(* IEC 61131-3 sources: LTL-Test-Case-Generation/, 14 files *)

(* ---- SF_DoubleValveMonitoring.st ---- *)
FUNCTION_BLOCK SF_DoubleValveMonitoring
VAR_INPUT
    Activate: BOOL;
    InitTime: TIME := T#500MS;
    S_OutControl: BOOL;
    EDM1: BOOL;
    EDM2: BOOL;
    ValveType: BOOL;
    MonitoringTime: TIME := T#100ms;
    S_StartReset: BOOL;
    Reset: BOOL;
END_VAR
VAR_OUTPUT
    Ready: BOOL;
    S_SafeState: BOOL;
    S_ValveOut: BOOL;
    S_ValveStatus: UINT;
    SafetyDemand: BOOL;
    ResetRequest: BOOL;
    Error: BOOL;
    DiagCode: UINT;
END_VAR
VAR
    T_Init: TON;
    T_Monitoring: TON;
    EDM1_: BOOL;
    EDM2_: BOOL;
    Reset_Before: BOOL;
    S_OutControl_Before: BOOL;
END_VAR

BEGIN

// state changes
IF NOT Activate THEN
    DiagCode := 16#0000;

    T_Init(IN:=0);
    T_Monitoring(IN:=0);

    Ready := FALSE;
    S_SafeState := FALSE;
    S_ValveOut := FALSE;
    SafetyDemand := FALSE;
    ResetRequest := FALSE;
    Error := FALSE;
    S_ValveStatus := DiagCode;

    Reset_Before := FALSE;
    S_OutControl_Before := FALSE;
    IF ValveType THEN
        EDM1_ := EDM1;
        EDM2_ := EDM2;
    ELSE
        EDM1_ := NOT EDM1;
        EDM2_ := NOT EDM2;
    END_IF;

ELSE
    T_Init(PT:=InitTime);
    T_Monitoring(PT:=MonitoringTime);

    IF ValveType THEN
        EDM1_ := EDM1;
        EDM2_ := EDM2;
    ELSE
        EDM1_ := NOT EDM1;
        EDM2_ := NOT EDM2;
    END_IF;

    CASE DiagCode OF
    16#0000:
        T_Init(IN:=0);
        T_Monitoring(IN:=0);
        T_Init(IN:=1, PT:=InitTime);
        DiagCode := 16#83FF;
    16#83FF:
        IF T_Init.Q THEN
            DiagCode := 16#8401;
        END_IF;
    16#8401:
        IF Reset_Before AND Reset THEN
            DiagCode := 16#C001;
        ELSIF NOT Reset_Before AND Reset AND NOT S_OutControl_Before AND S_OutControl AND NOT S_StartReset THEN
            DiagCode := 16#C100;
        ELSIF (NOT Reset_Before AND Reset) OR S_StartReset THEN
            T_Monitoring(IN:=0);T_Monitoring(IN:=1, PT:=MonitoringTime);
            DiagCode := 16#8802;
        END_IF;
    16#C001:
        IF NOT Reset THEN
            DiagCode := 16#8401;
        END_IF;
    16#C100:
        IF NOT Reset THEN
            DiagCode := 16#8401;
        END_IF;
    16#8802:
        IF S_OutControl AND NOT EDM1_ AND NOT EDM2_ THEN
            T_Monitoring(IN:=0);
            DiagCode := 16#C030;
        ELSIF S_OutControl AND EDM1_ AND NOT EDM2_ THEN
            T_Monitoring(IN:=0);
            DiagCode := 16#C020;
        ELSIF S_OutControl AND NOT EDM1_ AND EDM2_ THEN
            T_Monitoring(IN:=0);
            DiagCode := 16#C010;
        ELSIF T_Monitoring.Q AND NOT EDM1_ AND NOT EDM2_ THEN
            DiagCode := 16#C060;
        ELSIF T_Monitoring.Q AND EDM1_ AND NOT EDM2_ THEN
            DiagCode := 16#C050;
        ELSIF T_Monitoring.Q AND NOT EDM1_ AND EDM2_ THEN
            DiagCode := 16#C040;
        ELSIF EDM1_ AND EDM2_ THEN
            T_Monitoring(IN:=0);
            DiagCode := 16#8804;
        END_IF;
    16#8804:
        IF NOT EDM1_ AND NOT EDM2_ THEN
            DiagCode := 16#C060;
        ELSIF EDM1_ AND NOT EDM2_ THEN
            DiagCode := 16#C050;
        ELSIF NOT EDM1_ AND EDM2_ THEN
            DiagCode := 16#C040;
        ELSIF S_OutControl THEN
            T_Monitoring(IN:=0);T_Monitoring(IN:=1, PT:=MonitoringTime);
            DiagCode := 16#8020;
        END_IF;
    16#8020:
        IF T_Monitoring.Q AND EDM1_ AND EDM2_ THEN
            DiagCode := 16#C090;
        ELSIF T_Monitoring.Q AND NOT EDM1_ AND EDM2_ THEN
            DiagCode := 16#C080;
        ELSIF T_Monitoring.Q AND EDM1_ AND NOT EDM2_ THEN
            DiagCode := 16#C070;
        ELSIF NOT S_OutControl THEN
            T_Monitoring(IN:=0);T_Monitoring(IN:=1, PT:=MonitoringTime);
            DiagCode := 16#8802;
        ELSIF NOT EDM1_ AND NOT EDM2_ THEN
            T_Monitoring(IN:=0);
            DiagCode := 16#8010;
        END_IF;
    16#8010:
        IF EDM1_ AND EDM2_ THEN
            DiagCode := 16#C090;
        ELSIF  NOT EDM1_ AND EDM2_ THEN
            DiagCode := 16#C080;
        ELSIF EDM1_ AND NOT EDM2_ THEN
            DiagCode := 16#C070;
        ELSIF NOT S_OutControl THEN
            T_Monitoring(IN:=0);T_Monitoring(IN:=1, PT:=MonitoringTime);
            DiagCode := 16#8802;
        END_IF;
    16#C010:
        IF Reset_Before AND Reset THEN
            DiagCode := DiagCode + 1;
        ELSIF NOT Reset_Before AND Reset AND NOT S_OutControl AND EDM1_ AND EDM2_ THEN
            T_Monitoring(IN:=0);T_Monitoring(IN:=1, PT:=MonitoringTime);
            DiagCode := 16#8802;
        ELSIF NOT S_OutControl THEN
            DiagCode := DiagCode + 16#400;
        END_IF;
    16#C020:
        IF Reset_Before AND Reset THEN
            DiagCode := DiagCode + 1;
        ELSIF NOT Reset_Before AND Reset AND NOT S_OutControl AND EDM1_ AND EDM2_ THEN
            T_Monitoring(IN:=0);T_Monitoring(IN:=1, PT:=MonitoringTime);
            DiagCode := 16#8802;
        ELSIF NOT S_OutControl THEN
            DiagCode := DiagCode + 16#400;
        END_IF;
    16#C030:
        IF Reset_Before AND Reset THEN
            DiagCode := DiagCode + 1;
        ELSIF NOT Reset_Before AND Reset AND NOT S_OutControl AND EDM1_ AND EDM2_ THEN
            T_Monitoring(IN:=0);T_Monitoring(IN:=1, PT:=MonitoringTime);
            DiagCode := 16#8802;
        ELSIF NOT S_OutControl THEN
            DiagCode := DiagCode + 16#400;
        END_IF;
    16#C040:
        IF Reset_Before AND Reset THEN
            DiagCode := DiagCode + 1;
        ELSIF NOT Reset_Before AND Reset AND NOT S_OutControl AND EDM1_ AND EDM2_ THEN
            T_Monitoring(IN:=0);T_Monitoring(IN:=1, PT:=MonitoringTime);
            DiagCode := 16#8802;
        ELSIF NOT S_OutControl THEN
            DiagCode := DiagCode + 16#400;
        END_IF;
    16#C050:
        IF Reset_Before AND Reset THEN
            DiagCode := DiagCode + 1;
        ELSIF NOT Reset_Before AND Reset AND NOT S_OutControl AND EDM1_ AND EDM2_ THEN
            T_Monitoring(IN:=0);T_Monitoring(IN:=1, PT:=MonitoringTime);
            DiagCode := 16#8802;
        ELSIF NOT S_OutControl THEN
            DiagCode := DiagCode + 16#400;
        END_IF;
    16#C060:
        IF Reset_Before AND Reset THEN
            DiagCode := DiagCode + 1;
        ELSIF NOT Reset_Before AND Reset AND NOT S_OutControl AND EDM1_ AND EDM2_ THEN
            T_Monitoring(IN:=0);T_Monitoring(IN:=1, PT:=MonitoringTime);
            DiagCode := 16#8802;
        ELSIF NOT S_OutControl THEN
            DiagCode := DiagCode + 16#400;
        END_IF;
    16#C070:
        IF Reset_Before AND Reset THEN
            DiagCode := DiagCode + 1;
        ELSIF NOT Reset_Before AND Reset AND NOT S_OutControl AND EDM1_ AND EDM2_ THEN
            T_Monitoring(IN:=0);T_Monitoring(IN:=1, PT:=MonitoringTime);
            DiagCode := 16#8802;
        ELSIF NOT S_OutControl THEN
            DiagCode := DiagCode + 16#400;
        END_IF;
    16#C080:
        IF Reset_Before AND Reset THEN
            DiagCode := DiagCode + 1;
        ELSIF NOT Reset_Before AND Reset AND NOT S_OutControl AND EDM1_ AND EDM2_ THEN
            T_Monitoring(IN:=0);T_Monitoring(IN:=1, PT:=MonitoringTime);
            DiagCode := 16#8802;
        ELSIF NOT S_OutControl THEN
            DiagCode := DiagCode + 16#400;
        END_IF;
    16#C090:
        IF Reset_Before AND Reset THEN
            DiagCode := DiagCode + 1;
        ELSIF NOT Reset_Before AND Reset AND NOT S_OutControl AND EDM1_ AND EDM2_ THEN
            T_Monitoring(IN:=0);T_Monitoring(IN:=1, PT:=MonitoringTime);
            DiagCode := 16#8802;
        ELSIF NOT S_OutControl THEN
            DiagCode := DiagCode + 16#400;
        END_IF;
    16#C011:
        IF NOT Reset THEN
            DiagCode := DiagCode - 1;
        END_IF;
    16#C021:
        IF NOT Reset THEN
            DiagCode := DiagCode - 1;
        END_IF;
    16#C031:
        IF NOT Reset THEN
            DiagCode := DiagCode - 1;
        END_IF;
    16#C041:
        IF NOT Reset THEN
            DiagCode := DiagCode - 1;
        END_IF;
    16#C051:
        IF NOT Reset THEN
            DiagCode := DiagCode - 1;
        END_IF;
    16#C061:
        IF NOT Reset THEN
            DiagCode := DiagCode - 1;
        END_IF;
    16#C071:
        IF NOT Reset THEN
            DiagCode := DiagCode - 1;
        END_IF;
    16#C081:
        IF NOT Reset THEN
            DiagCode := DiagCode - 1;
        END_IF;
    16#C091:
        IF NOT Reset THEN
            DiagCode := DiagCode - 1;
        END_IF;
    16#C410:
        IF Reset_Before AND Reset THEN
            DiagCode := DiagCode - 16#400 + 1;
        ELSIF NOT Reset_Before AND Reset AND NOT S_OutControl AND EDM1_ AND EDM2_ THEN
            T_Monitoring(IN:=0);T_Monitoring(IN:=1, PT:=MonitoringTime);
            DiagCode := 16#8802;
        ELSIF S_OutControl THEN
            DiagCode := DiagCode - 16#400;
        END_IF;
    16#C420:
        IF Reset_Before AND Reset THEN
            DiagCode := DiagCode - 16#400 + 1;
        ELSIF NOT Reset_Before AND Reset AND NOT S_OutControl AND EDM1_ AND EDM2_ THEN
            T_Monitoring(IN:=0);T_Monitoring(IN:=1, PT:=MonitoringTime);
            DiagCode := 16#8802;
        ELSIF S_OutControl THEN
            DiagCode := DiagCode - 16#400;
        END_IF;
    16#C430:
        IF Reset_Before AND Reset THEN
            DiagCode := DiagCode - 16#400 + 1;
        ELSIF NOT Reset_Before AND Reset AND NOT S_OutControl AND EDM1_ AND EDM2_ THEN
            T_Monitoring(IN:=0);T_Monitoring(IN:=1, PT:=MonitoringTime);
            DiagCode := 16#8802;
        ELSIF S_OutControl THEN
            DiagCode := DiagCode - 16#400;
        END_IF;
    16#C440:
        IF Reset_Before AND Reset THEN
            DiagCode := DiagCode - 16#400 + 1;
        ELSIF NOT Reset_Before AND Reset AND NOT S_OutControl AND EDM1_ AND EDM2_ THEN
            T_Monitoring(IN:=0);T_Monitoring(IN:=1, PT:=MonitoringTime);
            DiagCode := 16#8802;
        ELSIF S_OutControl THEN
            DiagCode := DiagCode - 16#400;
        END_IF;
    16#C450:
        IF Reset_Before AND Reset THEN
            DiagCode := DiagCode - 16#400 + 1;
        ELSIF NOT Reset_Before AND Reset AND NOT S_OutControl AND EDM1_ AND EDM2_ THEN
            T_Monitoring(IN:=0);T_Monitoring(IN:=1, PT:=MonitoringTime);
            DiagCode := 16#8802;
        ELSIF S_OutControl THEN
            DiagCode := DiagCode - 16#400;
        END_IF;
    16#C460:
        IF Reset_Before AND Reset THEN
            DiagCode := DiagCode - 16#400 + 1;
        ELSIF NOT Reset_Before AND Reset AND NOT S_OutControl AND EDM1_ AND EDM2_ THEN
            T_Monitoring(IN:=0);T_Monitoring(IN:=1, PT:=MonitoringTime);
            DiagCode := 16#8802;
        ELSIF S_OutControl THEN
            DiagCode := DiagCode - 16#400;
        END_IF;
    16#C470:
        IF Reset_Before AND Reset THEN
            DiagCode := DiagCode - 16#400 + 1;
        ELSIF NOT Reset_Before AND Reset AND NOT S_OutControl AND EDM1_ AND EDM2_ THEN
            T_Monitoring(IN:=0);T_Monitoring(IN:=1, PT:=MonitoringTime);
            DiagCode := 16#8802;
        ELSIF S_OutControl THEN
            DiagCode := DiagCode - 16#400;
        END_IF;
    16#C480:
        IF Reset_Before AND Reset THEN
            DiagCode := DiagCode - 16#400 + 1;
        ELSIF NOT Reset_Before AND Reset AND NOT S_OutControl AND EDM1_ AND EDM2_ THEN
            T_Monitoring(IN:=0);T_Monitoring(IN:=1, PT:=MonitoringTime);
            DiagCode := 16#8802;
        ELSIF S_OutControl THEN
            DiagCode := DiagCode - 16#400;
        END_IF;
    16#C490:
        IF Reset_Before AND Reset THEN
            DiagCode := DiagCode - 16#400 + 1;
        ELSIF NOT Reset_Before AND Reset AND NOT S_OutControl AND EDM1_ AND EDM2_ THEN
            T_Monitoring(IN:=0);T_Monitoring(IN:=1, PT:=MonitoringTime);
            DiagCode := 16#8802;
        ELSIF S_OutControl THEN
            DiagCode := DiagCode - 16#400;
        END_IF;
    END_CASE;
    CASE DiagCode OF
    16#C010:
        IF NOT S_OutControl THEN
            DiagCode := DiagCode + 16#400;
        END_IF;
    16#C020:
        IF NOT S_OutControl THEN
            DiagCode := DiagCode + 16#400;
        END_IF;
    16#C030:
        IF NOT S_OutControl THEN
            DiagCode := DiagCode + 16#400;
        END_IF;
    16#C040:
        IF NOT S_OutControl THEN
            DiagCode := DiagCode + 16#400;
        END_IF;
    16#C050:
        IF NOT S_OutControl THEN
            DiagCode := DiagCode + 16#400;
        END_IF;
    16#C060:
        IF NOT S_OutControl THEN
            DiagCode := DiagCode + 16#400;
        END_IF;
    16#C070:
        IF NOT S_OutControl THEN
            DiagCode := DiagCode + 16#400;
        END_IF;
    16#C080:
        IF NOT S_OutControl THEN
            DiagCode := DiagCode + 16#400;
        END_IF;
    16#C090:
        IF NOT S_OutControl THEN
            DiagCode := DiagCode + 16#400;
        END_IF;
    END_CASE;

    // set output variables
    S_ValveStatus := DiagCode;

    IF DiagCode > 16#C000 THEN
        Ready := TRUE;
        S_SafeState := FALSE;
        S_ValveOut := FALSE;
        SafetyDemand := FALSE;
        ResetRequest := FALSE;
        Error := TRUE;
    END_IF;
    IF DiagCode > 16#C400 THEN
        ResetRequest := TRUE;
    END_IF;

    CASE DiagCode OF
    16#83FF:
        Ready := TRUE;
        S_SafeState := FALSE;
        S_ValveOut := FALSE;
        SafetyDemand := FALSE;
        ResetRequest := FALSE;
        Error := FALSE;
    16#8401:
        Ready := TRUE;
        S_SafeState := FALSE;
        S_ValveOut := FALSE;
        SafetyDemand := FALSE;
        ResetRequest := TRUE;
        Error := FALSE;
    16#8802:
        Ready := TRUE;
        S_SafeState := FALSE;
        S_ValveOut := FALSE;
        SafetyDemand := TRUE;
        ResetRequest := FALSE;
        Error := FALSE;
    16#8804:
        Ready := TRUE;
        S_SafeState := TRUE;
        S_ValveOut := FALSE;
        SafetyDemand := TRUE;
        ResetRequest := FALSE;
        Error := FALSE;
    16#8010:
        Ready := TRUE;
        S_SafeState := FALSE;
        S_ValveOut := TRUE;
        SafetyDemand := FALSE;
        ResetRequest := FALSE;
        Error := FALSE;
    16#8020:
        Ready := TRUE;
        S_SafeState := FALSE;
        S_ValveOut := TRUE;
        SafetyDemand := FALSE;
        ResetRequest := FALSE;
        Error := FALSE;
    END_CASE;

    Reset_Before := Reset;
    S_OutControl_Before := S_OutControl;
END_IF;

END_FUNCTION_BLOCK

(* ---- SF_DoubleValveMonitoring_Test.st ---- *)
FUNCTION_BLOCK SF_DoubleValveMonitoring_Test
VAR_INPUT
END_VAR
VAR_OUTPUT
	failed_0: BOOL := FALSE;
	finished_0: BOOL := FALSE;
END_VAR
VAR
	fb_0: SF_DoubleValveMonitoring_BranchCounters;
	waitCounter_0: UINT := 0;
	testState_0: UINT := 0;
END_VAR

IF NOT failed_0 AND NOT finished_0 THEN
CASE testState_0 OF
0:
	fb_0.Activate := FALSE;
	fb_0();
	failed_0 := NOT ((((((((((((NOT (fb_0.Reset_Before) AND NOT (fb_0.S_OutControl_Before)) AND NOT (fb_0.T_Init.Q)) AND NOT (fb_0.T_Monitoring.Q)) AND (fb_0.DiagCode = 0)) AND NOT (fb_0.Ready)) AND NOT (fb_0.S_SafeState)) AND NOT (fb_0.S_ValveOut)) AND (fb_0.S_ValveStatus = fb_0.DiagCode)) AND NOT (fb_0.SafetyDemand)) AND NOT (fb_0.ResetRequest)) AND NOT (fb_0.Error)));
	testState_0 := testState_0 + 1;
1:
	fb_0.Activate := TRUE; fb_0.S_OutControl := FALSE; fb_0.EDM1 := FALSE; fb_0.EDM2 := FALSE; fb_0.ValveType := TRUE; fb_0.S_StartReset := FALSE; fb_0.Reset := FALSE;
	fb_0();
	failed_0 := NOT ((((((((((((NOT (fb_0.Reset_Before) AND NOT (fb_0.S_OutControl_Before)) AND NOT (fb_0.T_Init.Q)) AND NOT (fb_0.T_Monitoring.Q)) AND (fb_0.DiagCode = 33791)) AND fb_0.Ready) AND NOT (fb_0.S_SafeState)) AND NOT (fb_0.S_ValveOut)) AND (fb_0.S_ValveStatus = fb_0.DiagCode)) AND NOT (fb_0.SafetyDemand)) AND NOT (fb_0.ResetRequest)) AND NOT (fb_0.Error)));
	testState_0 := testState_0 + 1;
2:
	IF (fb_0.T_Init.Q AND (fb_0.DiagCode = 33793)) THEN
		waitCounter_0 := 0;
		testState_0 := testState_0 + 1;
	ELSE
		failed_0 := NOT ((NOT (fb_0.Reset_Before) AND (NOT (fb_0.S_OutControl_Before) AND (NOT (fb_0.T_Init.Q) AND (NOT (fb_0.T_Monitoring.Q) AND ((fb_0.DiagCode = 33791) AND (fb_0.Ready AND (NOT (fb_0.S_SafeState) AND (NOT (fb_0.S_ValveOut) AND ((fb_0.S_ValveStatus = fb_0.DiagCode) AND (NOT (fb_0.SafetyDemand) AND (NOT (fb_0.ResetRequest) AND NOT (fb_0.Error)))))))))))));
		IF waitCounter_0 > 100 THEN
			finished_0 := TRUE;
		ELSE
			waitCounter_0 := waitCounter_0 + 1;
			fb_0();
		END_IF
	END_IF
3:
	failed_0 := NOT ((((((((((((NOT (fb_0.Reset_Before) AND NOT (fb_0.S_OutControl_Before)) AND fb_0.T_Init.Q) AND NOT (fb_0.T_Monitoring.Q)) AND (fb_0.DiagCode = 33793)) AND fb_0.Ready) AND NOT (fb_0.S_SafeState)) AND NOT (fb_0.S_ValveOut)) AND (fb_0.S_ValveStatus = fb_0.DiagCode)) AND NOT (fb_0.SafetyDemand)) AND fb_0.ResetRequest) AND NOT (fb_0.Error)));
	testState_0 := testState_0 + 1;
4:
	fb_0.Activate := TRUE; fb_0.S_OutControl := TRUE; fb_0.EDM1 := FALSE; fb_0.EDM2 := FALSE; fb_0.ValveType := TRUE; fb_0.S_StartReset := FALSE; fb_0.Reset := TRUE;
	fb_0();
	failed_0 := NOT ((((((((((((fb_0.Reset_Before AND fb_0.S_OutControl_Before) AND fb_0.T_Init.Q) AND NOT (fb_0.T_Monitoring.Q)) AND (fb_0.DiagCode = 49408)) AND fb_0.Ready) AND NOT (fb_0.S_SafeState)) AND NOT (fb_0.S_ValveOut)) AND (fb_0.S_ValveStatus = fb_0.DiagCode)) AND NOT (fb_0.SafetyDemand)) AND NOT (fb_0.ResetRequest)) AND fb_0.Error));
	testState_0 := testState_0 + 1;
5:
	fb_0.Activate := TRUE; fb_0.S_OutControl := TRUE; fb_0.EDM1 := FALSE; fb_0.EDM2 := FALSE; fb_0.ValveType := TRUE; fb_0.S_StartReset := FALSE; fb_0.Reset := TRUE;
	fb_0();
	failed_0 := NOT ((((((((((((fb_0.Reset_Before AND fb_0.S_OutControl_Before) AND fb_0.T_Init.Q) AND NOT (fb_0.T_Monitoring.Q)) AND (fb_0.DiagCode = 49408)) AND fb_0.Ready) AND NOT (fb_0.S_SafeState)) AND NOT (fb_0.S_ValveOut)) AND (fb_0.S_ValveStatus = fb_0.DiagCode)) AND NOT (fb_0.SafetyDemand)) AND NOT (fb_0.ResetRequest)) AND fb_0.Error));
	testState_0 := testState_0 + 1;
6:
	fb_0.Activate := TRUE; fb_0.S_OutControl := TRUE; fb_0.EDM1 := FALSE; fb_0.EDM2 := FALSE; fb_0.ValveType := TRUE; fb_0.S_StartReset := FALSE; fb_0.Reset := FALSE;
	fb_0();
	failed_0 := NOT ((((((((((((NOT (fb_0.Reset_Before) AND fb_0.S_OutControl_Before) AND fb_0.T_Init.Q) AND NOT (fb_0.T_Monitoring.Q)) AND (fb_0.DiagCode = 33793)) AND fb_0.Ready) AND NOT (fb_0.S_SafeState)) AND NOT (fb_0.S_ValveOut)) AND (fb_0.S_ValveStatus = fb_0.DiagCode)) AND NOT (fb_0.SafetyDemand)) AND fb_0.ResetRequest) AND NOT (fb_0.Error)));
	testState_0 := testState_0 + 1;
7:
	fb_0.Activate := TRUE; fb_0.S_OutControl := FALSE; fb_0.EDM1 := FALSE; fb_0.EDM2 := FALSE; fb_0.ValveType := TRUE; fb_0.S_StartReset := FALSE; fb_0.Reset := FALSE;
	fb_0();
	failed_0 := NOT ((((((((((((NOT (fb_0.Reset_Before) AND NOT (fb_0.S_OutControl_Before)) AND fb_0.T_Init.Q) AND NOT (fb_0.T_Monitoring.Q)) AND (fb_0.DiagCode = 33793)) AND fb_0.Ready) AND NOT (fb_0.S_SafeState)) AND NOT (fb_0.S_ValveOut)) AND (fb_0.S_ValveStatus = fb_0.DiagCode)) AND NOT (fb_0.SafetyDemand)) AND fb_0.ResetRequest) AND NOT (fb_0.Error)));
	testState_0 := testState_0 + 1;
8:
	fb_0.Activate := FALSE; fb_0.S_OutControl := FALSE; fb_0.EDM1 := FALSE; fb_0.EDM2 := FALSE; fb_0.ValveType := TRUE; fb_0.S_StartReset := FALSE; fb_0.Reset := FALSE;
	fb_0();
	failed_0 := NOT ((((((((((((NOT (fb_0.Reset_Before) AND NOT (fb_0.S_OutControl_Before)) AND NOT (fb_0.T_Init.Q)) AND NOT (fb_0.T_Monitoring.Q)) AND (fb_0.DiagCode = 0)) AND NOT (fb_0.Ready)) AND NOT (fb_0.S_SafeState)) AND NOT (fb_0.S_ValveOut)) AND (fb_0.S_ValveStatus = fb_0.DiagCode)) AND NOT (fb_0.SafetyDemand)) AND NOT (fb_0.ResetRequest)) AND NOT (fb_0.Error)));
	testState_0 := testState_0 + 1;
9:
	fb_0.Activate := TRUE; fb_0.S_OutControl := FALSE; fb_0.EDM1 := FALSE; fb_0.EDM2 := FALSE; fb_0.ValveType := TRUE; fb_0.S_StartReset := FALSE; fb_0.Reset := TRUE;
	fb_0();
	failed_0 := NOT ((((((((((((fb_0.Reset_Before AND NOT (fb_0.S_OutControl_Before)) AND NOT (fb_0.T_Init.Q)) AND NOT (fb_0.T_Monitoring.Q)) AND (fb_0.DiagCode = 33791)) AND fb_0.Ready) AND NOT (fb_0.S_SafeState)) AND NOT (fb_0.S_ValveOut)) AND (fb_0.S_ValveStatus = fb_0.DiagCode)) AND NOT (fb_0.SafetyDemand)) AND NOT (fb_0.ResetRequest)) AND NOT (fb_0.Error)));
	testState_0 := testState_0 + 1;
10:
	IF (fb_0.T_Init.Q AND (fb_0.DiagCode = 33793)) THEN
		waitCounter_0 := 0;
		testState_0 := testState_0 + 1;
	ELSE
		failed_0 := NOT ((fb_0.Reset_Before AND (NOT (fb_0.S_OutControl_Before) AND (NOT (fb_0.T_Init.Q) AND (NOT (fb_0.T_Monitoring.Q) AND ((fb_0.DiagCode = 33791) AND (fb_0.Ready AND (NOT (fb_0.S_SafeState) AND (NOT (fb_0.S_ValveOut) AND ((fb_0.S_ValveStatus = fb_0.DiagCode) AND (NOT (fb_0.SafetyDemand) AND (NOT (fb_0.ResetRequest) AND NOT (fb_0.Error)))))))))))));
		IF waitCounter_0 > 100 THEN
			finished_0 := TRUE;
		ELSE
			waitCounter_0 := waitCounter_0 + 1;
			fb_0();
		END_IF
	END_IF
11:
	failed_0 := NOT ((((((((((((fb_0.Reset_Before AND NOT (fb_0.S_OutControl_Before)) AND fb_0.T_Init.Q) AND NOT (fb_0.T_Monitoring.Q)) AND (fb_0.DiagCode = 33793)) AND fb_0.Ready) AND NOT (fb_0.S_SafeState)) AND NOT (fb_0.S_ValveOut)) AND (fb_0.S_ValveStatus = fb_0.DiagCode)) AND NOT (fb_0.SafetyDemand)) AND fb_0.ResetRequest) AND NOT (fb_0.Error)));
	testState_0 := testState_0 + 1;
12:
	fb_0.Activate := TRUE; fb_0.S_OutControl := FALSE; fb_0.EDM1 := FALSE; fb_0.EDM2 := FALSE; fb_0.ValveType := TRUE; fb_0.S_StartReset := FALSE; fb_0.Reset := TRUE;
	fb_0();
	failed_0 := NOT ((((((((((((fb_0.Reset_Before AND NOT (fb_0.S_OutControl_Before)) AND fb_0.T_Init.Q) AND NOT (fb_0.T_Monitoring.Q)) AND (fb_0.DiagCode = 49153)) AND fb_0.Ready) AND NOT (fb_0.S_SafeState)) AND NOT (fb_0.S_ValveOut)) AND (fb_0.S_ValveStatus = fb_0.DiagCode)) AND NOT (fb_0.SafetyDemand)) AND NOT (fb_0.ResetRequest)) AND fb_0.Error));
	testState_0 := testState_0 + 1;
13:
	fb_0.Activate := TRUE; fb_0.S_OutControl := FALSE; fb_0.EDM1 := FALSE; fb_0.EDM2 := FALSE; fb_0.ValveType := TRUE; fb_0.S_StartReset := FALSE; fb_0.Reset := TRUE;
	fb_0();
	failed_0 := NOT ((((((((((((fb_0.Reset_Before AND NOT (fb_0.S_OutControl_Before)) AND fb_0.T_Init.Q) AND NOT (fb_0.T_Monitoring.Q)) AND (fb_0.DiagCode = 49153)) AND fb_0.Ready) AND NOT (fb_0.S_SafeState)) AND NOT (fb_0.S_ValveOut)) AND (fb_0.S_ValveStatus = fb_0.DiagCode)) AND NOT (fb_0.SafetyDemand)) AND NOT (fb_0.ResetRequest)) AND fb_0.Error));
	testState_0 := testState_0 + 1;
14:
	fb_0.Activate := TRUE; fb_0.S_OutControl := FALSE; fb_0.EDM1 := FALSE; fb_0.EDM2 := FALSE; fb_0.ValveType := TRUE; fb_0.S_StartReset := FALSE; fb_0.Reset := FALSE;
	fb_0();
	failed_0 := NOT ((((((((((((NOT (fb_0.Reset_Before) AND NOT (fb_0.S_OutControl_Before)) AND fb_0.T_Init.Q) AND NOT (fb_0.T_Monitoring.Q)) AND (fb_0.DiagCode = 33793)) AND fb_0.Ready) AND NOT (fb_0.S_SafeState)) AND NOT (fb_0.S_ValveOut)) AND (fb_0.S_ValveStatus = fb_0.DiagCode)) AND NOT (fb_0.SafetyDemand)) AND fb_0.ResetRequest) AND NOT (fb_0.Error)));
	testState_0 := testState_0 + 1;
15:
	fb_0.Activate := TRUE; fb_0.S_OutControl := FALSE; fb_0.EDM1 := FALSE; fb_0.EDM2 := FALSE; fb_0.ValveType := TRUE; fb_0.S_StartReset := FALSE; fb_0.Reset := TRUE;
	fb_0();
	failed_0 := NOT ((((((((((((fb_0.Reset_Before AND NOT (fb_0.S_OutControl_Before)) AND fb_0.T_Init.Q) AND NOT (fb_0.T_Monitoring.Q)) AND (fb_0.DiagCode = 34818)) AND fb_0.Ready) AND NOT (fb_0.S_SafeState)) AND NOT (fb_0.S_ValveOut)) AND (fb_0.S_ValveStatus = fb_0.DiagCode)) AND fb_0.SafetyDemand) AND NOT (fb_0.ResetRequest)) AND NOT (fb_0.Error)));
	testState_0 := testState_0 + 1;
16:
	fb_0.Activate := FALSE; fb_0.S_OutControl := FALSE; fb_0.EDM1 := FALSE; fb_0.EDM2 := FALSE; fb_0.ValveType := TRUE; fb_0.S_StartReset := FALSE; fb_0.Reset := FALSE;
	fb_0();
	failed_0 := NOT ((((((((((((NOT (fb_0.Reset_Before) AND NOT (fb_0.S_OutControl_Before)) AND NOT (fb_0.T_Init.Q)) AND NOT (fb_0.T_Monitoring.Q)) AND (fb_0.DiagCode = 0)) AND NOT (fb_0.Ready)) AND NOT (fb_0.S_SafeState)) AND NOT (fb_0.S_ValveOut)) AND (fb_0.S_ValveStatus = fb_0.DiagCode)) AND NOT (fb_0.SafetyDemand)) AND NOT (fb_0.ResetRequest)) AND NOT (fb_0.Error)));
	testState_0 := testState_0 + 1;
17:
	fb_0.Activate := TRUE; fb_0.S_OutControl := FALSE; fb_0.EDM1 := FALSE; fb_0.EDM2 := FALSE; fb_0.ValveType := TRUE; fb_0.S_StartReset := TRUE; fb_0.Reset := FALSE;
	fb_0();
	failed_0 := NOT ((((((((((((NOT (fb_0.Reset_Before) AND NOT (fb_0.S_OutControl_Before)) AND NOT (fb_0.T_Init.Q)) AND NOT (fb_0.T_Monitoring.Q)) AND (fb_0.DiagCode = 33791)) AND fb_0.Ready) AND NOT (fb_0.S_SafeState)) AND NOT (fb_0.S_ValveOut)) AND (fb_0.S_ValveStatus = fb_0.DiagCode)) AND NOT (fb_0.SafetyDemand)) AND NOT (fb_0.ResetRequest)) AND NOT (fb_0.Error)));
	testState_0 := testState_0 + 1;
18:
	IF (fb_0.T_Init.Q AND (fb_0.DiagCode = 33793)) THEN
		waitCounter_0 := 0;
		testState_0 := testState_0 + 1;
	ELSE
		failed_0 := NOT ((NOT (fb_0.Reset_Before) AND (NOT (fb_0.S_OutControl_Before) AND (NOT (fb_0.T_Init.Q) AND (NOT (fb_0.T_Monitoring.Q) AND ((fb_0.DiagCode = 33791) AND (fb_0.Ready AND (NOT (fb_0.S_SafeState) AND (NOT (fb_0.S_ValveOut) AND ((fb_0.S_ValveStatus = fb_0.DiagCode) AND (NOT (fb_0.SafetyDemand) AND (NOT (fb_0.ResetRequest) AND NOT (fb_0.Error)))))))))))));
		IF waitCounter_0 > 100 THEN
			finished_0 := TRUE;
		ELSE
			waitCounter_0 := waitCounter_0 + 1;
			fb_0();
		END_IF
	END_IF
19:
	failed_0 := NOT ((((((((((((NOT (fb_0.Reset_Before) AND NOT (fb_0.S_OutControl_Before)) AND fb_0.T_Init.Q) AND NOT (fb_0.T_Monitoring.Q)) AND (fb_0.DiagCode = 33793)) AND fb_0.Ready) AND NOT (fb_0.S_SafeState)) AND NOT (fb_0.S_ValveOut)) AND (fb_0.S_ValveStatus = fb_0.DiagCode)) AND NOT (fb_0.SafetyDemand)) AND fb_0.ResetRequest) AND NOT (fb_0.Error)));
	testState_0 := testState_0 + 1;
20:
	fb_0.Activate := TRUE; fb_0.S_OutControl := FALSE; fb_0.EDM1 := FALSE; fb_0.EDM2 := TRUE; fb_0.ValveType := TRUE; fb_0.S_StartReset := TRUE; fb_0.Reset := FALSE;
	fb_0();
	failed_0 := NOT ((((((((((((NOT (fb_0.Reset_Before) AND NOT (fb_0.S_OutControl_Before)) AND fb_0.T_Init.Q) AND NOT (fb_0.T_Monitoring.Q)) AND (fb_0.DiagCode = 34818)) AND fb_0.Ready) AND NOT (fb_0.S_SafeState)) AND NOT (fb_0.S_ValveOut)) AND (fb_0.S_ValveStatus = fb_0.DiagCode)) AND fb_0.SafetyDemand) AND NOT (fb_0.ResetRequest)) AND NOT (fb_0.Error)));
	testState_0 := testState_0 + 1;
21:
	IF (fb_0.T_Monitoring.Q AND (fb_0.DiagCode = 50240)) THEN
		waitCounter_0 := 0;
		testState_0 := testState_0 + 1;
	ELSE
		failed_0 := NOT ((NOT (fb_0.Reset_Before) AND (NOT (fb_0.S_OutControl_Before) AND (fb_0.T_Init.Q AND (NOT (fb_0.T_Monitoring.Q) AND ((fb_0.DiagCode = 34818) AND (fb_0.Ready AND (NOT (fb_0.S_SafeState) AND (NOT (fb_0.S_ValveOut) AND ((fb_0.S_ValveStatus = fb_0.DiagCode) AND (fb_0.SafetyDemand AND (NOT (fb_0.ResetRequest) AND NOT (fb_0.Error)))))))))))));
		IF waitCounter_0 > 100 THEN
			finished_0 := TRUE;
		ELSE
			waitCounter_0 := waitCounter_0 + 1;
			fb_0();
		END_IF
	END_IF
22:
	failed_0 := NOT ((((((((((((NOT (fb_0.Reset_Before) AND NOT (fb_0.S_OutControl_Before)) AND fb_0.T_Init.Q) AND fb_0.T_Monitoring.Q) AND (fb_0.DiagCode = 50240)) AND fb_0.Ready) AND NOT (fb_0.S_SafeState)) AND NOT (fb_0.S_ValveOut)) AND (fb_0.S_ValveStatus = fb_0.DiagCode)) AND NOT (fb_0.SafetyDemand)) AND fb_0.ResetRequest) AND fb_0.Error));
	testState_0 := testState_0 + 1;
23:
	fb_0.Activate := TRUE; fb_0.S_OutControl := TRUE; fb_0.EDM1 := FALSE; fb_0.EDM2 := TRUE; fb_0.ValveType := TRUE; fb_0.S_StartReset := TRUE; fb_0.Reset := FALSE;
	fb_0();
	failed_0 := NOT ((((((((((((NOT (fb_0.Reset_Before) AND fb_0.S_OutControl_Before) AND fb_0.T_Init.Q) AND fb_0.T_Monitoring.Q) AND (fb_0.DiagCode = 49216)) AND fb_0.Ready) AND NOT (fb_0.S_SafeState)) AND NOT (fb_0.S_ValveOut)) AND (fb_0.S_ValveStatus = fb_0.DiagCode)) AND NOT (fb_0.SafetyDemand)) AND NOT (fb_0.ResetRequest)) AND fb_0.Error));
	testState_0 := testState_0 + 1;
24:
	fb_0.Activate := TRUE; fb_0.S_OutControl := TRUE; fb_0.EDM1 := FALSE; fb_0.EDM2 := TRUE; fb_0.ValveType := TRUE; fb_0.S_StartReset := TRUE; fb_0.Reset := TRUE;
	fb_0();
	failed_0 := NOT ((((((((((((fb_0.Reset_Before AND fb_0.S_OutControl_Before) AND fb_0.T_Init.Q) AND fb_0.T_Monitoring.Q) AND (fb_0.DiagCode = 49216)) AND fb_0.Ready) AND NOT (fb_0.S_SafeState)) AND NOT (fb_0.S_ValveOut)) AND (fb_0.S_ValveStatus = fb_0.DiagCode)) AND NOT (fb_0.SafetyDemand)) AND NOT (fb_0.ResetRequest)) AND fb_0.Error));
	testState_0 := testState_0 + 1;
25:
	fb_0.Activate := TRUE; fb_0.S_OutControl := TRUE; fb_0.EDM1 := FALSE; fb_0.EDM2 := TRUE; fb_0.ValveType := TRUE; fb_0.S_StartReset := TRUE; fb_0.Reset := TRUE;
	fb_0();
	failed_0 := NOT ((((((((((((fb_0.Reset_Before AND fb_0.S_OutControl_Before) AND fb_0.T_Init.Q) AND fb_0.T_Monitoring.Q) AND (fb_0.DiagCode = 49217)) AND fb_0.Ready) AND NOT (fb_0.S_SafeState)) AND NOT (fb_0.S_ValveOut)) AND (fb_0.S_ValveStatus = fb_0.DiagCode)) AND NOT (fb_0.SafetyDemand)) AND NOT (fb_0.ResetRequest)) AND fb_0.Error));
	testState_0 := testState_0 + 1;
26:
	fb_0.Activate := TRUE; fb_0.S_OutControl := TRUE; fb_0.EDM1 := FALSE; fb_0.EDM2 := TRUE; fb_0.ValveType := TRUE; fb_0.S_StartReset := TRUE; fb_0.Reset := TRUE;
	fb_0();
	failed_0 := NOT ((((((((((((fb_0.Reset_Before AND fb_0.S_OutControl_Before) AND fb_0.T_Init.Q) AND fb_0.T_Monitoring.Q) AND (fb_0.DiagCode = 49217)) AND fb_0.Ready) AND NOT (fb_0.S_SafeState)) AND NOT (fb_0.S_ValveOut)) AND (fb_0.S_ValveStatus = fb_0.DiagCode)) AND NOT (fb_0.SafetyDemand)) AND NOT (fb_0.ResetRequest)) AND fb_0.Error));
	testState_0 := testState_0 + 1;
27:
	fb_0.Activate := TRUE; fb_0.S_OutControl := TRUE; fb_0.EDM1 := FALSE; fb_0.EDM2 := TRUE; fb_0.ValveType := TRUE; fb_0.S_StartReset := TRUE; fb_0.Reset := FALSE;
	fb_0();
	failed_0 := NOT ((((((((((((NOT (fb_0.Reset_Before) AND fb_0.S_OutControl_Before) AND fb_0.T_Init.Q) AND fb_0.T_Monitoring.Q) AND (fb_0.DiagCode = 49216)) AND fb_0.Ready) AND NOT (fb_0.S_SafeState)) AND NOT (fb_0.S_ValveOut)) AND (fb_0.S_ValveStatus = fb_0.DiagCode)) AND NOT (fb_0.SafetyDemand)) AND NOT (fb_0.ResetRequest)) AND fb_0.Error));
	testState_0 := testState_0 + 1;
28:
	fb_0.Activate := TRUE; fb_0.S_OutControl := FALSE; fb_0.EDM1 := FALSE; fb_0.EDM2 := TRUE; fb_0.ValveType := TRUE; fb_0.S_StartReset := TRUE; fb_0.Reset := FALSE;
	fb_0();
	failed_0 := NOT ((((((((((((NOT (fb_0.Reset_Before) AND NOT (fb_0.S_OutControl_Before)) AND fb_0.T_Init.Q) AND fb_0.T_Monitoring.Q) AND (fb_0.DiagCode = 50240)) AND fb_0.Ready) AND NOT (fb_0.S_SafeState)) AND NOT (fb_0.S_ValveOut)) AND (fb_0.S_ValveStatus = fb_0.DiagCode)) AND NOT (fb_0.SafetyDemand)) AND fb_0.ResetRequest) AND fb_0.Error));
	testState_0 := testState_0 + 1;
29:
	fb_0.Activate := TRUE; fb_0.S_OutControl := TRUE; fb_0.EDM1 := FALSE; fb_0.EDM2 := TRUE; fb_0.ValveType := TRUE; fb_0.S_StartReset := TRUE; fb_0.Reset := FALSE;
	fb_0();
	failed_0 := NOT ((((((((((((NOT (fb_0.Reset_Before) AND fb_0.S_OutControl_Before) AND fb_0.T_Init.Q) AND fb_0.T_Monitoring.Q) AND (fb_0.DiagCode = 49216)) AND fb_0.Ready) AND NOT (fb_0.S_SafeState)) AND NOT (fb_0.S_ValveOut)) AND (fb_0.S_ValveStatus = fb_0.DiagCode)) AND NOT (fb_0.SafetyDemand)) AND NOT (fb_0.ResetRequest)) AND fb_0.Error));
	testState_0 := testState_0 + 1;
30:
	fb_0.Activate := TRUE; fb_0.S_OutControl := FALSE; fb_0.EDM1 := TRUE; fb_0.EDM2 := TRUE; fb_0.ValveType := TRUE; fb_0.S_StartReset := TRUE; fb_0.Reset := TRUE;
	fb_0();
	failed_0 := NOT ((((((((((((fb_0.Reset_Before AND NOT (fb_0.S_OutControl_Before)) AND fb_0.T_Init.Q) AND NOT (fb_0.T_Monitoring.Q)) AND (fb_0.DiagCode = 34818)) AND fb_0.Ready) AND NOT (fb_0.S_SafeState)) AND NOT (fb_0.S_ValveOut)) AND (fb_0.S_ValveStatus = fb_0.DiagCode)) AND fb_0.SafetyDemand) AND NOT (fb_0.ResetRequest)) AND NOT (fb_0.Error)));
	testState_0 := testState_0 + 1;
31:
	fb_0.Activate := TRUE; fb_0.S_OutControl := FALSE; fb_0.EDM1 := FALSE; fb_0.EDM2 := TRUE; fb_0.ValveType := TRUE; fb_0.S_StartReset := TRUE; fb_0.Reset := FALSE;
	fb_0();
	failed_0 := NOT ((((((((((((NOT (fb_0.Reset_Before) AND NOT (fb_0.S_OutControl_Before)) AND fb_0.T_Init.Q) AND NOT (fb_0.T_Monitoring.Q)) AND (fb_0.DiagCode = 34818)) AND fb_0.Ready) AND NOT (fb_0.S_SafeState)) AND NOT (fb_0.S_ValveOut)) AND (fb_0.S_ValveStatus = fb_0.DiagCode)) AND fb_0.SafetyDemand) AND NOT (fb_0.ResetRequest)) AND NOT (fb_0.Error)));
	testState_0 := testState_0 + 1;
32:
	IF (fb_0.T_Monitoring.Q AND (fb_0.DiagCode = 50240)) THEN
		waitCounter_0 := 0;
		testState_0 := testState_0 + 1;
	ELSE
		failed_0 := NOT ((NOT (fb_0.Reset_Before) AND (NOT (fb_0.S_OutControl_Before) AND (fb_0.T_Init.Q AND (NOT (fb_0.T_Monitoring.Q) AND ((fb_0.DiagCode = 34818) AND (fb_0.Ready AND (NOT (fb_0.S_SafeState) AND (NOT (fb_0.S_ValveOut) AND ((fb_0.S_ValveStatus = fb_0.DiagCode) AND (fb_0.SafetyDemand AND (NOT (fb_0.ResetRequest) AND NOT (fb_0.Error)))))))))))));
		IF waitCounter_0 > 100 THEN
			finished_0 := TRUE;
		ELSE
			waitCounter_0 := waitCounter_0 + 1;
			fb_0();
		END_IF
	END_IF
33:
	failed_0 := NOT ((((((((((((NOT (fb_0.Reset_Before) AND NOT (fb_0.S_OutControl_Before)) AND fb_0.T_Init.Q) AND fb_0.T_Monitoring.Q) AND (fb_0.DiagCode = 50240)) AND fb_0.Ready) AND NOT (fb_0.S_SafeState)) AND NOT (fb_0.S_ValveOut)) AND (fb_0.S_ValveStatus = fb_0.DiagCode)) AND NOT (fb_0.SafetyDemand)) AND fb_0.ResetRequest) AND fb_0.Error));
	testState_0 := testState_0 + 1;
34:
	fb_0.Activate := TRUE; fb_0.S_OutControl := FALSE; fb_0.EDM1 := FALSE; fb_0.EDM2 := TRUE; fb_0.ValveType := TRUE; fb_0.S_StartReset := TRUE; fb_0.Reset := TRUE;
	fb_0();
	failed_0 := NOT ((((((((((((fb_0.Reset_Before AND NOT (fb_0.S_OutControl_Before)) AND fb_0.T_Init.Q) AND fb_0.T_Monitoring.Q) AND (fb_0.DiagCode = 50240)) AND fb_0.Ready) AND NOT (fb_0.S_SafeState)) AND NOT (fb_0.S_ValveOut)) AND (fb_0.S_ValveStatus = fb_0.DiagCode)) AND NOT (fb_0.SafetyDemand)) AND fb_0.ResetRequest) AND fb_0.Error));
	testState_0 := testState_0 + 1;
35:
	fb_0.Activate := TRUE; fb_0.S_OutControl := FALSE; fb_0.EDM1 := FALSE; fb_0.EDM2 := TRUE; fb_0.ValveType := TRUE; fb_0.S_StartReset := TRUE; fb_0.Reset := TRUE;
	fb_0();
	failed_0 := NOT ((((((((((((fb_0.Reset_Before AND NOT (fb_0.S_OutControl_Before)) AND fb_0.T_Init.Q) AND fb_0.T_Monitoring.Q) AND (fb_0.DiagCode = 49217)) AND fb_0.Ready) AND NOT (fb_0.S_SafeState)) AND NOT (fb_0.S_ValveOut)) AND (fb_0.S_ValveStatus = fb_0.DiagCode)) AND NOT (fb_0.SafetyDemand)) AND NOT (fb_0.ResetRequest)) AND fb_0.Error));
	testState_0 := testState_0 + 1;
36:
	fb_0.Activate := TRUE; fb_0.S_OutControl := FALSE; fb_0.EDM1 := FALSE; fb_0.EDM2 := TRUE; fb_0.ValveType := TRUE; fb_0.S_StartReset := TRUE; fb_0.Reset := FALSE;
	fb_0();
	failed_0 := NOT ((((((((((((NOT (fb_0.Reset_Before) AND NOT (fb_0.S_OutControl_Before)) AND fb_0.T_Init.Q) AND fb_0.T_Monitoring.Q) AND (fb_0.DiagCode = 50240)) AND fb_0.Ready) AND NOT (fb_0.S_SafeState)) AND NOT (fb_0.S_ValveOut)) AND (fb_0.S_ValveStatus = fb_0.DiagCode)) AND NOT (fb_0.SafetyDemand)) AND fb_0.ResetRequest) AND fb_0.Error));
	testState_0 := testState_0 + 1;
37:
	fb_0.Activate := TRUE; fb_0.S_OutControl := FALSE; fb_0.EDM1 := TRUE; fb_0.EDM2 := TRUE; fb_0.ValveType := TRUE; fb_0.S_StartReset := TRUE; fb_0.Reset := TRUE;
	fb_0();
	failed_0 := NOT ((((((((((((fb_0.Reset_Before AND NOT (fb_0.S_OutControl_Before)) AND fb_0.T_Init.Q) AND NOT (fb_0.T_Monitoring.Q)) AND (fb_0.DiagCode = 34818)) AND fb_0.Ready) AND NOT (fb_0.S_SafeState)) AND NOT (fb_0.S_ValveOut)) AND (fb_0.S_ValveStatus = fb_0.DiagCode)) AND fb_0.SafetyDemand) AND NOT (fb_0.ResetRequest)) AND NOT (fb_0.Error)));
	testState_0 := testState_0 + 1;
38:
	fb_0.Activate := TRUE; fb_0.S_OutControl := FALSE; fb_0.EDM1 := TRUE; fb_0.EDM2 := FALSE; fb_0.ValveType := TRUE; fb_0.S_StartReset := TRUE; fb_0.Reset := FALSE;
	fb_0();
	failed_0 := NOT ((((((((((((NOT (fb_0.Reset_Before) AND NOT (fb_0.S_OutControl_Before)) AND fb_0.T_Init.Q) AND NOT (fb_0.T_Monitoring.Q)) AND (fb_0.DiagCode = 34818)) AND fb_0.Ready) AND NOT (fb_0.S_SafeState)) AND NOT (fb_0.S_ValveOut)) AND (fb_0.S_ValveStatus = fb_0.DiagCode)) AND fb_0.SafetyDemand) AND NOT (fb_0.ResetRequest)) AND NOT (fb_0.Error)));
	testState_0 := testState_0 + 1;
39:
	IF (fb_0.T_Monitoring.Q AND (fb_0.DiagCode = 50256)) THEN
		waitCounter_0 := 0;
		testState_0 := testState_0 + 1;
	ELSE
		failed_0 := NOT ((NOT (fb_0.Reset_Before) AND (NOT (fb_0.S_OutControl_Before) AND (fb_0.T_Init.Q AND (NOT (fb_0.T_Monitoring.Q) AND ((fb_0.DiagCode = 34818) AND (fb_0.Ready AND (NOT (fb_0.S_SafeState) AND (NOT (fb_0.S_ValveOut) AND ((fb_0.S_ValveStatus = fb_0.DiagCode) AND (fb_0.SafetyDemand AND (NOT (fb_0.ResetRequest) AND NOT (fb_0.Error)))))))))))));
		IF waitCounter_0 > 100 THEN
			finished_0 := TRUE;
		ELSE
			waitCounter_0 := waitCounter_0 + 1;
			fb_0();
		END_IF
	END_IF
40:
	failed_0 := NOT ((((((((((((NOT (fb_0.Reset_Before) AND NOT (fb_0.S_OutControl_Before)) AND fb_0.T_Init.Q) AND fb_0.T_Monitoring.Q) AND (fb_0.DiagCode = 50256)) AND fb_0.Ready) AND NOT (fb_0.S_SafeState)) AND NOT (fb_0.S_ValveOut)) AND (fb_0.S_ValveStatus = fb_0.DiagCode)) AND NOT (fb_0.SafetyDemand)) AND fb_0.ResetRequest) AND fb_0.Error));
	testState_0 := testState_0 + 1;
41:
	fb_0.Activate := TRUE; fb_0.S_OutControl := TRUE; fb_0.EDM1 := TRUE; fb_0.EDM2 := FALSE; fb_0.ValveType := TRUE; fb_0.S_StartReset := TRUE; fb_0.Reset := FALSE;
	fb_0();
	failed_0 := NOT ((((((((((((NOT (fb_0.Reset_Before) AND fb_0.S_OutControl_Before) AND fb_0.T_Init.Q) AND fb_0.T_Monitoring.Q) AND (fb_0.DiagCode = 49232)) AND fb_0.Ready) AND NOT (fb_0.S_SafeState)) AND NOT (fb_0.S_ValveOut)) AND (fb_0.S_ValveStatus = fb_0.DiagCode)) AND NOT (fb_0.SafetyDemand)) AND NOT (fb_0.ResetRequest)) AND fb_0.Error));
	testState_0 := testState_0 + 1;
42:
	fb_0.Activate := TRUE; fb_0.S_OutControl := TRUE; fb_0.EDM1 := TRUE; fb_0.EDM2 := FALSE; fb_0.ValveType := TRUE; fb_0.S_StartReset := TRUE; fb_0.Reset := TRUE;
	fb_0();
	failed_0 := NOT ((((((((((((fb_0.Reset_Before AND fb_0.S_OutControl_Before) AND fb_0.T_Init.Q) AND fb_0.T_Monitoring.Q) AND (fb_0.DiagCode = 49232)) AND fb_0.Ready) AND NOT (fb_0.S_SafeState)) AND NOT (fb_0.S_ValveOut)) AND (fb_0.S_ValveStatus = fb_0.DiagCode)) AND NOT (fb_0.SafetyDemand)) AND NOT (fb_0.ResetRequest)) AND fb_0.Error));
	testState_0 := testState_0 + 1;
43:
	fb_0.Activate := TRUE; fb_0.S_OutControl := TRUE; fb_0.EDM1 := TRUE; fb_0.EDM2 := FALSE; fb_0.ValveType := TRUE; fb_0.S_StartReset := TRUE; fb_0.Reset := TRUE;
	fb_0();
	failed_0 := NOT ((((((((((((fb_0.Reset_Before AND fb_0.S_OutControl_Before) AND fb_0.T_Init.Q) AND fb_0.T_Monitoring.Q) AND (fb_0.DiagCode = 49233)) AND fb_0.Ready) AND NOT (fb_0.S_SafeState)) AND NOT (fb_0.S_ValveOut)) AND (fb_0.S_ValveStatus = fb_0.DiagCode)) AND NOT (fb_0.SafetyDemand)) AND NOT (fb_0.ResetRequest)) AND fb_0.Error));
	testState_0 := testState_0 + 1;
44:
	fb_0.Activate := TRUE; fb_0.S_OutControl := TRUE; fb_0.EDM1 := TRUE; fb_0.EDM2 := FALSE; fb_0.ValveType := TRUE; fb_0.S_StartReset := TRUE; fb_0.Reset := TRUE;
	fb_0();
	failed_0 := NOT ((((((((((((fb_0.Reset_Before AND fb_0.S_OutControl_Before) AND fb_0.T_Init.Q) AND fb_0.T_Monitoring.Q) AND (fb_0.DiagCode = 49233)) AND fb_0.Ready) AND NOT (fb_0.S_SafeState)) AND NOT (fb_0.S_ValveOut)) AND (fb_0.S_ValveStatus = fb_0.DiagCode)) AND NOT (fb_0.SafetyDemand)) AND NOT (fb_0.ResetRequest)) AND fb_0.Error));
	testState_0 := testState_0 + 1;
45:
	fb_0.Activate := TRUE; fb_0.S_OutControl := TRUE; fb_0.EDM1 := TRUE; fb_0.EDM2 := FALSE; fb_0.ValveType := TRUE; fb_0.S_StartReset := TRUE; fb_0.Reset := FALSE;
	fb_0();
	failed_0 := NOT ((((((((((((NOT (fb_0.Reset_Before) AND fb_0.S_OutControl_Before) AND fb_0.T_Init.Q) AND fb_0.T_Monitoring.Q) AND (fb_0.DiagCode = 49232)) AND fb_0.Ready) AND NOT (fb_0.S_SafeState)) AND NOT (fb_0.S_ValveOut)) AND (fb_0.S_ValveStatus = fb_0.DiagCode)) AND NOT (fb_0.SafetyDemand)) AND NOT (fb_0.ResetRequest)) AND fb_0.Error));
	testState_0 := testState_0 + 1;
46:
	fb_0.Activate := TRUE; fb_0.S_OutControl := FALSE; fb_0.EDM1 := TRUE; fb_0.EDM2 := FALSE; fb_0.ValveType := TRUE; fb_0.S_StartReset := TRUE; fb_0.Reset := FALSE;
	fb_0();
	failed_0 := NOT ((((((((((((NOT (fb_0.Reset_Before) AND NOT (fb_0.S_OutControl_Before)) AND fb_0.T_Init.Q) AND fb_0.T_Monitoring.Q) AND (fb_0.DiagCode = 50256)) AND fb_0.Ready) AND NOT (fb_0.S_SafeState)) AND NOT (fb_0.S_ValveOut)) AND (fb_0.S_ValveStatus = fb_0.DiagCode)) AND NOT (fb_0.SafetyDemand)) AND fb_0.ResetRequest) AND fb_0.Error));
	testState_0 := testState_0 + 1;
47:
	fb_0.Activate := TRUE; fb_0.S_OutControl := TRUE; fb_0.EDM1 := TRUE; fb_0.EDM2 := FALSE; fb_0.ValveType := TRUE; fb_0.S_StartReset := TRUE; fb_0.Reset := FALSE;
	fb_0();
	failed_0 := NOT ((((((((((((NOT (fb_0.Reset_Before) AND fb_0.S_OutControl_Before) AND fb_0.T_Init.Q) AND fb_0.T_Monitoring.Q) AND (fb_0.DiagCode = 49232)) AND fb_0.Ready) AND NOT (fb_0.S_SafeState)) AND NOT (fb_0.S_ValveOut)) AND (fb_0.S_ValveStatus = fb_0.DiagCode)) AND NOT (fb_0.SafetyDemand)) AND NOT (fb_0.ResetRequest)) AND fb_0.Error));
	testState_0 := testState_0 + 1;
48:
	fb_0.Activate := TRUE; fb_0.S_OutControl := FALSE; fb_0.EDM1 := TRUE; fb_0.EDM2 := TRUE; fb_0.ValveType := TRUE; fb_0.S_StartReset := TRUE; fb_0.Reset := TRUE;
	fb_0();
	failed_0 := NOT ((((((((((((fb_0.Reset_Before AND NOT (fb_0.S_OutControl_Before)) AND fb_0.T_Init.Q) AND NOT (fb_0.T_Monitoring.Q)) AND (fb_0.DiagCode = 34818)) AND fb_0.Ready) AND NOT (fb_0.S_SafeState)) AND NOT (fb_0.S_ValveOut)) AND (fb_0.S_ValveStatus = fb_0.DiagCode)) AND fb_0.SafetyDemand) AND NOT (fb_0.ResetRequest)) AND NOT (fb_0.Error)));
	testState_0 := testState_0 + 1;
49:
	fb_0.Activate := TRUE; fb_0.S_OutControl := FALSE; fb_0.EDM1 := TRUE; fb_0.EDM2 := FALSE; fb_0.ValveType := TRUE; fb_0.S_StartReset := TRUE; fb_0.Reset := FALSE;
	fb_0();
	failed_0 := NOT ((((((((((((NOT (fb_0.Reset_Before) AND NOT (fb_0.S_OutControl_Before)) AND fb_0.T_Init.Q) AND NOT (fb_0.T_Monitoring.Q)) AND (fb_0.DiagCode = 34818)) AND fb_0.Ready) AND NOT (fb_0.S_SafeState)) AND NOT (fb_0.S_ValveOut)) AND (fb_0.S_ValveStatus = fb_0.DiagCode)) AND fb_0.SafetyDemand) AND NOT (fb_0.ResetRequest)) AND NOT (fb_0.Error)));
	testState_0 := testState_0 + 1;
50:
	IF (fb_0.T_Monitoring.Q AND (fb_0.DiagCode = 50256)) THEN
		waitCounter_0 := 0;
		testState_0 := testState_0 + 1;
	ELSE
		failed_0 := NOT ((NOT (fb_0.Reset_Before) AND (NOT (fb_0.S_OutControl_Before) AND (fb_0.T_Init.Q AND (NOT (fb_0.T_Monitoring.Q) AND ((fb_0.DiagCode = 34818) AND (fb_0.Ready AND (NOT (fb_0.S_SafeState) AND (NOT (fb_0.S_ValveOut) AND ((fb_0.S_ValveStatus = fb_0.DiagCode) AND (fb_0.SafetyDemand AND (NOT (fb_0.ResetRequest) AND NOT (fb_0.Error)))))))))))));
		IF waitCounter_0 > 100 THEN
			finished_0 := TRUE;
		ELSE
			waitCounter_0 := waitCounter_0 + 1;
			fb_0();
		END_IF
	END_IF
51:
	failed_0 := NOT ((((((((((((NOT (fb_0.Reset_Before) AND NOT (fb_0.S_OutControl_Before)) AND fb_0.T_Init.Q) AND fb_0.T_Monitoring.Q) AND (fb_0.DiagCode = 50256)) AND fb_0.Ready) AND NOT (fb_0.S_SafeState)) AND NOT (fb_0.S_ValveOut)) AND (fb_0.S_ValveStatus = fb_0.DiagCode)) AND NOT (fb_0.SafetyDemand)) AND fb_0.ResetRequest) AND fb_0.Error));
	testState_0 := testState_0 + 1;
52:
	fb_0.Activate := TRUE; fb_0.S_OutControl := FALSE; fb_0.EDM1 := TRUE; fb_0.EDM2 := FALSE; fb_0.ValveType := TRUE; fb_0.S_StartReset := TRUE; fb_0.Reset := TRUE;
	fb_0();
	failed_0 := NOT ((((((((((((fb_0.Reset_Before AND NOT (fb_0.S_OutControl_Before)) AND fb_0.T_Init.Q) AND fb_0.T_Monitoring.Q) AND (fb_0.DiagCode = 50256)) AND fb_0.Ready) AND NOT (fb_0.S_SafeState)) AND NOT (fb_0.S_ValveOut)) AND (fb_0.S_ValveStatus = fb_0.DiagCode)) AND NOT (fb_0.SafetyDemand)) AND fb_0.ResetRequest) AND fb_0.Error));
	testState_0 := testState_0 + 1;
53:
	fb_0.Activate := TRUE; fb_0.S_OutControl := FALSE; fb_0.EDM1 := TRUE; fb_0.EDM2 := FALSE; fb_0.ValveType := TRUE; fb_0.S_StartReset := TRUE; fb_0.Reset := TRUE;
	fb_0();
	failed_0 := NOT ((((((((((((fb_0.Reset_Before AND NOT (fb_0.S_OutControl_Before)) AND fb_0.T_Init.Q) AND fb_0.T_Monitoring.Q) AND (fb_0.DiagCode = 49233)) AND fb_0.Ready) AND NOT (fb_0.S_SafeState)) AND NOT (fb_0.S_ValveOut)) AND (fb_0.S_ValveStatus = fb_0.DiagCode)) AND NOT (fb_0.SafetyDemand)) AND NOT (fb_0.ResetRequest)) AND fb_0.Error));
	testState_0 := testState_0 + 1;
54:
	fb_0.Activate := TRUE; fb_0.S_OutControl := FALSE; fb_0.EDM1 := TRUE; fb_0.EDM2 := FALSE; fb_0.ValveType := TRUE; fb_0.S_StartReset := TRUE; fb_0.Reset := FALSE;
	fb_0();
	failed_0 := NOT ((((((((((((NOT (fb_0.Reset_Before) AND NOT (fb_0.S_OutControl_Before)) AND fb_0.T_Init.Q) AND fb_0.T_Monitoring.Q) AND (fb_0.DiagCode = 50256)) AND fb_0.Ready) AND NOT (fb_0.S_SafeState)) AND NOT (fb_0.S_ValveOut)) AND (fb_0.S_ValveStatus = fb_0.DiagCode)) AND NOT (fb_0.SafetyDemand)) AND fb_0.ResetRequest) AND fb_0.Error));
	testState_0 := testState_0 + 1;
55:
	fb_0.Activate := TRUE; fb_0.S_OutControl := FALSE; fb_0.EDM1 := TRUE; fb_0.EDM2 := TRUE; fb_0.ValveType := TRUE; fb_0.S_StartReset := TRUE; fb_0.Reset := TRUE;
	fb_0();
	failed_0 := NOT ((((((((((((fb_0.Reset_Before AND NOT (fb_0.S_OutControl_Before)) AND fb_0.T_Init.Q) AND NOT (fb_0.T_Monitoring.Q)) AND (fb_0.DiagCode = 34818)) AND fb_0.Ready) AND NOT (fb_0.S_SafeState)) AND NOT (fb_0.S_ValveOut)) AND (fb_0.S_ValveStatus = fb_0.DiagCode)) AND fb_0.SafetyDemand) AND NOT (fb_0.ResetRequest)) AND NOT (fb_0.Error)));
	testState_0 := testState_0 + 1;
56:
	fb_0.Activate := TRUE; fb_0.S_OutControl := FALSE; fb_0.EDM1 := FALSE; fb_0.EDM2 := FALSE; fb_0.ValveType := TRUE; fb_0.S_StartReset := TRUE; fb_0.Reset := FALSE;
	fb_0();
	failed_0 := NOT ((((((((((((NOT (fb_0.Reset_Before) AND NOT (fb_0.S_OutControl_Before)) AND fb_0.T_Init.Q) AND NOT (fb_0.T_Monitoring.Q)) AND (fb_0.DiagCode = 34818)) AND fb_0.Ready) AND NOT (fb_0.S_SafeState)) AND NOT (fb_0.S_ValveOut)) AND (fb_0.S_ValveStatus = fb_0.DiagCode)) AND fb_0.SafetyDemand) AND NOT (fb_0.ResetRequest)) AND NOT (fb_0.Error)));
	testState_0 := testState_0 + 1;
57:
	IF (fb_0.T_Monitoring.Q AND (fb_0.DiagCode = 50272)) THEN
		waitCounter_0 := 0;
		testState_0 := testState_0 + 1;
	ELSE
		failed_0 := NOT ((NOT (fb_0.Reset_Before) AND (NOT (fb_0.S_OutControl_Before) AND (fb_0.T_Init.Q AND (NOT (fb_0.T_Monitoring.Q) AND ((fb_0.DiagCode = 34818) AND (fb_0.Ready AND (NOT (fb_0.S_SafeState) AND (NOT (fb_0.S_ValveOut) AND ((fb_0.S_ValveStatus = fb_0.DiagCode) AND (fb_0.SafetyDemand AND (NOT (fb_0.ResetRequest) AND NOT (fb_0.Error)))))))))))));
		IF waitCounter_0 > 100 THEN
			finished_0 := TRUE;
		ELSE
			waitCounter_0 := waitCounter_0 + 1;
			fb_0();
		END_IF
	END_IF
58:
	failed_0 := NOT ((((((((((((NOT (fb_0.Reset_Before) AND NOT (fb_0.S_OutControl_Before)) AND fb_0.T_Init.Q) AND fb_0.T_Monitoring.Q) AND (fb_0.DiagCode = 50272)) AND fb_0.Ready) AND NOT (fb_0.S_SafeState)) AND NOT (fb_0.S_ValveOut)) AND (fb_0.S_ValveStatus = fb_0.DiagCode)) AND NOT (fb_0.SafetyDemand)) AND fb_0.ResetRequest) AND fb_0.Error));
	testState_0 := testState_0 + 1;
59:
	fb_0.Activate := TRUE; fb_0.S_OutControl := TRUE; fb_0.EDM1 := FALSE; fb_0.EDM2 := FALSE; fb_0.ValveType := TRUE; fb_0.S_StartReset := TRUE; fb_0.Reset := FALSE;
	fb_0();
	failed_0 := NOT ((((((((((((NOT (fb_0.Reset_Before) AND fb_0.S_OutControl_Before) AND fb_0.T_Init.Q) AND fb_0.T_Monitoring.Q) AND (fb_0.DiagCode = 49248)) AND fb_0.Ready) AND NOT (fb_0.S_SafeState)) AND NOT (fb_0.S_ValveOut)) AND (fb_0.S_ValveStatus = fb_0.DiagCode)) AND NOT (fb_0.SafetyDemand)) AND NOT (fb_0.ResetRequest)) AND fb_0.Error));
	testState_0 := testState_0 + 1;
60:
	fb_0.Activate := TRUE; fb_0.S_OutControl := TRUE; fb_0.EDM1 := FALSE; fb_0.EDM2 := FALSE; fb_0.ValveType := TRUE; fb_0.S_StartReset := TRUE; fb_0.Reset := TRUE;
	fb_0();
	failed_0 := NOT ((((((((((((fb_0.Reset_Before AND fb_0.S_OutControl_Before) AND fb_0.T_Init.Q) AND fb_0.T_Monitoring.Q) AND (fb_0.DiagCode = 49248)) AND fb_0.Ready) AND NOT (fb_0.S_SafeState)) AND NOT (fb_0.S_ValveOut)) AND (fb_0.S_ValveStatus = fb_0.DiagCode)) AND NOT (fb_0.SafetyDemand)) AND NOT (fb_0.ResetRequest)) AND fb_0.Error));
	testState_0 := testState_0 + 1;
61:
	fb_0.Activate := TRUE; fb_0.S_OutControl := TRUE; fb_0.EDM1 := FALSE; fb_0.EDM2 := FALSE; fb_0.ValveType := TRUE; fb_0.S_StartReset := TRUE; fb_0.Reset := TRUE;
	fb_0();
	failed_0 := NOT ((((((((((((fb_0.Reset_Before AND fb_0.S_OutControl_Before) AND fb_0.T_Init.Q) AND fb_0.T_Monitoring.Q) AND (fb_0.DiagCode = 49249)) AND fb_0.Ready) AND NOT (fb_0.S_SafeState)) AND NOT (fb_0.S_ValveOut)) AND (fb_0.S_ValveStatus = fb_0.DiagCode)) AND NOT (fb_0.SafetyDemand)) AND NOT (fb_0.ResetRequest)) AND fb_0.Error));
	testState_0 := testState_0 + 1;
62:
	fb_0.Activate := TRUE; fb_0.S_OutControl := TRUE; fb_0.EDM1 := FALSE; fb_0.EDM2 := FALSE; fb_0.ValveType := TRUE; fb_0.S_StartReset := TRUE; fb_0.Reset := TRUE;
	fb_0();
	failed_0 := NOT ((((((((((((fb_0.Reset_Before AND fb_0.S_OutControl_Before) AND fb_0.T_Init.Q) AND fb_0.T_Monitoring.Q) AND (fb_0.DiagCode = 49249)) AND fb_0.Ready) AND NOT (fb_0.S_SafeState)) AND NOT (fb_0.S_ValveOut)) AND (fb_0.S_ValveStatus = fb_0.DiagCode)) AND NOT (fb_0.SafetyDemand)) AND NOT (fb_0.ResetRequest)) AND fb_0.Error));
	testState_0 := testState_0 + 1;
63:
	fb_0.Activate := TRUE; fb_0.S_OutControl := TRUE; fb_0.EDM1 := FALSE; fb_0.EDM2 := FALSE; fb_0.ValveType := TRUE; fb_0.S_StartReset := TRUE; fb_0.Reset := FALSE;
	fb_0();
	failed_0 := NOT ((((((((((((NOT (fb_0.Reset_Before) AND fb_0.S_OutControl_Before) AND fb_0.T_Init.Q) AND fb_0.T_Monitoring.Q) AND (fb_0.DiagCode = 49248)) AND fb_0.Ready) AND NOT (fb_0.S_SafeState)) AND NOT (fb_0.S_ValveOut)) AND (fb_0.S_ValveStatus = fb_0.DiagCode)) AND NOT (fb_0.SafetyDemand)) AND NOT (fb_0.ResetRequest)) AND fb_0.Error));
	testState_0 := testState_0 + 1;
64:
	fb_0.Activate := TRUE; fb_0.S_OutControl := FALSE; fb_0.EDM1 := FALSE; fb_0.EDM2 := FALSE; fb_0.ValveType := TRUE; fb_0.S_StartReset := TRUE; fb_0.Reset := FALSE;
	fb_0();
	failed_0 := NOT ((((((((((((NOT (fb_0.Reset_Before) AND NOT (fb_0.S_OutControl_Before)) AND fb_0.T_Init.Q) AND fb_0.T_Monitoring.Q) AND (fb_0.DiagCode = 50272)) AND fb_0.Ready) AND NOT (fb_0.S_SafeState)) AND NOT (fb_0.S_ValveOut)) AND (fb_0.S_ValveStatus = fb_0.DiagCode)) AND NOT (fb_0.SafetyDemand)) AND fb_0.ResetRequest) AND fb_0.Error));
	testState_0 := testState_0 + 1;
65:
	fb_0.Activate := TRUE; fb_0.S_OutControl := TRUE; fb_0.EDM1 := FALSE; fb_0.EDM2 := FALSE; fb_0.ValveType := TRUE; fb_0.S_StartReset := TRUE; fb_0.Reset := FALSE;
	fb_0();
	failed_0 := NOT ((((((((((((NOT (fb_0.Reset_Before) AND fb_0.S_OutControl_Before) AND fb_0.T_Init.Q) AND fb_0.T_Monitoring.Q) AND (fb_0.DiagCode = 49248)) AND fb_0.Ready) AND NOT (fb_0.S_SafeState)) AND NOT (fb_0.S_ValveOut)) AND (fb_0.S_ValveStatus = fb_0.DiagCode)) AND NOT (fb_0.SafetyDemand)) AND NOT (fb_0.ResetRequest)) AND fb_0.Error));
	testState_0 := testState_0 + 1;
66:
	fb_0.Activate := TRUE; fb_0.S_OutControl := FALSE; fb_0.EDM1 := TRUE; fb_0.EDM2 := TRUE; fb_0.ValveType := TRUE; fb_0.S_StartReset := TRUE; fb_0.Reset := TRUE;
	fb_0();
	failed_0 := NOT ((((((((((((fb_0.Reset_Before AND NOT (fb_0.S_OutControl_Before)) AND fb_0.T_Init.Q) AND NOT (fb_0.T_Monitoring.Q)) AND (fb_0.DiagCode = 34818)) AND fb_0.Ready) AND NOT (fb_0.S_SafeState)) AND NOT (fb_0.S_ValveOut)) AND (fb_0.S_ValveStatus = fb_0.DiagCode)) AND fb_0.SafetyDemand) AND NOT (fb_0.ResetRequest)) AND NOT (fb_0.Error)));
	testState_0 := testState_0 + 1;
67:
	fb_0.Activate := TRUE; fb_0.S_OutControl := FALSE; fb_0.EDM1 := FALSE; fb_0.EDM2 := FALSE; fb_0.ValveType := TRUE; fb_0.S_StartReset := TRUE; fb_0.Reset := FALSE;
	fb_0();
	failed_0 := NOT ((((((((((((NOT (fb_0.Reset_Before) AND NOT (fb_0.S_OutControl_Before)) AND fb_0.T_Init.Q) AND NOT (fb_0.T_Monitoring.Q)) AND (fb_0.DiagCode = 34818)) AND fb_0.Ready) AND NOT (fb_0.S_SafeState)) AND NOT (fb_0.S_ValveOut)) AND (fb_0.S_ValveStatus = fb_0.DiagCode)) AND fb_0.SafetyDemand) AND NOT (fb_0.ResetRequest)) AND NOT (fb_0.Error)));
	testState_0 := testState_0 + 1;
68:
	IF (fb_0.T_Monitoring.Q AND (fb_0.DiagCode = 50272)) THEN
		waitCounter_0 := 0;
		testState_0 := testState_0 + 1;
	ELSE
		failed_0 := NOT ((NOT (fb_0.Reset_Before) AND (NOT (fb_0.S_OutControl_Before) AND (fb_0.T_Init.Q AND (NOT (fb_0.T_Monitoring.Q) AND ((fb_0.DiagCode = 34818) AND (fb_0.Ready AND (NOT (fb_0.S_SafeState) AND (NOT (fb_0.S_ValveOut) AND ((fb_0.S_ValveStatus = fb_0.DiagCode) AND (fb_0.SafetyDemand AND (NOT (fb_0.ResetRequest) AND NOT (fb_0.Error)))))))))))));
		IF waitCounter_0 > 100 THEN
			finished_0 := TRUE;
		ELSE
			waitCounter_0 := waitCounter_0 + 1;
			fb_0();
		END_IF
	END_IF
69:
	failed_0 := NOT ((((((((((((NOT (fb_0.Reset_Before) AND NOT (fb_0.S_OutControl_Before)) AND fb_0.T_Init.Q) AND fb_0.T_Monitoring.Q) AND (fb_0.DiagCode = 50272)) AND fb_0.Ready) AND NOT (fb_0.S_SafeState)) AND NOT (fb_0.S_ValveOut)) AND (fb_0.S_ValveStatus = fb_0.DiagCode)) AND NOT (fb_0.SafetyDemand)) AND fb_0.ResetRequest) AND fb_0.Error));
	testState_0 := testState_0 + 1;
70:
	fb_0.Activate := TRUE; fb_0.S_OutControl := FALSE; fb_0.EDM1 := FALSE; fb_0.EDM2 := FALSE; fb_0.ValveType := TRUE; fb_0.S_StartReset := TRUE; fb_0.Reset := TRUE;
	fb_0();
	failed_0 := NOT ((((((((((((fb_0.Reset_Before AND NOT (fb_0.S_OutControl_Before)) AND fb_0.T_Init.Q) AND fb_0.T_Monitoring.Q) AND (fb_0.DiagCode = 50272)) AND fb_0.Ready) AND NOT (fb_0.S_SafeState)) AND NOT (fb_0.S_ValveOut)) AND (fb_0.S_ValveStatus = fb_0.DiagCode)) AND NOT (fb_0.SafetyDemand)) AND fb_0.ResetRequest) AND fb_0.Error));
	testState_0 := testState_0 + 1;
71:
	fb_0.Activate := TRUE; fb_0.S_OutControl := FALSE; fb_0.EDM1 := FALSE; fb_0.EDM2 := FALSE; fb_0.ValveType := TRUE; fb_0.S_StartReset := TRUE; fb_0.Reset := TRUE;
	fb_0();
	failed_0 := NOT ((((((((((((fb_0.Reset_Before AND NOT (fb_0.S_OutControl_Before)) AND fb_0.T_Init.Q) AND fb_0.T_Monitoring.Q) AND (fb_0.DiagCode = 49249)) AND fb_0.Ready) AND NOT (fb_0.S_SafeState)) AND NOT (fb_0.S_ValveOut)) AND (fb_0.S_ValveStatus = fb_0.DiagCode)) AND NOT (fb_0.SafetyDemand)) AND NOT (fb_0.ResetRequest)) AND fb_0.Error));
	testState_0 := testState_0 + 1;
72:
	fb_0.Activate := TRUE; fb_0.S_OutControl := FALSE; fb_0.EDM1 := FALSE; fb_0.EDM2 := FALSE; fb_0.ValveType := TRUE; fb_0.S_StartReset := TRUE; fb_0.Reset := FALSE;
	fb_0();
	failed_0 := NOT ((((((((((((NOT (fb_0.Reset_Before) AND NOT (fb_0.S_OutControl_Before)) AND fb_0.T_Init.Q) AND fb_0.T_Monitoring.Q) AND (fb_0.DiagCode = 50272)) AND fb_0.Ready) AND NOT (fb_0.S_SafeState)) AND NOT (fb_0.S_ValveOut)) AND (fb_0.S_ValveStatus = fb_0.DiagCode)) AND NOT (fb_0.SafetyDemand)) AND fb_0.ResetRequest) AND fb_0.Error));
	testState_0 := testState_0 + 1;
73:
	fb_0.Activate := TRUE; fb_0.S_OutControl := FALSE; fb_0.EDM1 := TRUE; fb_0.EDM2 := TRUE; fb_0.ValveType := TRUE; fb_0.S_StartReset := TRUE; fb_0.Reset := TRUE;
	fb_0();
	failed_0 := NOT ((((((((((((fb_0.Reset_Before AND NOT (fb_0.S_OutControl_Before)) AND fb_0.T_Init.Q) AND NOT (fb_0.T_Monitoring.Q)) AND (fb_0.DiagCode = 34818)) AND fb_0.Ready) AND NOT (fb_0.S_SafeState)) AND NOT (fb_0.S_ValveOut)) AND (fb_0.S_ValveStatus = fb_0.DiagCode)) AND fb_0.SafetyDemand) AND NOT (fb_0.ResetRequest)) AND NOT (fb_0.Error)));
	testState_0 := testState_0 + 1;
74:
	fb_0.Activate := TRUE; fb_0.S_OutControl := FALSE; fb_0.EDM1 := TRUE; fb_0.EDM2 := TRUE; fb_0.ValveType := TRUE; fb_0.S_StartReset := TRUE; fb_0.Reset := FALSE;
	fb_0();
	IF fb_0.T_Monitoring.Q THEN
		finished_0 := TRUE;
	ELSE
		testState_0 := testState_0 + 1;
	END_IF
75:
	failed_0 := NOT ((((((((((((NOT (fb_0.Reset_Before) AND NOT (fb_0.S_OutControl_Before)) AND fb_0.T_Init.Q) AND NOT (fb_0.T_Monitoring.Q)) AND (fb_0.DiagCode = 34820)) AND fb_0.Ready) AND fb_0.S_SafeState) AND NOT (fb_0.S_ValveOut)) AND (fb_0.S_ValveStatus = fb_0.DiagCode)) AND fb_0.SafetyDemand) AND NOT (fb_0.ResetRequest)) AND NOT (fb_0.Error)));
	testState_0 := testState_0 + 1;
76:
	fb_0.Activate := TRUE; fb_0.S_OutControl := FALSE; fb_0.EDM1 := TRUE; fb_0.EDM2 := TRUE; fb_0.ValveType := TRUE; fb_0.S_StartReset := TRUE; fb_0.Reset := FALSE;
	fb_0();
	failed_0 := NOT ((((((((((((NOT (fb_0.Reset_Before) AND NOT (fb_0.S_OutControl_Before)) AND fb_0.T_Init.Q) AND NOT (fb_0.T_Monitoring.Q)) AND (fb_0.DiagCode = 34820)) AND fb_0.Ready) AND fb_0.S_SafeState) AND NOT (fb_0.S_ValveOut)) AND (fb_0.S_ValveStatus = fb_0.DiagCode)) AND fb_0.SafetyDemand) AND NOT (fb_0.ResetRequest)) AND NOT (fb_0.Error)));
	testState_0 := testState_0 + 1;
77:
	fb_0.Activate := TRUE; fb_0.S_OutControl := FALSE; fb_0.EDM1 := FALSE; fb_0.EDM2 := TRUE; fb_0.ValveType := TRUE; fb_0.S_StartReset := TRUE; fb_0.Reset := FALSE;
	fb_0();
	failed_0 := NOT ((((((((((((NOT (fb_0.Reset_Before) AND NOT (fb_0.S_OutControl_Before)) AND fb_0.T_Init.Q) AND NOT (fb_0.T_Monitoring.Q)) AND (fb_0.DiagCode = 50240)) AND fb_0.Ready) AND NOT (fb_0.S_SafeState)) AND NOT (fb_0.S_ValveOut)) AND (fb_0.S_ValveStatus = fb_0.DiagCode)) AND NOT (fb_0.SafetyDemand)) AND fb_0.ResetRequest) AND fb_0.Error));
	testState_0 := testState_0 + 1;
78:
	fb_0.Activate := TRUE; fb_0.S_OutControl := FALSE; fb_0.EDM1 := TRUE; fb_0.EDM2 := TRUE; fb_0.ValveType := TRUE; fb_0.S_StartReset := TRUE; fb_0.Reset := TRUE;
	fb_0();
	failed_0 := NOT ((((((((((((fb_0.Reset_Before AND NOT (fb_0.S_OutControl_Before)) AND fb_0.T_Init.Q) AND NOT (fb_0.T_Monitoring.Q)) AND (fb_0.DiagCode = 34818)) AND fb_0.Ready) AND NOT (fb_0.S_SafeState)) AND NOT (fb_0.S_ValveOut)) AND (fb_0.S_ValveStatus = fb_0.DiagCode)) AND fb_0.SafetyDemand) AND NOT (fb_0.ResetRequest)) AND NOT (fb_0.Error)));
	testState_0 := testState_0 + 1;
79:
	fb_0.Activate := TRUE; fb_0.S_OutControl := FALSE; fb_0.EDM1 := TRUE; fb_0.EDM2 := TRUE; fb_0.ValveType := TRUE; fb_0.S_StartReset := TRUE; fb_0.Reset := FALSE;
	fb_0();
	IF fb_0.T_Monitoring.Q THEN
		finished_0 := TRUE;
	ELSE
		testState_0 := testState_0 + 1;
	END_IF
80:
	failed_0 := NOT ((((((((((((NOT (fb_0.Reset_Before) AND NOT (fb_0.S_OutControl_Before)) AND fb_0.T_Init.Q) AND NOT (fb_0.T_Monitoring.Q)) AND (fb_0.DiagCode = 34820)) AND fb_0.Ready) AND fb_0.S_SafeState) AND NOT (fb_0.S_ValveOut)) AND (fb_0.S_ValveStatus = fb_0.DiagCode)) AND fb_0.SafetyDemand) AND NOT (fb_0.ResetRequest)) AND NOT (fb_0.Error)));
	testState_0 := testState_0 + 1;
81:
	fb_0.Activate := TRUE; fb_0.S_OutControl := FALSE; fb_0.EDM1 := TRUE; fb_0.EDM2 := FALSE; fb_0.ValveType := TRUE; fb_0.S_StartReset := TRUE; fb_0.Reset := FALSE;
	fb_0();
	failed_0 := NOT ((((((((((((NOT (fb_0.Reset_Before) AND NOT (fb_0.S_OutControl_Before)) AND fb_0.T_Init.Q) AND NOT (fb_0.T_Monitoring.Q)) AND (fb_0.DiagCode = 50256)) AND fb_0.Ready) AND NOT (fb_0.S_SafeState)) AND NOT (fb_0.S_ValveOut)) AND (fb_0.S_ValveStatus = fb_0.DiagCode)) AND NOT (fb_0.SafetyDemand)) AND fb_0.ResetRequest) AND fb_0.Error));
	testState_0 := testState_0 + 1;
82:
	fb_0.Activate := TRUE; fb_0.S_OutControl := FALSE; fb_0.EDM1 := TRUE; fb_0.EDM2 := TRUE; fb_0.ValveType := TRUE; fb_0.S_StartReset := TRUE; fb_0.Reset := TRUE;
	fb_0();
	failed_0 := NOT ((((((((((((fb_0.Reset_Before AND NOT (fb_0.S_OutControl_Before)) AND fb_0.T_Init.Q) AND NOT (fb_0.T_Monitoring.Q)) AND (fb_0.DiagCode = 34818)) AND fb_0.Ready) AND NOT (fb_0.S_SafeState)) AND NOT (fb_0.S_ValveOut)) AND (fb_0.S_ValveStatus = fb_0.DiagCode)) AND fb_0.SafetyDemand) AND NOT (fb_0.ResetRequest)) AND NOT (fb_0.Error)));
	testState_0 := testState_0 + 1;
83:
	fb_0.Activate := TRUE; fb_0.S_OutControl := FALSE; fb_0.EDM1 := TRUE; fb_0.EDM2 := TRUE; fb_0.ValveType := TRUE; fb_0.S_StartReset := TRUE; fb_0.Reset := FALSE;
	fb_0();
	IF fb_0.T_Monitoring.Q THEN
		finished_0 := TRUE;
	ELSE
		testState_0 := testState_0 + 1;
	END_IF
84:
	failed_0 := NOT ((((((((((((NOT (fb_0.Reset_Before) AND NOT (fb_0.S_OutControl_Before)) AND fb_0.T_Init.Q) AND NOT (fb_0.T_Monitoring.Q)) AND (fb_0.DiagCode = 34820)) AND fb_0.Ready) AND fb_0.S_SafeState) AND NOT (fb_0.S_ValveOut)) AND (fb_0.S_ValveStatus = fb_0.DiagCode)) AND fb_0.SafetyDemand) AND NOT (fb_0.ResetRequest)) AND NOT (fb_0.Error)));
	testState_0 := testState_0 + 1;
85:
	fb_0.Activate := TRUE; fb_0.S_OutControl := FALSE; fb_0.EDM1 := FALSE; fb_0.EDM2 := FALSE; fb_0.ValveType := TRUE; fb_0.S_StartReset := TRUE; fb_0.Reset := FALSE;
	fb_0();
	failed_0 := NOT ((((((((((((NOT (fb_0.Reset_Before) AND NOT (fb_0.S_OutControl_Before)) AND fb_0.T_Init.Q) AND NOT (fb_0.T_Monitoring.Q)) AND (fb_0.DiagCode = 50272)) AND fb_0.Ready) AND NOT (fb_0.S_SafeState)) AND NOT (fb_0.S_ValveOut)) AND (fb_0.S_ValveStatus = fb_0.DiagCode)) AND NOT (fb_0.SafetyDemand)) AND fb_0.ResetRequest) AND fb_0.Error));
	testState_0 := testState_0 + 1;
86:
	fb_0.Activate := TRUE; fb_0.S_OutControl := FALSE; fb_0.EDM1 := TRUE; fb_0.EDM2 := TRUE; fb_0.ValveType := TRUE; fb_0.S_StartReset := TRUE; fb_0.Reset := TRUE;
	fb_0();
	failed_0 := NOT ((((((((((((fb_0.Reset_Before AND NOT (fb_0.S_OutControl_Before)) AND fb_0.T_Init.Q) AND NOT (fb_0.T_Monitoring.Q)) AND (fb_0.DiagCode = 34818)) AND fb_0.Ready) AND NOT (fb_0.S_SafeState)) AND NOT (fb_0.S_ValveOut)) AND (fb_0.S_ValveStatus = fb_0.DiagCode)) AND fb_0.SafetyDemand) AND NOT (fb_0.ResetRequest)) AND NOT (fb_0.Error)));
	testState_0 := testState_0 + 1;
87:
	fb_0.Activate := TRUE; fb_0.S_OutControl := FALSE; fb_0.EDM1 := TRUE; fb_0.EDM2 := TRUE; fb_0.ValveType := TRUE; fb_0.S_StartReset := TRUE; fb_0.Reset := FALSE;
	fb_0();
	IF fb_0.T_Monitoring.Q THEN
		finished_0 := TRUE;
	ELSE
		testState_0 := testState_0 + 1;
	END_IF
88:
	failed_0 := NOT ((((((((((((NOT (fb_0.Reset_Before) AND NOT (fb_0.S_OutControl_Before)) AND fb_0.T_Init.Q) AND NOT (fb_0.T_Monitoring.Q)) AND (fb_0.DiagCode = 34820)) AND fb_0.Ready) AND fb_0.S_SafeState) AND NOT (fb_0.S_ValveOut)) AND (fb_0.S_ValveStatus = fb_0.DiagCode)) AND fb_0.SafetyDemand) AND NOT (fb_0.ResetRequest)) AND NOT (fb_0.Error)));
	testState_0 := testState_0 + 1;
89:
	fb_0.Activate := TRUE; fb_0.S_OutControl := TRUE; fb_0.EDM1 := TRUE; fb_0.EDM2 := TRUE; fb_0.ValveType := TRUE; fb_0.S_StartReset := TRUE; fb_0.Reset := FALSE;
	fb_0();
	failed_0 := NOT ((((((((((((NOT (fb_0.Reset_Before) AND fb_0.S_OutControl_Before) AND fb_0.T_Init.Q) AND NOT (fb_0.T_Monitoring.Q)) AND (fb_0.DiagCode = 32800)) AND fb_0.Ready) AND NOT (fb_0.S_SafeState)) AND fb_0.S_ValveOut) AND (fb_0.S_ValveStatus = fb_0.DiagCode)) AND NOT (fb_0.SafetyDemand)) AND NOT (fb_0.ResetRequest)) AND NOT (fb_0.Error)));
	testState_0 := testState_0 + 1;
90:
	fb_0.Activate := TRUE; fb_0.S_OutControl := FALSE; fb_0.EDM1 := TRUE; fb_0.EDM2 := TRUE; fb_0.ValveType := TRUE; fb_0.S_StartReset := TRUE; fb_0.Reset := FALSE;
	fb_0();
	IF fb_0.T_Monitoring.Q THEN
		finished_0 := TRUE;
	ELSE
		testState_0 := testState_0 + 1;
	END_IF
91:
	failed_0 := NOT ((((((((((((NOT (fb_0.Reset_Before) AND NOT (fb_0.S_OutControl_Before)) AND fb_0.T_Init.Q) AND NOT (fb_0.T_Monitoring.Q)) AND (fb_0.DiagCode = 34818)) AND fb_0.Ready) AND NOT (fb_0.S_SafeState)) AND NOT (fb_0.S_ValveOut)) AND (fb_0.S_ValveStatus = fb_0.DiagCode)) AND fb_0.SafetyDemand) AND NOT (fb_0.ResetRequest)) AND NOT (fb_0.Error)));
	testState_0 := testState_0 + 1;
92:
	fb_0.Activate := TRUE; fb_0.S_OutControl := FALSE; fb_0.EDM1 := TRUE; fb_0.EDM2 := TRUE; fb_0.ValveType := TRUE; fb_0.S_StartReset := TRUE; fb_0.Reset := FALSE;
	fb_0();
	IF fb_0.T_Monitoring.Q THEN
		finished_0 := TRUE;
	ELSE
		testState_0 := testState_0 + 1;
	END_IF
93:
	failed_0 := NOT ((((((((((((NOT (fb_0.Reset_Before) AND NOT (fb_0.S_OutControl_Before)) AND fb_0.T_Init.Q) AND NOT (fb_0.T_Monitoring.Q)) AND (fb_0.DiagCode = 34820)) AND fb_0.Ready) AND fb_0.S_SafeState) AND NOT (fb_0.S_ValveOut)) AND (fb_0.S_ValveStatus = fb_0.DiagCode)) AND fb_0.SafetyDemand) AND NOT (fb_0.ResetRequest)) AND NOT (fb_0.Error)));
	testState_0 := testState_0 + 1;
94:
	fb_0.Activate := TRUE; fb_0.S_OutControl := TRUE; fb_0.EDM1 := TRUE; fb_0.EDM2 := TRUE; fb_0.ValveType := TRUE; fb_0.S_StartReset := TRUE; fb_0.Reset := FALSE;
	fb_0();
	failed_0 := NOT ((((((((((((NOT (fb_0.Reset_Before) AND fb_0.S_OutControl_Before) AND fb_0.T_Init.Q) AND NOT (fb_0.T_Monitoring.Q)) AND (fb_0.DiagCode = 32800)) AND fb_0.Ready) AND NOT (fb_0.S_SafeState)) AND fb_0.S_ValveOut) AND (fb_0.S_ValveStatus = fb_0.DiagCode)) AND NOT (fb_0.SafetyDemand)) AND NOT (fb_0.ResetRequest)) AND NOT (fb_0.Error)));
	testState_0 := testState_0 + 1;
95:
	fb_0.Activate := TRUE; fb_0.S_OutControl := TRUE; fb_0.EDM1 := TRUE; fb_0.EDM2 := FALSE; fb_0.ValveType := TRUE; fb_0.S_StartReset := TRUE; fb_0.Reset := FALSE;
	fb_0();
	failed_0 := NOT ((((((((((((NOT (fb_0.Reset_Before) AND fb_0.S_OutControl_Before) AND fb_0.T_Init.Q) AND NOT (fb_0.T_Monitoring.Q)) AND (fb_0.DiagCode = 32800)) AND fb_0.Ready) AND NOT (fb_0.S_SafeState)) AND fb_0.S_ValveOut) AND (fb_0.S_ValveStatus = fb_0.DiagCode)) AND NOT (fb_0.SafetyDemand)) AND NOT (fb_0.ResetRequest)) AND NOT (fb_0.Error)));
	testState_0 := testState_0 + 1;
96:
	IF (fb_0.T_Monitoring.Q AND (fb_0.DiagCode = 49264)) THEN
		waitCounter_0 := 0;
		testState_0 := testState_0 + 1;
	ELSE
		failed_0 := NOT ((NOT (fb_0.Reset_Before) AND (fb_0.S_OutControl_Before AND (fb_0.T_Init.Q AND (NOT (fb_0.T_Monitoring.Q) AND ((fb_0.DiagCode = 32800) AND (fb_0.Ready AND (NOT (fb_0.S_SafeState) AND (fb_0.S_ValveOut AND ((fb_0.S_ValveStatus = fb_0.DiagCode) AND (NOT (fb_0.SafetyDemand) AND (NOT (fb_0.ResetRequest) AND NOT (fb_0.Error)))))))))))));
		IF waitCounter_0 > 100 THEN
			finished_0 := TRUE;
		ELSE
			waitCounter_0 := waitCounter_0 + 1;
			fb_0();
		END_IF
	END_IF
97:
	failed_0 := NOT ((((((((((((NOT (fb_0.Reset_Before) AND fb_0.S_OutControl_Before) AND fb_0.T_Init.Q) AND fb_0.T_Monitoring.Q) AND (fb_0.DiagCode = 49264)) AND fb_0.Ready) AND NOT (fb_0.S_SafeState)) AND NOT (fb_0.S_ValveOut)) AND (fb_0.S_ValveStatus = fb_0.DiagCode)) AND NOT (fb_0.SafetyDemand)) AND NOT (fb_0.ResetRequest)) AND fb_0.Error));
	testState_0 := testState_0 + 1;
98:
	fb_0.Activate := TRUE; fb_0.S_OutControl := TRUE; fb_0.EDM1 := TRUE; fb_0.EDM2 := FALSE; fb_0.ValveType := TRUE; fb_0.S_StartReset := TRUE; fb_0.Reset := TRUE;
	fb_0();
	failed_0 := NOT ((((((((((((fb_0.Reset_Before AND fb_0.S_OutControl_Before) AND fb_0.T_Init.Q) AND fb_0.T_Monitoring.Q) AND (fb_0.DiagCode = 49264)) AND fb_0.Ready) AND NOT (fb_0.S_SafeState)) AND NOT (fb_0.S_ValveOut)) AND (fb_0.S_ValveStatus = fb_0.DiagCode)) AND NOT (fb_0.SafetyDemand)) AND NOT (fb_0.ResetRequest)) AND fb_0.Error));
	testState_0 := testState_0 + 1;
99:
	fb_0.Activate := TRUE; fb_0.S_OutControl := TRUE; fb_0.EDM1 := TRUE; fb_0.EDM2 := FALSE; fb_0.ValveType := TRUE; fb_0.S_StartReset := TRUE; fb_0.Reset := TRUE;
	fb_0();
	failed_0 := NOT ((((((((((((fb_0.Reset_Before AND fb_0.S_OutControl_Before) AND fb_0.T_Init.Q) AND fb_0.T_Monitoring.Q) AND (fb_0.DiagCode = 49265)) AND fb_0.Ready) AND NOT (fb_0.S_SafeState)) AND NOT (fb_0.S_ValveOut)) AND (fb_0.S_ValveStatus = fb_0.DiagCode)) AND NOT (fb_0.SafetyDemand)) AND NOT (fb_0.ResetRequest)) AND fb_0.Error));
	testState_0 := testState_0 + 1;
100:
	fb_0.Activate := TRUE; fb_0.S_OutControl := TRUE; fb_0.EDM1 := TRUE; fb_0.EDM2 := FALSE; fb_0.ValveType := TRUE; fb_0.S_StartReset := TRUE; fb_0.Reset := TRUE;
	fb_0();
	failed_0 := NOT ((((((((((((fb_0.Reset_Before AND fb_0.S_OutControl_Before) AND fb_0.T_Init.Q) AND fb_0.T_Monitoring.Q) AND (fb_0.DiagCode = 49265)) AND fb_0.Ready) AND NOT (fb_0.S_SafeState)) AND NOT (fb_0.S_ValveOut)) AND (fb_0.S_ValveStatus = fb_0.DiagCode)) AND NOT (fb_0.SafetyDemand)) AND NOT (fb_0.ResetRequest)) AND fb_0.Error));
	testState_0 := testState_0 + 1;
101:
	fb_0.Activate := TRUE; fb_0.S_OutControl := TRUE; fb_0.EDM1 := TRUE; fb_0.EDM2 := FALSE; fb_0.ValveType := TRUE; fb_0.S_StartReset := TRUE; fb_0.Reset := FALSE;
	fb_0();
	failed_0 := NOT ((((((((((((NOT (fb_0.Reset_Before) AND fb_0.S_OutControl_Before) AND fb_0.T_Init.Q) AND fb_0.T_Monitoring.Q) AND (fb_0.DiagCode = 49264)) AND fb_0.Ready) AND NOT (fb_0.S_SafeState)) AND NOT (fb_0.S_ValveOut)) AND (fb_0.S_ValveStatus = fb_0.DiagCode)) AND NOT (fb_0.SafetyDemand)) AND NOT (fb_0.ResetRequest)) AND fb_0.Error));
	testState_0 := testState_0 + 1;
102:
	fb_0.Activate := TRUE; fb_0.S_OutControl := FALSE; fb_0.EDM1 := TRUE; fb_0.EDM2 := FALSE; fb_0.ValveType := TRUE; fb_0.S_StartReset := TRUE; fb_0.Reset := TRUE;
	fb_0();
	failed_0 := NOT ((((((((((((fb_0.Reset_Before AND NOT (fb_0.S_OutControl_Before)) AND fb_0.T_Init.Q) AND fb_0.T_Monitoring.Q) AND (fb_0.DiagCode = 50288)) AND fb_0.Ready) AND NOT (fb_0.S_SafeState)) AND NOT (fb_0.S_ValveOut)) AND (fb_0.S_ValveStatus = fb_0.DiagCode)) AND NOT (fb_0.SafetyDemand)) AND fb_0.ResetRequest) AND fb_0.Error));
	testState_0 := testState_0 + 1;
103:
	fb_0.Activate := TRUE; fb_0.S_OutControl := FALSE; fb_0.EDM1 := TRUE; fb_0.EDM2 := FALSE; fb_0.ValveType := TRUE; fb_0.S_StartReset := TRUE; fb_0.Reset := TRUE;
	fb_0();
	failed_0 := NOT ((((((((((((fb_0.Reset_Before AND NOT (fb_0.S_OutControl_Before)) AND fb_0.T_Init.Q) AND fb_0.T_Monitoring.Q) AND (fb_0.DiagCode = 49265)) AND fb_0.Ready) AND NOT (fb_0.S_SafeState)) AND NOT (fb_0.S_ValveOut)) AND (fb_0.S_ValveStatus = fb_0.DiagCode)) AND NOT (fb_0.SafetyDemand)) AND NOT (fb_0.ResetRequest)) AND fb_0.Error));
	testState_0 := testState_0 + 1;
104:
	fb_0.Activate := TRUE; fb_0.S_OutControl := FALSE; fb_0.EDM1 := TRUE; fb_0.EDM2 := FALSE; fb_0.ValveType := TRUE; fb_0.S_StartReset := TRUE; fb_0.Reset := FALSE;
	fb_0();
	failed_0 := NOT ((((((((((((NOT (fb_0.Reset_Before) AND NOT (fb_0.S_OutControl_Before)) AND fb_0.T_Init.Q) AND fb_0.T_Monitoring.Q) AND (fb_0.DiagCode = 50288)) AND fb_0.Ready) AND NOT (fb_0.S_SafeState)) AND NOT (fb_0.S_ValveOut)) AND (fb_0.S_ValveStatus = fb_0.DiagCode)) AND NOT (fb_0.SafetyDemand)) AND fb_0.ResetRequest) AND fb_0.Error));
	testState_0 := testState_0 + 1;
105:
	fb_0.Activate := TRUE; fb_0.S_OutControl := FALSE; fb_0.EDM1 := TRUE; fb_0.EDM2 := FALSE; fb_0.ValveType := TRUE; fb_0.S_StartReset := TRUE; fb_0.Reset := FALSE;
	fb_0();
	failed_0 := NOT ((((((((((((NOT (fb_0.Reset_Before) AND NOT (fb_0.S_OutControl_Before)) AND fb_0.T_Init.Q) AND fb_0.T_Monitoring.Q) AND (fb_0.DiagCode = 50288)) AND fb_0.Ready) AND NOT (fb_0.S_SafeState)) AND NOT (fb_0.S_ValveOut)) AND (fb_0.S_ValveStatus = fb_0.DiagCode)) AND NOT (fb_0.SafetyDemand)) AND fb_0.ResetRequest) AND fb_0.Error));
	testState_0 := testState_0 + 1;
106:
	fb_0.Activate := TRUE; fb_0.S_OutControl := TRUE; fb_0.EDM1 := TRUE; fb_0.EDM2 := FALSE; fb_0.ValveType := TRUE; fb_0.S_StartReset := TRUE; fb_0.Reset := FALSE;
	fb_0();
	failed_0 := NOT ((((((((((((NOT (fb_0.Reset_Before) AND fb_0.S_OutControl_Before) AND fb_0.T_Init.Q) AND fb_0.T_Monitoring.Q) AND (fb_0.DiagCode = 49264)) AND fb_0.Ready) AND NOT (fb_0.S_SafeState)) AND NOT (fb_0.S_ValveOut)) AND (fb_0.S_ValveStatus = fb_0.DiagCode)) AND NOT (fb_0.SafetyDemand)) AND NOT (fb_0.ResetRequest)) AND fb_0.Error));
	testState_0 := testState_0 + 1;
107:
	fb_0.Activate := TRUE; fb_0.S_OutControl := FALSE; fb_0.EDM1 := TRUE; fb_0.EDM2 := FALSE; fb_0.ValveType := TRUE; fb_0.S_StartReset := TRUE; fb_0.Reset := FALSE;
	fb_0();
	failed_0 := NOT ((((((((((((NOT (fb_0.Reset_Before) AND NOT (fb_0.S_OutControl_Before)) AND fb_0.T_Init.Q) AND fb_0.T_Monitoring.Q) AND (fb_0.DiagCode = 50288)) AND fb_0.Ready) AND NOT (fb_0.S_SafeState)) AND NOT (fb_0.S_ValveOut)) AND (fb_0.S_ValveStatus = fb_0.DiagCode)) AND NOT (fb_0.SafetyDemand)) AND fb_0.ResetRequest) AND fb_0.Error));
	testState_0 := testState_0 + 1;
108:
	fb_0.Activate := TRUE; fb_0.S_OutControl := FALSE; fb_0.EDM1 := TRUE; fb_0.EDM2 := TRUE; fb_0.ValveType := TRUE; fb_0.S_StartReset := TRUE; fb_0.Reset := TRUE;
	fb_0();
	failed_0 := NOT ((((((((((((fb_0.Reset_Before AND NOT (fb_0.S_OutControl_Before)) AND fb_0.T_Init.Q) AND NOT (fb_0.T_Monitoring.Q)) AND (fb_0.DiagCode = 34818)) AND fb_0.Ready) AND NOT (fb_0.S_SafeState)) AND NOT (fb_0.S_ValveOut)) AND (fb_0.S_ValveStatus = fb_0.DiagCode)) AND fb_0.SafetyDemand) AND NOT (fb_0.ResetRequest)) AND NOT (fb_0.Error)));
	testState_0 := testState_0 + 1;
109:
	fb_0.Activate := TRUE; fb_0.S_OutControl := FALSE; fb_0.EDM1 := TRUE; fb_0.EDM2 := TRUE; fb_0.ValveType := TRUE; fb_0.S_StartReset := TRUE; fb_0.Reset := FALSE;
	fb_0();
	IF fb_0.T_Monitoring.Q THEN
		finished_0 := TRUE;
	ELSE
		testState_0 := testState_0 + 1;
	END_IF
110:
	failed_0 := NOT ((((((((((((NOT (fb_0.Reset_Before) AND NOT (fb_0.S_OutControl_Before)) AND fb_0.T_Init.Q) AND NOT (fb_0.T_Monitoring.Q)) AND (fb_0.DiagCode = 34820)) AND fb_0.Ready) AND fb_0.S_SafeState) AND NOT (fb_0.S_ValveOut)) AND (fb_0.S_ValveStatus = fb_0.DiagCode)) AND fb_0.SafetyDemand) AND NOT (fb_0.ResetRequest)) AND NOT (fb_0.Error)));
	testState_0 := testState_0 + 1;
111:
	fb_0.Activate := TRUE; fb_0.S_OutControl := TRUE; fb_0.EDM1 := TRUE; fb_0.EDM2 := TRUE; fb_0.ValveType := TRUE; fb_0.S_StartReset := TRUE; fb_0.Reset := FALSE;
	fb_0();
	failed_0 := NOT ((((((((((((NOT (fb_0.Reset_Before) AND fb_0.S_OutControl_Before) AND fb_0.T_Init.Q) AND NOT (fb_0.T_Monitoring.Q)) AND (fb_0.DiagCode = 32800)) AND fb_0.Ready) AND NOT (fb_0.S_SafeState)) AND fb_0.S_ValveOut) AND (fb_0.S_ValveStatus = fb_0.DiagCode)) AND NOT (fb_0.SafetyDemand)) AND NOT (fb_0.ResetRequest)) AND NOT (fb_0.Error)));
	testState_0 := testState_0 + 1;
112:
	fb_0.Activate := TRUE; fb_0.S_OutControl := TRUE; fb_0.EDM1 := TRUE; fb_0.EDM2 := FALSE; fb_0.ValveType := TRUE; fb_0.S_StartReset := TRUE; fb_0.Reset := FALSE;
	fb_0();
	failed_0 := NOT ((((((((((((NOT (fb_0.Reset_Before) AND fb_0.S_OutControl_Before) AND fb_0.T_Init.Q) AND NOT (fb_0.T_Monitoring.Q)) AND (fb_0.DiagCode = 32800)) AND fb_0.Ready) AND NOT (fb_0.S_SafeState)) AND fb_0.S_ValveOut) AND (fb_0.S_ValveStatus = fb_0.DiagCode)) AND NOT (fb_0.SafetyDemand)) AND NOT (fb_0.ResetRequest)) AND NOT (fb_0.Error)));
	testState_0 := testState_0 + 1;
113:
	IF (fb_0.T_Monitoring.Q AND (fb_0.DiagCode = 49264)) THEN
		waitCounter_0 := 0;
		testState_0 := testState_0 + 1;
	ELSE
		failed_0 := NOT ((NOT (fb_0.Reset_Before) AND (fb_0.S_OutControl_Before AND (fb_0.T_Init.Q AND (NOT (fb_0.T_Monitoring.Q) AND ((fb_0.DiagCode = 32800) AND (fb_0.Ready AND (NOT (fb_0.S_SafeState) AND (fb_0.S_ValveOut AND ((fb_0.S_ValveStatus = fb_0.DiagCode) AND (NOT (fb_0.SafetyDemand) AND (NOT (fb_0.ResetRequest) AND NOT (fb_0.Error)))))))))))));
		IF waitCounter_0 > 100 THEN
			finished_0 := TRUE;
		ELSE
			waitCounter_0 := waitCounter_0 + 1;
			fb_0();
		END_IF
	END_IF
114:
	failed_0 := NOT ((((((((((((NOT (fb_0.Reset_Before) AND fb_0.S_OutControl_Before) AND fb_0.T_Init.Q) AND fb_0.T_Monitoring.Q) AND (fb_0.DiagCode = 49264)) AND fb_0.Ready) AND NOT (fb_0.S_SafeState)) AND NOT (fb_0.S_ValveOut)) AND (fb_0.S_ValveStatus = fb_0.DiagCode)) AND NOT (fb_0.SafetyDemand)) AND NOT (fb_0.ResetRequest)) AND fb_0.Error));
	testState_0 := testState_0 + 1;
115:
	fb_0.Activate := TRUE; fb_0.S_OutControl := FALSE; fb_0.EDM1 := TRUE; fb_0.EDM2 := TRUE; fb_0.ValveType := TRUE; fb_0.S_StartReset := TRUE; fb_0.Reset := TRUE;
	fb_0();
	failed_0 := NOT ((((((((((((fb_0.Reset_Before AND NOT (fb_0.S_OutControl_Before)) AND fb_0.T_Init.Q) AND NOT (fb_0.T_Monitoring.Q)) AND (fb_0.DiagCode = 34818)) AND fb_0.Ready) AND NOT (fb_0.S_SafeState)) AND NOT (fb_0.S_ValveOut)) AND (fb_0.S_ValveStatus = fb_0.DiagCode)) AND fb_0.SafetyDemand) AND NOT (fb_0.ResetRequest)) AND NOT (fb_0.Error)));
	testState_0 := testState_0 + 1;
116:
	fb_0.Activate := TRUE; fb_0.S_OutControl := FALSE; fb_0.EDM1 := TRUE; fb_0.EDM2 := TRUE; fb_0.ValveType := TRUE; fb_0.S_StartReset := TRUE; fb_0.Reset := FALSE;
	fb_0();
	IF fb_0.T_Monitoring.Q THEN
		finished_0 := TRUE;
	ELSE
		testState_0 := testState_0 + 1;
	END_IF
117:
	failed_0 := NOT ((((((((((((NOT (fb_0.Reset_Before) AND NOT (fb_0.S_OutControl_Before)) AND fb_0.T_Init.Q) AND NOT (fb_0.T_Monitoring.Q)) AND (fb_0.DiagCode = 34820)) AND fb_0.Ready) AND fb_0.S_SafeState) AND NOT (fb_0.S_ValveOut)) AND (fb_0.S_ValveStatus = fb_0.DiagCode)) AND fb_0.SafetyDemand) AND NOT (fb_0.ResetRequest)) AND NOT (fb_0.Error)));
	testState_0 := testState_0 + 1;
118:
	fb_0.Activate := TRUE; fb_0.S_OutControl := TRUE; fb_0.EDM1 := TRUE; fb_0.EDM2 := TRUE; fb_0.ValveType := TRUE; fb_0.S_StartReset := TRUE; fb_0.Reset := FALSE;
	fb_0();
	failed_0 := NOT ((((((((((((NOT (fb_0.Reset_Before) AND fb_0.S_OutControl_Before) AND fb_0.T_Init.Q) AND NOT (fb_0.T_Monitoring.Q)) AND (fb_0.DiagCode = 32800)) AND fb_0.Ready) AND NOT (fb_0.S_SafeState)) AND fb_0.S_ValveOut) AND (fb_0.S_ValveStatus = fb_0.DiagCode)) AND NOT (fb_0.SafetyDemand)) AND NOT (fb_0.ResetRequest)) AND NOT (fb_0.Error)));
	testState_0 := testState_0 + 1;
119:
	fb_0.Activate := TRUE; fb_0.S_OutControl := TRUE; fb_0.EDM1 := FALSE; fb_0.EDM2 := TRUE; fb_0.ValveType := TRUE; fb_0.S_StartReset := TRUE; fb_0.Reset := FALSE;
	fb_0();
	failed_0 := NOT ((((((((((((NOT (fb_0.Reset_Before) AND fb_0.S_OutControl_Before) AND fb_0.T_Init.Q) AND NOT (fb_0.T_Monitoring.Q)) AND (fb_0.DiagCode = 32800)) AND fb_0.Ready) AND NOT (fb_0.S_SafeState)) AND fb_0.S_ValveOut) AND (fb_0.S_ValveStatus = fb_0.DiagCode)) AND NOT (fb_0.SafetyDemand)) AND NOT (fb_0.ResetRequest)) AND NOT (fb_0.Error)));
	testState_0 := testState_0 + 1;
120:
	IF (fb_0.T_Monitoring.Q AND (fb_0.DiagCode = 49280)) THEN
		waitCounter_0 := 0;
		testState_0 := testState_0 + 1;
	ELSE
		failed_0 := NOT ((NOT (fb_0.Reset_Before) AND (fb_0.S_OutControl_Before AND (fb_0.T_Init.Q AND (NOT (fb_0.T_Monitoring.Q) AND ((fb_0.DiagCode = 32800) AND (fb_0.Ready AND (NOT (fb_0.S_SafeState) AND (fb_0.S_ValveOut AND ((fb_0.S_ValveStatus = fb_0.DiagCode) AND (NOT (fb_0.SafetyDemand) AND (NOT (fb_0.ResetRequest) AND NOT (fb_0.Error)))))))))))));
		IF waitCounter_0 > 100 THEN
			finished_0 := TRUE;
		ELSE
			waitCounter_0 := waitCounter_0 + 1;
			fb_0();
		END_IF
	END_IF
121:
	failed_0 := NOT ((((((((((((NOT (fb_0.Reset_Before) AND fb_0.S_OutControl_Before) AND fb_0.T_Init.Q) AND fb_0.T_Monitoring.Q) AND (fb_0.DiagCode = 49280)) AND fb_0.Ready) AND NOT (fb_0.S_SafeState)) AND NOT (fb_0.S_ValveOut)) AND (fb_0.S_ValveStatus = fb_0.DiagCode)) AND NOT (fb_0.SafetyDemand)) AND NOT (fb_0.ResetRequest)) AND fb_0.Error));
	testState_0 := testState_0 + 1;
122:
	fb_0.Activate := TRUE; fb_0.S_OutControl := TRUE; fb_0.EDM1 := FALSE; fb_0.EDM2 := TRUE; fb_0.ValveType := TRUE; fb_0.S_StartReset := TRUE; fb_0.Reset := TRUE;
	fb_0();
	failed_0 := NOT ((((((((((((fb_0.Reset_Before AND fb_0.S_OutControl_Before) AND fb_0.T_Init.Q) AND fb_0.T_Monitoring.Q) AND (fb_0.DiagCode = 49280)) AND fb_0.Ready) AND NOT (fb_0.S_SafeState)) AND NOT (fb_0.S_ValveOut)) AND (fb_0.S_ValveStatus = fb_0.DiagCode)) AND NOT (fb_0.SafetyDemand)) AND NOT (fb_0.ResetRequest)) AND fb_0.Error));
	testState_0 := testState_0 + 1;
123:
	fb_0.Activate := TRUE; fb_0.S_OutControl := TRUE; fb_0.EDM1 := FALSE; fb_0.EDM2 := TRUE; fb_0.ValveType := TRUE; fb_0.S_StartReset := TRUE; fb_0.Reset := TRUE;
	fb_0();
	failed_0 := NOT ((((((((((((fb_0.Reset_Before AND fb_0.S_OutControl_Before) AND fb_0.T_Init.Q) AND fb_0.T_Monitoring.Q) AND (fb_0.DiagCode = 49281)) AND fb_0.Ready) AND NOT (fb_0.S_SafeState)) AND NOT (fb_0.S_ValveOut)) AND (fb_0.S_ValveStatus = fb_0.DiagCode)) AND NOT (fb_0.SafetyDemand)) AND NOT (fb_0.ResetRequest)) AND fb_0.Error));
	testState_0 := testState_0 + 1;
124:
	fb_0.Activate := TRUE; fb_0.S_OutControl := TRUE; fb_0.EDM1 := FALSE; fb_0.EDM2 := TRUE; fb_0.ValveType := TRUE; fb_0.S_StartReset := TRUE; fb_0.Reset := TRUE;
	fb_0();
	failed_0 := NOT ((((((((((((fb_0.Reset_Before AND fb_0.S_OutControl_Before) AND fb_0.T_Init.Q) AND fb_0.T_Monitoring.Q) AND (fb_0.DiagCode = 49281)) AND fb_0.Ready) AND NOT (fb_0.S_SafeState)) AND NOT (fb_0.S_ValveOut)) AND (fb_0.S_ValveStatus = fb_0.DiagCode)) AND NOT (fb_0.SafetyDemand)) AND NOT (fb_0.ResetRequest)) AND fb_0.Error));
	testState_0 := testState_0 + 1;
125:
	fb_0.Activate := TRUE; fb_0.S_OutControl := TRUE; fb_0.EDM1 := FALSE; fb_0.EDM2 := TRUE; fb_0.ValveType := TRUE; fb_0.S_StartReset := TRUE; fb_0.Reset := FALSE;
	fb_0();
	failed_0 := NOT ((((((((((((NOT (fb_0.Reset_Before) AND fb_0.S_OutControl_Before) AND fb_0.T_Init.Q) AND fb_0.T_Monitoring.Q) AND (fb_0.DiagCode = 49280)) AND fb_0.Ready) AND NOT (fb_0.S_SafeState)) AND NOT (fb_0.S_ValveOut)) AND (fb_0.S_ValveStatus = fb_0.DiagCode)) AND NOT (fb_0.SafetyDemand)) AND NOT (fb_0.ResetRequest)) AND fb_0.Error));
	testState_0 := testState_0 + 1;
126:
	fb_0.Activate := TRUE; fb_0.S_OutControl := FALSE; fb_0.EDM1 := FALSE; fb_0.EDM2 := TRUE; fb_0.ValveType := TRUE; fb_0.S_StartReset := TRUE; fb_0.Reset := TRUE;
	fb_0();
	failed_0 := NOT ((((((((((((fb_0.Reset_Before AND NOT (fb_0.S_OutControl_Before)) AND fb_0.T_Init.Q) AND fb_0.T_Monitoring.Q) AND (fb_0.DiagCode = 50304)) AND fb_0.Ready) AND NOT (fb_0.S_SafeState)) AND NOT (fb_0.S_ValveOut)) AND (fb_0.S_ValveStatus = fb_0.DiagCode)) AND NOT (fb_0.SafetyDemand)) AND fb_0.ResetRequest) AND fb_0.Error));
	testState_0 := testState_0 + 1;
127:
	fb_0.Activate := TRUE; fb_0.S_OutControl := FALSE; fb_0.EDM1 := FALSE; fb_0.EDM2 := TRUE; fb_0.ValveType := TRUE; fb_0.S_StartReset := TRUE; fb_0.Reset := TRUE;
	fb_0();
	failed_0 := NOT ((((((((((((fb_0.Reset_Before AND NOT (fb_0.S_OutControl_Before)) AND fb_0.T_Init.Q) AND fb_0.T_Monitoring.Q) AND (fb_0.DiagCode = 49281)) AND fb_0.Ready) AND NOT (fb_0.S_SafeState)) AND NOT (fb_0.S_ValveOut)) AND (fb_0.S_ValveStatus = fb_0.DiagCode)) AND NOT (fb_0.SafetyDemand)) AND NOT (fb_0.ResetRequest)) AND fb_0.Error));
	testState_0 := testState_0 + 1;
128:
	fb_0.Activate := TRUE; fb_0.S_OutControl := FALSE; fb_0.EDM1 := FALSE; fb_0.EDM2 := TRUE; fb_0.ValveType := TRUE; fb_0.S_StartReset := TRUE; fb_0.Reset := FALSE;
	fb_0();
	failed_0 := NOT ((((((((((((NOT (fb_0.Reset_Before) AND NOT (fb_0.S_OutControl_Before)) AND fb_0.T_Init.Q) AND fb_0.T_Monitoring.Q) AND (fb_0.DiagCode = 50304)) AND fb_0.Ready) AND NOT (fb_0.S_SafeState)) AND NOT (fb_0.S_ValveOut)) AND (fb_0.S_ValveStatus = fb_0.DiagCode)) AND NOT (fb_0.SafetyDemand)) AND fb_0.ResetRequest) AND fb_0.Error));
	testState_0 := testState_0 + 1;
129:
	fb_0.Activate := TRUE; fb_0.S_OutControl := FALSE; fb_0.EDM1 := FALSE; fb_0.EDM2 := TRUE; fb_0.ValveType := TRUE; fb_0.S_StartReset := TRUE; fb_0.Reset := FALSE;
	fb_0();
	failed_0 := NOT ((((((((((((NOT (fb_0.Reset_Before) AND NOT (fb_0.S_OutControl_Before)) AND fb_0.T_Init.Q) AND fb_0.T_Monitoring.Q) AND (fb_0.DiagCode = 50304)) AND fb_0.Ready) AND NOT (fb_0.S_SafeState)) AND NOT (fb_0.S_ValveOut)) AND (fb_0.S_ValveStatus = fb_0.DiagCode)) AND NOT (fb_0.SafetyDemand)) AND fb_0.ResetRequest) AND fb_0.Error));
	testState_0 := testState_0 + 1;
130:
	fb_0.Activate := TRUE; fb_0.S_OutControl := TRUE; fb_0.EDM1 := FALSE; fb_0.EDM2 := TRUE; fb_0.ValveType := TRUE; fb_0.S_StartReset := TRUE; fb_0.Reset := FALSE;
	fb_0();
	failed_0 := NOT ((((((((((((NOT (fb_0.Reset_Before) AND fb_0.S_OutControl_Before) AND fb_0.T_Init.Q) AND fb_0.T_Monitoring.Q) AND (fb_0.DiagCode = 49280)) AND fb_0.Ready) AND NOT (fb_0.S_SafeState)) AND NOT (fb_0.S_ValveOut)) AND (fb_0.S_ValveStatus = fb_0.DiagCode)) AND NOT (fb_0.SafetyDemand)) AND NOT (fb_0.ResetRequest)) AND fb_0.Error));
	testState_0 := testState_0 + 1;
131:
	fb_0.Activate := TRUE; fb_0.S_OutControl := FALSE; fb_0.EDM1 := FALSE; fb_0.EDM2 := TRUE; fb_0.ValveType := TRUE; fb_0.S_StartReset := TRUE; fb_0.Reset := FALSE;
	fb_0();
	failed_0 := NOT ((((((((((((NOT (fb_0.Reset_Before) AND NOT (fb_0.S_OutControl_Before)) AND fb_0.T_Init.Q) AND fb_0.T_Monitoring.Q) AND (fb_0.DiagCode = 50304)) AND fb_0.Ready) AND NOT (fb_0.S_SafeState)) AND NOT (fb_0.S_ValveOut)) AND (fb_0.S_ValveStatus = fb_0.DiagCode)) AND NOT (fb_0.SafetyDemand)) AND fb_0.ResetRequest) AND fb_0.Error));
	testState_0 := testState_0 + 1;
132:
	fb_0.Activate := TRUE; fb_0.S_OutControl := FALSE; fb_0.EDM1 := TRUE; fb_0.EDM2 := TRUE; fb_0.ValveType := TRUE; fb_0.S_StartReset := TRUE; fb_0.Reset := TRUE;
	fb_0();
	failed_0 := NOT ((((((((((((fb_0.Reset_Before AND NOT (fb_0.S_OutControl_Before)) AND fb_0.T_Init.Q) AND NOT (fb_0.T_Monitoring.Q)) AND (fb_0.DiagCode = 34818)) AND fb_0.Ready) AND NOT (fb_0.S_SafeState)) AND NOT (fb_0.S_ValveOut)) AND (fb_0.S_ValveStatus = fb_0.DiagCode)) AND fb_0.SafetyDemand) AND NOT (fb_0.ResetRequest)) AND NOT (fb_0.Error)));
	testState_0 := testState_0 + 1;
133:
	fb_0.Activate := TRUE; fb_0.S_OutControl := FALSE; fb_0.EDM1 := TRUE; fb_0.EDM2 := TRUE; fb_0.ValveType := TRUE; fb_0.S_StartReset := TRUE; fb_0.Reset := FALSE;
	fb_0();
	IF fb_0.T_Monitoring.Q THEN
		finished_0 := TRUE;
	ELSE
		testState_0 := testState_0 + 1;
	END_IF
134:
	failed_0 := NOT ((((((((((((NOT (fb_0.Reset_Before) AND NOT (fb_0.S_OutControl_Before)) AND fb_0.T_Init.Q) AND NOT (fb_0.T_Monitoring.Q)) AND (fb_0.DiagCode = 34820)) AND fb_0.Ready) AND fb_0.S_SafeState) AND NOT (fb_0.S_ValveOut)) AND (fb_0.S_ValveStatus = fb_0.DiagCode)) AND fb_0.SafetyDemand) AND NOT (fb_0.ResetRequest)) AND NOT (fb_0.Error)));
	testState_0 := testState_0 + 1;
135:
	fb_0.Activate := TRUE; fb_0.S_OutControl := TRUE; fb_0.EDM1 := TRUE; fb_0.EDM2 := TRUE; fb_0.ValveType := TRUE; fb_0.S_StartReset := TRUE; fb_0.Reset := FALSE;
	fb_0();
	failed_0 := NOT ((((((((((((NOT (fb_0.Reset_Before) AND fb_0.S_OutControl_Before) AND fb_0.T_Init.Q) AND NOT (fb_0.T_Monitoring.Q)) AND (fb_0.DiagCode = 32800)) AND fb_0.Ready) AND NOT (fb_0.S_SafeState)) AND fb_0.S_ValveOut) AND (fb_0.S_ValveStatus = fb_0.DiagCode)) AND NOT (fb_0.SafetyDemand)) AND NOT (fb_0.ResetRequest)) AND NOT (fb_0.Error)));
	testState_0 := testState_0 + 1;
136:
	fb_0.Activate := TRUE; fb_0.S_OutControl := TRUE; fb_0.EDM1 := FALSE; fb_0.EDM2 := TRUE; fb_0.ValveType := TRUE; fb_0.S_StartReset := TRUE; fb_0.Reset := FALSE;
	fb_0();
	failed_0 := NOT ((((((((((((NOT (fb_0.Reset_Before) AND fb_0.S_OutControl_Before) AND fb_0.T_Init.Q) AND NOT (fb_0.T_Monitoring.Q)) AND (fb_0.DiagCode = 32800)) AND fb_0.Ready) AND NOT (fb_0.S_SafeState)) AND fb_0.S_ValveOut) AND (fb_0.S_ValveStatus = fb_0.DiagCode)) AND NOT (fb_0.SafetyDemand)) AND NOT (fb_0.ResetRequest)) AND NOT (fb_0.Error)));
	testState_0 := testState_0 + 1;
137:
	IF (fb_0.T_Monitoring.Q AND (fb_0.DiagCode = 49280)) THEN
		waitCounter_0 := 0;
		testState_0 := testState_0 + 1;
	ELSE
		failed_0 := NOT ((NOT (fb_0.Reset_Before) AND (fb_0.S_OutControl_Before AND (fb_0.T_Init.Q AND (NOT (fb_0.T_Monitoring.Q) AND ((fb_0.DiagCode = 32800) AND (fb_0.Ready AND (NOT (fb_0.S_SafeState) AND (fb_0.S_ValveOut AND ((fb_0.S_ValveStatus = fb_0.DiagCode) AND (NOT (fb_0.SafetyDemand) AND (NOT (fb_0.ResetRequest) AND NOT (fb_0.Error)))))))))))));
		IF waitCounter_0 > 100 THEN
			finished_0 := TRUE;
		ELSE
			waitCounter_0 := waitCounter_0 + 1;
			fb_0();
		END_IF
	END_IF
138:
	failed_0 := NOT ((((((((((((NOT (fb_0.Reset_Before) AND fb_0.S_OutControl_Before) AND fb_0.T_Init.Q) AND fb_0.T_Monitoring.Q) AND (fb_0.DiagCode = 49280)) AND fb_0.Ready) AND NOT (fb_0.S_SafeState)) AND NOT (fb_0.S_ValveOut)) AND (fb_0.S_ValveStatus = fb_0.DiagCode)) AND NOT (fb_0.SafetyDemand)) AND NOT (fb_0.ResetRequest)) AND fb_0.Error));
	testState_0 := testState_0 + 1;
139:
	fb_0.Activate := TRUE; fb_0.S_OutControl := FALSE; fb_0.EDM1 := TRUE; fb_0.EDM2 := TRUE; fb_0.ValveType := TRUE; fb_0.S_StartReset := TRUE; fb_0.Reset := TRUE;
	fb_0();
	failed_0 := NOT ((((((((((((fb_0.Reset_Before AND NOT (fb_0.S_OutControl_Before)) AND fb_0.T_Init.Q) AND NOT (fb_0.T_Monitoring.Q)) AND (fb_0.DiagCode = 34818)) AND fb_0.Ready) AND NOT (fb_0.S_SafeState)) AND NOT (fb_0.S_ValveOut)) AND (fb_0.S_ValveStatus = fb_0.DiagCode)) AND fb_0.SafetyDemand) AND NOT (fb_0.ResetRequest)) AND NOT (fb_0.Error)));
	testState_0 := testState_0 + 1;
140:
	fb_0.Activate := TRUE; fb_0.S_OutControl := FALSE; fb_0.EDM1 := TRUE; fb_0.EDM2 := TRUE; fb_0.ValveType := TRUE; fb_0.S_StartReset := TRUE; fb_0.Reset := FALSE;
	fb_0();
	IF fb_0.T_Monitoring.Q THEN
		finished_0 := TRUE;
	ELSE
		testState_0 := testState_0 + 1;
	END_IF
141:
	failed_0 := NOT ((((((((((((NOT (fb_0.Reset_Before) AND NOT (fb_0.S_OutControl_Before)) AND fb_0.T_Init.Q) AND NOT (fb_0.T_Monitoring.Q)) AND (fb_0.DiagCode = 34820)) AND fb_0.Ready) AND fb_0.S_SafeState) AND NOT (fb_0.S_ValveOut)) AND (fb_0.S_ValveStatus = fb_0.DiagCode)) AND fb_0.SafetyDemand) AND NOT (fb_0.ResetRequest)) AND NOT (fb_0.Error)));
	testState_0 := testState_0 + 1;
142:
	fb_0.Activate := TRUE; fb_0.S_OutControl := TRUE; fb_0.EDM1 := TRUE; fb_0.EDM2 := TRUE; fb_0.ValveType := TRUE; fb_0.S_StartReset := TRUE; fb_0.Reset := FALSE;
	fb_0();
	failed_0 := NOT ((((((((((((NOT (fb_0.Reset_Before) AND fb_0.S_OutControl_Before) AND fb_0.T_Init.Q) AND NOT (fb_0.T_Monitoring.Q)) AND (fb_0.DiagCode = 32800)) AND fb_0.Ready) AND NOT (fb_0.S_SafeState)) AND fb_0.S_ValveOut) AND (fb_0.S_ValveStatus = fb_0.DiagCode)) AND NOT (fb_0.SafetyDemand)) AND NOT (fb_0.ResetRequest)) AND NOT (fb_0.Error)));
	testState_0 := testState_0 + 1;
143:
	fb_0.Activate := TRUE; fb_0.S_OutControl := TRUE; fb_0.EDM1 := TRUE; fb_0.EDM2 := TRUE; fb_0.ValveType := TRUE; fb_0.S_StartReset := TRUE; fb_0.Reset := FALSE;
	fb_0();
	failed_0 := NOT ((((((((((((NOT (fb_0.Reset_Before) AND fb_0.S_OutControl_Before) AND fb_0.T_Init.Q) AND NOT (fb_0.T_Monitoring.Q)) AND (fb_0.DiagCode = 32800)) AND fb_0.Ready) AND NOT (fb_0.S_SafeState)) AND fb_0.S_ValveOut) AND (fb_0.S_ValveStatus = fb_0.DiagCode)) AND NOT (fb_0.SafetyDemand)) AND NOT (fb_0.ResetRequest)) AND NOT (fb_0.Error)));
	testState_0 := testState_0 + 1;
144:
	IF (fb_0.T_Monitoring.Q AND (fb_0.DiagCode = 49296)) THEN
		waitCounter_0 := 0;
		testState_0 := testState_0 + 1;
	ELSE
		failed_0 := NOT ((NOT (fb_0.Reset_Before) AND (fb_0.S_OutControl_Before AND (fb_0.T_Init.Q AND (NOT (fb_0.T_Monitoring.Q) AND ((fb_0.DiagCode = 32800) AND (fb_0.Ready AND (NOT (fb_0.S_SafeState) AND (fb_0.S_ValveOut AND ((fb_0.S_ValveStatus = fb_0.DiagCode) AND (NOT (fb_0.SafetyDemand) AND (NOT (fb_0.ResetRequest) AND NOT (fb_0.Error)))))))))))));
		IF waitCounter_0 > 100 THEN
			finished_0 := TRUE;
		ELSE
			waitCounter_0 := waitCounter_0 + 1;
			fb_0();
		END_IF
	END_IF
145:
	failed_0 := NOT ((((((((((((NOT (fb_0.Reset_Before) AND fb_0.S_OutControl_Before) AND fb_0.T_Init.Q) AND fb_0.T_Monitoring.Q) AND (fb_0.DiagCode = 49296)) AND fb_0.Ready) AND NOT (fb_0.S_SafeState)) AND NOT (fb_0.S_ValveOut)) AND (fb_0.S_ValveStatus = fb_0.DiagCode)) AND NOT (fb_0.SafetyDemand)) AND NOT (fb_0.ResetRequest)) AND fb_0.Error));
	testState_0 := testState_0 + 1;
146:
	fb_0.Activate := TRUE; fb_0.S_OutControl := TRUE; fb_0.EDM1 := TRUE; fb_0.EDM2 := TRUE; fb_0.ValveType := TRUE; fb_0.S_StartReset := TRUE; fb_0.Reset := TRUE;
	fb_0();
	failed_0 := NOT ((((((((((((fb_0.Reset_Before AND fb_0.S_OutControl_Before) AND fb_0.T_Init.Q) AND fb_0.T_Monitoring.Q) AND (fb_0.DiagCode = 49296)) AND fb_0.Ready) AND NOT (fb_0.S_SafeState)) AND NOT (fb_0.S_ValveOut)) AND (fb_0.S_ValveStatus = fb_0.DiagCode)) AND NOT (fb_0.SafetyDemand)) AND NOT (fb_0.ResetRequest)) AND fb_0.Error));
	testState_0 := testState_0 + 1;
147:
	fb_0.Activate := TRUE; fb_0.S_OutControl := TRUE; fb_0.EDM1 := TRUE; fb_0.EDM2 := TRUE; fb_0.ValveType := TRUE; fb_0.S_StartReset := TRUE; fb_0.Reset := TRUE;
	fb_0();
	failed_0 := NOT ((((((((((((fb_0.Reset_Before AND fb_0.S_OutControl_Before) AND fb_0.T_Init.Q) AND fb_0.T_Monitoring.Q) AND (fb_0.DiagCode = 49297)) AND fb_0.Ready) AND NOT (fb_0.S_SafeState)) AND NOT (fb_0.S_ValveOut)) AND (fb_0.S_ValveStatus = fb_0.DiagCode)) AND NOT (fb_0.SafetyDemand)) AND NOT (fb_0.ResetRequest)) AND fb_0.Error));
	testState_0 := testState_0 + 1;
148:
	fb_0.Activate := TRUE; fb_0.S_OutControl := TRUE; fb_0.EDM1 := TRUE; fb_0.EDM2 := TRUE; fb_0.ValveType := TRUE; fb_0.S_StartReset := TRUE; fb_0.Reset := TRUE;
	fb_0();
	failed_0 := NOT ((((((((((((fb_0.Reset_Before AND fb_0.S_OutControl_Before) AND fb_0.T_Init.Q) AND fb_0.T_Monitoring.Q) AND (fb_0.DiagCode = 49297)) AND fb_0.Ready) AND NOT (fb_0.S_SafeState)) AND NOT (fb_0.S_ValveOut)) AND (fb_0.S_ValveStatus = fb_0.DiagCode)) AND NOT (fb_0.SafetyDemand)) AND NOT (fb_0.ResetRequest)) AND fb_0.Error));
	testState_0 := testState_0 + 1;
149:
	fb_0.Activate := TRUE; fb_0.S_OutControl := TRUE; fb_0.EDM1 := TRUE; fb_0.EDM2 := TRUE; fb_0.ValveType := TRUE; fb_0.S_StartReset := TRUE; fb_0.Reset := FALSE;
	fb_0();
	failed_0 := NOT ((((((((((((NOT (fb_0.Reset_Before) AND fb_0.S_OutControl_Before) AND fb_0.T_Init.Q) AND fb_0.T_Monitoring.Q) AND (fb_0.DiagCode = 49296)) AND fb_0.Ready) AND NOT (fb_0.S_SafeState)) AND NOT (fb_0.S_ValveOut)) AND (fb_0.S_ValveStatus = fb_0.DiagCode)) AND NOT (fb_0.SafetyDemand)) AND NOT (fb_0.ResetRequest)) AND fb_0.Error));
	testState_0 := testState_0 + 1;
150:
	fb_0.Activate := TRUE; fb_0.S_OutControl := FALSE; fb_0.EDM1 := TRUE; fb_0.EDM2 := TRUE; fb_0.ValveType := TRUE; fb_0.S_StartReset := TRUE; fb_0.Reset := FALSE;
	fb_0();
	failed_0 := NOT ((((((((((((NOT (fb_0.Reset_Before) AND NOT (fb_0.S_OutControl_Before)) AND fb_0.T_Init.Q) AND fb_0.T_Monitoring.Q) AND (fb_0.DiagCode = 50320)) AND fb_0.Ready) AND NOT (fb_0.S_SafeState)) AND NOT (fb_0.S_ValveOut)) AND (fb_0.S_ValveStatus = fb_0.DiagCode)) AND NOT (fb_0.SafetyDemand)) AND fb_0.ResetRequest) AND fb_0.Error));
	testState_0 := testState_0 + 1;
151:
	fb_0.Activate := TRUE; fb_0.S_OutControl := FALSE; fb_0.EDM1 := TRUE; fb_0.EDM2 := TRUE; fb_0.ValveType := TRUE; fb_0.S_StartReset := TRUE; fb_0.Reset := FALSE;
	fb_0();
	failed_0 := NOT ((((((((((((NOT (fb_0.Reset_Before) AND NOT (fb_0.S_OutControl_Before)) AND fb_0.T_Init.Q) AND fb_0.T_Monitoring.Q) AND (fb_0.DiagCode = 50320)) AND fb_0.Ready) AND NOT (fb_0.S_SafeState)) AND NOT (fb_0.S_ValveOut)) AND (fb_0.S_ValveStatus = fb_0.DiagCode)) AND NOT (fb_0.SafetyDemand)) AND fb_0.ResetRequest) AND fb_0.Error));
	testState_0 := testState_0 + 1;
152:
	fb_0.Activate := TRUE; fb_0.S_OutControl := TRUE; fb_0.EDM1 := TRUE; fb_0.EDM2 := TRUE; fb_0.ValveType := TRUE; fb_0.S_StartReset := TRUE; fb_0.Reset := FALSE;
	fb_0();
	failed_0 := NOT ((((((((((((NOT (fb_0.Reset_Before) AND fb_0.S_OutControl_Before) AND fb_0.T_Init.Q) AND fb_0.T_Monitoring.Q) AND (fb_0.DiagCode = 49296)) AND fb_0.Ready) AND NOT (fb_0.S_SafeState)) AND NOT (fb_0.S_ValveOut)) AND (fb_0.S_ValveStatus = fb_0.DiagCode)) AND NOT (fb_0.SafetyDemand)) AND NOT (fb_0.ResetRequest)) AND fb_0.Error));
	testState_0 := testState_0 + 1;
153:
	fb_0.Activate := TRUE; fb_0.S_OutControl := FALSE; fb_0.EDM1 := TRUE; fb_0.EDM2 := TRUE; fb_0.ValveType := TRUE; fb_0.S_StartReset := TRUE; fb_0.Reset := FALSE;
	fb_0();
	failed_0 := NOT ((((((((((((NOT (fb_0.Reset_Before) AND NOT (fb_0.S_OutControl_Before)) AND fb_0.T_Init.Q) AND fb_0.T_Monitoring.Q) AND (fb_0.DiagCode = 50320)) AND fb_0.Ready) AND NOT (fb_0.S_SafeState)) AND NOT (fb_0.S_ValveOut)) AND (fb_0.S_ValveStatus = fb_0.DiagCode)) AND NOT (fb_0.SafetyDemand)) AND fb_0.ResetRequest) AND fb_0.Error));
	testState_0 := testState_0 + 1;
154:
	fb_0.Activate := TRUE; fb_0.S_OutControl := FALSE; fb_0.EDM1 := TRUE; fb_0.EDM2 := TRUE; fb_0.ValveType := TRUE; fb_0.S_StartReset := TRUE; fb_0.Reset := TRUE;
	fb_0();
	failed_0 := NOT ((((((((((((fb_0.Reset_Before AND NOT (fb_0.S_OutControl_Before)) AND fb_0.T_Init.Q) AND NOT (fb_0.T_Monitoring.Q)) AND (fb_0.DiagCode = 34818)) AND fb_0.Ready) AND NOT (fb_0.S_SafeState)) AND NOT (fb_0.S_ValveOut)) AND (fb_0.S_ValveStatus = fb_0.DiagCode)) AND fb_0.SafetyDemand) AND NOT (fb_0.ResetRequest)) AND NOT (fb_0.Error)));
	testState_0 := testState_0 + 1;
155:
	fb_0.Activate := TRUE; fb_0.S_OutControl := FALSE; fb_0.EDM1 := TRUE; fb_0.EDM2 := TRUE; fb_0.ValveType := TRUE; fb_0.S_StartReset := TRUE; fb_0.Reset := FALSE;
	fb_0();
	IF fb_0.T_Monitoring.Q THEN
		finished_0 := TRUE;
	ELSE
		testState_0 := testState_0 + 1;
	END_IF
156:
	failed_0 := NOT ((((((((((((NOT (fb_0.Reset_Before) AND NOT (fb_0.S_OutControl_Before)) AND fb_0.T_Init.Q) AND NOT (fb_0.T_Monitoring.Q)) AND (fb_0.DiagCode = 34820)) AND fb_0.Ready) AND fb_0.S_SafeState) AND NOT (fb_0.S_ValveOut)) AND (fb_0.S_ValveStatus = fb_0.DiagCode)) AND fb_0.SafetyDemand) AND NOT (fb_0.ResetRequest)) AND NOT (fb_0.Error)));
	testState_0 := testState_0 + 1;
157:
	fb_0.Activate := TRUE; fb_0.S_OutControl := TRUE; fb_0.EDM1 := TRUE; fb_0.EDM2 := TRUE; fb_0.ValveType := TRUE; fb_0.S_StartReset := TRUE; fb_0.Reset := FALSE;
	fb_0();
	failed_0 := NOT ((((((((((((NOT (fb_0.Reset_Before) AND fb_0.S_OutControl_Before) AND fb_0.T_Init.Q) AND NOT (fb_0.T_Monitoring.Q)) AND (fb_0.DiagCode = 32800)) AND fb_0.Ready) AND NOT (fb_0.S_SafeState)) AND fb_0.S_ValveOut) AND (fb_0.S_ValveStatus = fb_0.DiagCode)) AND NOT (fb_0.SafetyDemand)) AND NOT (fb_0.ResetRequest)) AND NOT (fb_0.Error)));
	testState_0 := testState_0 + 1;
158:
	fb_0.Activate := TRUE; fb_0.S_OutControl := TRUE; fb_0.EDM1 := TRUE; fb_0.EDM2 := TRUE; fb_0.ValveType := TRUE; fb_0.S_StartReset := TRUE; fb_0.Reset := FALSE;
	fb_0();
	failed_0 := NOT ((((((((((((NOT (fb_0.Reset_Before) AND fb_0.S_OutControl_Before) AND fb_0.T_Init.Q) AND NOT (fb_0.T_Monitoring.Q)) AND (fb_0.DiagCode = 32800)) AND fb_0.Ready) AND NOT (fb_0.S_SafeState)) AND fb_0.S_ValveOut) AND (fb_0.S_ValveStatus = fb_0.DiagCode)) AND NOT (fb_0.SafetyDemand)) AND NOT (fb_0.ResetRequest)) AND NOT (fb_0.Error)));
	testState_0 := testState_0 + 1;
159:
	IF (fb_0.T_Monitoring.Q AND (fb_0.DiagCode = 49296)) THEN
		waitCounter_0 := 0;
		testState_0 := testState_0 + 1;
	ELSE
		failed_0 := NOT ((NOT (fb_0.Reset_Before) AND (fb_0.S_OutControl_Before AND (fb_0.T_Init.Q AND (NOT (fb_0.T_Monitoring.Q) AND ((fb_0.DiagCode = 32800) AND (fb_0.Ready AND (NOT (fb_0.S_SafeState) AND (fb_0.S_ValveOut AND ((fb_0.S_ValveStatus = fb_0.DiagCode) AND (NOT (fb_0.SafetyDemand) AND (NOT (fb_0.ResetRequest) AND NOT (fb_0.Error)))))))))))));
		IF waitCounter_0 > 100 THEN
			finished_0 := TRUE;
		ELSE
			waitCounter_0 := waitCounter_0 + 1;
			fb_0();
		END_IF
	END_IF
160:
	failed_0 := NOT ((((((((((((NOT (fb_0.Reset_Before) AND fb_0.S_OutControl_Before) AND fb_0.T_Init.Q) AND fb_0.T_Monitoring.Q) AND (fb_0.DiagCode = 49296)) AND fb_0.Ready) AND NOT (fb_0.S_SafeState)) AND NOT (fb_0.S_ValveOut)) AND (fb_0.S_ValveStatus = fb_0.DiagCode)) AND NOT (fb_0.SafetyDemand)) AND NOT (fb_0.ResetRequest)) AND fb_0.Error));
	testState_0 := testState_0 + 1;
161:
	fb_0.Activate := TRUE; fb_0.S_OutControl := FALSE; fb_0.EDM1 := TRUE; fb_0.EDM2 := TRUE; fb_0.ValveType := TRUE; fb_0.S_StartReset := TRUE; fb_0.Reset := TRUE;
	fb_0();
	failed_0 := NOT ((((((((((((fb_0.Reset_Before AND NOT (fb_0.S_OutControl_Before)) AND fb_0.T_Init.Q) AND NOT (fb_0.T_Monitoring.Q)) AND (fb_0.DiagCode = 34818)) AND fb_0.Ready) AND NOT (fb_0.S_SafeState)) AND NOT (fb_0.S_ValveOut)) AND (fb_0.S_ValveStatus = fb_0.DiagCode)) AND fb_0.SafetyDemand) AND NOT (fb_0.ResetRequest)) AND NOT (fb_0.Error)));
	testState_0 := testState_0 + 1;
162:
	fb_0.Activate := TRUE; fb_0.S_OutControl := TRUE; fb_0.EDM1 := FALSE; fb_0.EDM2 := TRUE; fb_0.ValveType := TRUE; fb_0.S_StartReset := TRUE; fb_0.Reset := FALSE;
	fb_0();
	failed_0 := NOT ((((((((((((NOT (fb_0.Reset_Before) AND fb_0.S_OutControl_Before) AND fb_0.T_Init.Q) AND NOT (fb_0.T_Monitoring.Q)) AND (fb_0.DiagCode = 49168)) AND fb_0.Ready) AND NOT (fb_0.S_SafeState)) AND NOT (fb_0.S_ValveOut)) AND (fb_0.S_ValveStatus = fb_0.DiagCode)) AND NOT (fb_0.SafetyDemand)) AND NOT (fb_0.ResetRequest)) AND fb_0.Error));
	testState_0 := testState_0 + 1;
163:
	fb_0.Activate := TRUE; fb_0.S_OutControl := TRUE; fb_0.EDM1 := FALSE; fb_0.EDM2 := TRUE; fb_0.ValveType := TRUE; fb_0.S_StartReset := TRUE; fb_0.Reset := TRUE;
	fb_0();
	failed_0 := NOT ((((((((((((fb_0.Reset_Before AND fb_0.S_OutControl_Before) AND fb_0.T_Init.Q) AND NOT (fb_0.T_Monitoring.Q)) AND (fb_0.DiagCode = 49168)) AND fb_0.Ready) AND NOT (fb_0.S_SafeState)) AND NOT (fb_0.S_ValveOut)) AND (fb_0.S_ValveStatus = fb_0.DiagCode)) AND NOT (fb_0.SafetyDemand)) AND NOT (fb_0.ResetRequest)) AND fb_0.Error));
	testState_0 := testState_0 + 1;
164:
	fb_0.Activate := TRUE; fb_0.S_OutControl := TRUE; fb_0.EDM1 := FALSE; fb_0.EDM2 := TRUE; fb_0.ValveType := TRUE; fb_0.S_StartReset := TRUE; fb_0.Reset := TRUE;
	fb_0();
	failed_0 := NOT ((((((((((((fb_0.Reset_Before AND fb_0.S_OutControl_Before) AND fb_0.T_Init.Q) AND NOT (fb_0.T_Monitoring.Q)) AND (fb_0.DiagCode = 49169)) AND fb_0.Ready) AND NOT (fb_0.S_SafeState)) AND NOT (fb_0.S_ValveOut)) AND (fb_0.S_ValveStatus = fb_0.DiagCode)) AND NOT (fb_0.SafetyDemand)) AND NOT (fb_0.ResetRequest)) AND fb_0.Error));
	testState_0 := testState_0 + 1;
165:
	fb_0.Activate := TRUE; fb_0.S_OutControl := TRUE; fb_0.EDM1 := FALSE; fb_0.EDM2 := TRUE; fb_0.ValveType := TRUE; fb_0.S_StartReset := TRUE; fb_0.Reset := TRUE;
	fb_0();
	failed_0 := NOT ((((((((((((fb_0.Reset_Before AND fb_0.S_OutControl_Before) AND fb_0.T_Init.Q) AND NOT (fb_0.T_Monitoring.Q)) AND (fb_0.DiagCode = 49169)) AND fb_0.Ready) AND NOT (fb_0.S_SafeState)) AND NOT (fb_0.S_ValveOut)) AND (fb_0.S_ValveStatus = fb_0.DiagCode)) AND NOT (fb_0.SafetyDemand)) AND NOT (fb_0.ResetRequest)) AND fb_0.Error));
	testState_0 := testState_0 + 1;
166:
	fb_0.Activate := TRUE; fb_0.S_OutControl := TRUE; fb_0.EDM1 := FALSE; fb_0.EDM2 := TRUE; fb_0.ValveType := TRUE; fb_0.S_StartReset := TRUE; fb_0.Reset := FALSE;
	fb_0();
	failed_0 := NOT ((((((((((((NOT (fb_0.Reset_Before) AND fb_0.S_OutControl_Before) AND fb_0.T_Init.Q) AND NOT (fb_0.T_Monitoring.Q)) AND (fb_0.DiagCode = 49168)) AND fb_0.Ready) AND NOT (fb_0.S_SafeState)) AND NOT (fb_0.S_ValveOut)) AND (fb_0.S_ValveStatus = fb_0.DiagCode)) AND NOT (fb_0.SafetyDemand)) AND NOT (fb_0.ResetRequest)) AND fb_0.Error));
	testState_0 := testState_0 + 1;
167:
	fb_0.Activate := TRUE; fb_0.S_OutControl := FALSE; fb_0.EDM1 := TRUE; fb_0.EDM2 := TRUE; fb_0.ValveType := TRUE; fb_0.S_StartReset := TRUE; fb_0.Reset := TRUE;
	fb_0();
	failed_0 := NOT ((((((((((((fb_0.Reset_Before AND NOT (fb_0.S_OutControl_Before)) AND fb_0.T_Init.Q) AND NOT (fb_0.T_Monitoring.Q)) AND (fb_0.DiagCode = 34818)) AND fb_0.Ready) AND NOT (fb_0.S_SafeState)) AND NOT (fb_0.S_ValveOut)) AND (fb_0.S_ValveStatus = fb_0.DiagCode)) AND fb_0.SafetyDemand) AND NOT (fb_0.ResetRequest)) AND NOT (fb_0.Error)));
	testState_0 := testState_0 + 1;
168:
	fb_0.Activate := TRUE; fb_0.S_OutControl := TRUE; fb_0.EDM1 := FALSE; fb_0.EDM2 := TRUE; fb_0.ValveType := TRUE; fb_0.S_StartReset := TRUE; fb_0.Reset := FALSE;
	fb_0();
	failed_0 := NOT ((((((((((((NOT (fb_0.Reset_Before) AND fb_0.S_OutControl_Before) AND fb_0.T_Init.Q) AND NOT (fb_0.T_Monitoring.Q)) AND (fb_0.DiagCode = 49168)) AND fb_0.Ready) AND NOT (fb_0.S_SafeState)) AND NOT (fb_0.S_ValveOut)) AND (fb_0.S_ValveStatus = fb_0.DiagCode)) AND NOT (fb_0.SafetyDemand)) AND NOT (fb_0.ResetRequest)) AND fb_0.Error));
	testState_0 := testState_0 + 1;
169:
	fb_0.Activate := TRUE; fb_0.S_OutControl := FALSE; fb_0.EDM1 := FALSE; fb_0.EDM2 := TRUE; fb_0.ValveType := TRUE; fb_0.S_StartReset := TRUE; fb_0.Reset := FALSE;
	fb_0();
	failed_0 := NOT ((((((((((((NOT (fb_0.Reset_Before) AND NOT (fb_0.S_OutControl_Before)) AND fb_0.T_Init.Q) AND NOT (fb_0.T_Monitoring.Q)) AND (fb_0.DiagCode = 50192)) AND fb_0.Ready) AND NOT (fb_0.S_SafeState)) AND NOT (fb_0.S_ValveOut)) AND (fb_0.S_ValveStatus = fb_0.DiagCode)) AND NOT (fb_0.SafetyDemand)) AND fb_0.ResetRequest) AND fb_0.Error));
	testState_0 := testState_0 + 1;
170:
	fb_0.Activate := TRUE; fb_0.S_OutControl := FALSE; fb_0.EDM1 := FALSE; fb_0.EDM2 := TRUE; fb_0.ValveType := TRUE; fb_0.S_StartReset := TRUE; fb_0.Reset := TRUE;
	fb_0();
	failed_0 := NOT ((((((((((((fb_0.Reset_Before AND NOT (fb_0.S_OutControl_Before)) AND fb_0.T_Init.Q) AND NOT (fb_0.T_Monitoring.Q)) AND (fb_0.DiagCode = 50192)) AND fb_0.Ready) AND NOT (fb_0.S_SafeState)) AND NOT (fb_0.S_ValveOut)) AND (fb_0.S_ValveStatus = fb_0.DiagCode)) AND NOT (fb_0.SafetyDemand)) AND fb_0.ResetRequest) AND fb_0.Error));
	testState_0 := testState_0 + 1;
171:
	fb_0.Activate := TRUE; fb_0.S_OutControl := FALSE; fb_0.EDM1 := FALSE; fb_0.EDM2 := TRUE; fb_0.ValveType := TRUE; fb_0.S_StartReset := TRUE; fb_0.Reset := TRUE;
	fb_0();
	failed_0 := NOT ((((((((((((fb_0.Reset_Before AND NOT (fb_0.S_OutControl_Before)) AND fb_0.T_Init.Q) AND NOT (fb_0.T_Monitoring.Q)) AND (fb_0.DiagCode = 49169)) AND fb_0.Ready) AND NOT (fb_0.S_SafeState)) AND NOT (fb_0.S_ValveOut)) AND (fb_0.S_ValveStatus = fb_0.DiagCode)) AND NOT (fb_0.SafetyDemand)) AND NOT (fb_0.ResetRequest)) AND fb_0.Error));
	testState_0 := testState_0 + 1;
172:
	fb_0.Activate := TRUE; fb_0.S_OutControl := FALSE; fb_0.EDM1 := FALSE; fb_0.EDM2 := TRUE; fb_0.ValveType := TRUE; fb_0.S_StartReset := TRUE; fb_0.Reset := FALSE;
	fb_0();
	failed_0 := NOT ((((((((((((NOT (fb_0.Reset_Before) AND NOT (fb_0.S_OutControl_Before)) AND fb_0.T_Init.Q) AND NOT (fb_0.T_Monitoring.Q)) AND (fb_0.DiagCode = 50192)) AND fb_0.Ready) AND NOT (fb_0.S_SafeState)) AND NOT (fb_0.S_ValveOut)) AND (fb_0.S_ValveStatus = fb_0.DiagCode)) AND NOT (fb_0.SafetyDemand)) AND fb_0.ResetRequest) AND fb_0.Error));
	testState_0 := testState_0 + 1;
173:
	fb_0.Activate := TRUE; fb_0.S_OutControl := TRUE; fb_0.EDM1 := FALSE; fb_0.EDM2 := TRUE; fb_0.ValveType := TRUE; fb_0.S_StartReset := TRUE; fb_0.Reset := FALSE;
	fb_0();
	failed_0 := NOT ((((((((((((NOT (fb_0.Reset_Before) AND fb_0.S_OutControl_Before) AND fb_0.T_Init.Q) AND NOT (fb_0.T_Monitoring.Q)) AND (fb_0.DiagCode = 49168)) AND fb_0.Ready) AND NOT (fb_0.S_SafeState)) AND NOT (fb_0.S_ValveOut)) AND (fb_0.S_ValveStatus = fb_0.DiagCode)) AND NOT (fb_0.SafetyDemand)) AND NOT (fb_0.ResetRequest)) AND fb_0.Error));
	testState_0 := testState_0 + 1;
174:
	fb_0.Activate := TRUE; fb_0.S_OutControl := FALSE; fb_0.EDM1 := FALSE; fb_0.EDM2 := TRUE; fb_0.ValveType := TRUE; fb_0.S_StartReset := TRUE; fb_0.Reset := FALSE;
	fb_0();
	failed_0 := NOT ((((((((((((NOT (fb_0.Reset_Before) AND NOT (fb_0.S_OutControl_Before)) AND fb_0.T_Init.Q) AND NOT (fb_0.T_Monitoring.Q)) AND (fb_0.DiagCode = 50192)) AND fb_0.Ready) AND NOT (fb_0.S_SafeState)) AND NOT (fb_0.S_ValveOut)) AND (fb_0.S_ValveStatus = fb_0.DiagCode)) AND NOT (fb_0.SafetyDemand)) AND fb_0.ResetRequest) AND fb_0.Error));
	testState_0 := testState_0 + 1;
175:
	fb_0.Activate := TRUE; fb_0.S_OutControl := FALSE; fb_0.EDM1 := TRUE; fb_0.EDM2 := TRUE; fb_0.ValveType := TRUE; fb_0.S_StartReset := TRUE; fb_0.Reset := TRUE;
	fb_0();
	failed_0 := NOT ((((((((((((fb_0.Reset_Before AND NOT (fb_0.S_OutControl_Before)) AND fb_0.T_Init.Q) AND NOT (fb_0.T_Monitoring.Q)) AND (fb_0.DiagCode = 34818)) AND fb_0.Ready) AND NOT (fb_0.S_SafeState)) AND NOT (fb_0.S_ValveOut)) AND (fb_0.S_ValveStatus = fb_0.DiagCode)) AND fb_0.SafetyDemand) AND NOT (fb_0.ResetRequest)) AND NOT (fb_0.Error)));
	testState_0 := testState_0 + 1;
176:
	fb_0.Activate := TRUE; fb_0.S_OutControl := TRUE; fb_0.EDM1 := TRUE; fb_0.EDM2 := FALSE; fb_0.ValveType := TRUE; fb_0.S_StartReset := TRUE; fb_0.Reset := FALSE;
	fb_0();
	failed_0 := NOT ((((((((((((NOT (fb_0.Reset_Before) AND fb_0.S_OutControl_Before) AND fb_0.T_Init.Q) AND NOT (fb_0.T_Monitoring.Q)) AND (fb_0.DiagCode = 49184)) AND fb_0.Ready) AND NOT (fb_0.S_SafeState)) AND NOT (fb_0.S_ValveOut)) AND (fb_0.S_ValveStatus = fb_0.DiagCode)) AND NOT (fb_0.SafetyDemand)) AND NOT (fb_0.ResetRequest)) AND fb_0.Error));
	testState_0 := testState_0 + 1;
177:
	fb_0.Activate := TRUE; fb_0.S_OutControl := TRUE; fb_0.EDM1 := TRUE; fb_0.EDM2 := FALSE; fb_0.ValveType := TRUE; fb_0.S_StartReset := TRUE; fb_0.Reset := TRUE;
	fb_0();
	failed_0 := NOT ((((((((((((fb_0.Reset_Before AND fb_0.S_OutControl_Before) AND fb_0.T_Init.Q) AND NOT (fb_0.T_Monitoring.Q)) AND (fb_0.DiagCode = 49184)) AND fb_0.Ready) AND NOT (fb_0.S_SafeState)) AND NOT (fb_0.S_ValveOut)) AND (fb_0.S_ValveStatus = fb_0.DiagCode)) AND NOT (fb_0.SafetyDemand)) AND NOT (fb_0.ResetRequest)) AND fb_0.Error));
	testState_0 := testState_0 + 1;
178:
	fb_0.Activate := TRUE; fb_0.S_OutControl := TRUE; fb_0.EDM1 := TRUE; fb_0.EDM2 := FALSE; fb_0.ValveType := TRUE; fb_0.S_StartReset := TRUE; fb_0.Reset := TRUE;
	fb_0();
	failed_0 := NOT ((((((((((((fb_0.Reset_Before AND fb_0.S_OutControl_Before) AND fb_0.T_Init.Q) AND NOT (fb_0.T_Monitoring.Q)) AND (fb_0.DiagCode = 49185)) AND fb_0.Ready) AND NOT (fb_0.S_SafeState)) AND NOT (fb_0.S_ValveOut)) AND (fb_0.S_ValveStatus = fb_0.DiagCode)) AND NOT (fb_0.SafetyDemand)) AND NOT (fb_0.ResetRequest)) AND fb_0.Error));
	testState_0 := testState_0 + 1;
179:
	fb_0.Activate := TRUE; fb_0.S_OutControl := TRUE; fb_0.EDM1 := TRUE; fb_0.EDM2 := FALSE; fb_0.ValveType := TRUE; fb_0.S_StartReset := TRUE; fb_0.Reset := TRUE;
	fb_0();
	failed_0 := NOT ((((((((((((fb_0.Reset_Before AND fb_0.S_OutControl_Before) AND fb_0.T_Init.Q) AND NOT (fb_0.T_Monitoring.Q)) AND (fb_0.DiagCode = 49185)) AND fb_0.Ready) AND NOT (fb_0.S_SafeState)) AND NOT (fb_0.S_ValveOut)) AND (fb_0.S_ValveStatus = fb_0.DiagCode)) AND NOT (fb_0.SafetyDemand)) AND NOT (fb_0.ResetRequest)) AND fb_0.Error));
	testState_0 := testState_0 + 1;
180:
	fb_0.Activate := TRUE; fb_0.S_OutControl := TRUE; fb_0.EDM1 := TRUE; fb_0.EDM2 := FALSE; fb_0.ValveType := TRUE; fb_0.S_StartReset := TRUE; fb_0.Reset := FALSE;
	fb_0();
	failed_0 := NOT ((((((((((((NOT (fb_0.Reset_Before) AND fb_0.S_OutControl_Before) AND fb_0.T_Init.Q) AND NOT (fb_0.T_Monitoring.Q)) AND (fb_0.DiagCode = 49184)) AND fb_0.Ready) AND NOT (fb_0.S_SafeState)) AND NOT (fb_0.S_ValveOut)) AND (fb_0.S_ValveStatus = fb_0.DiagCode)) AND NOT (fb_0.SafetyDemand)) AND NOT (fb_0.ResetRequest)) AND fb_0.Error));
	testState_0 := testState_0 + 1;
181:
	fb_0.Activate := TRUE; fb_0.S_OutControl := FALSE; fb_0.EDM1 := TRUE; fb_0.EDM2 := TRUE; fb_0.ValveType := TRUE; fb_0.S_StartReset := TRUE; fb_0.Reset := TRUE;
	fb_0();
	failed_0 := NOT ((((((((((((fb_0.Reset_Before AND NOT (fb_0.S_OutControl_Before)) AND fb_0.T_Init.Q) AND NOT (fb_0.T_Monitoring.Q)) AND (fb_0.DiagCode = 34818)) AND fb_0.Ready) AND NOT (fb_0.S_SafeState)) AND NOT (fb_0.S_ValveOut)) AND (fb_0.S_ValveStatus = fb_0.DiagCode)) AND fb_0.SafetyDemand) AND NOT (fb_0.ResetRequest)) AND NOT (fb_0.Error)));
	testState_0 := testState_0 + 1;
182:
	fb_0.Activate := TRUE; fb_0.S_OutControl := TRUE; fb_0.EDM1 := TRUE; fb_0.EDM2 := FALSE; fb_0.ValveType := TRUE; fb_0.S_StartReset := TRUE; fb_0.Reset := FALSE;
	fb_0();
	failed_0 := NOT ((((((((((((NOT (fb_0.Reset_Before) AND fb_0.S_OutControl_Before) AND fb_0.T_Init.Q) AND NOT (fb_0.T_Monitoring.Q)) AND (fb_0.DiagCode = 49184)) AND fb_0.Ready) AND NOT (fb_0.S_SafeState)) AND NOT (fb_0.S_ValveOut)) AND (fb_0.S_ValveStatus = fb_0.DiagCode)) AND NOT (fb_0.SafetyDemand)) AND NOT (fb_0.ResetRequest)) AND fb_0.Error));
	testState_0 := testState_0 + 1;
183:
	fb_0.Activate := TRUE; fb_0.S_OutControl := FALSE; fb_0.EDM1 := TRUE; fb_0.EDM2 := FALSE; fb_0.ValveType := TRUE; fb_0.S_StartReset := TRUE; fb_0.Reset := FALSE;
	fb_0();
	failed_0 := NOT ((((((((((((NOT (fb_0.Reset_Before) AND NOT (fb_0.S_OutControl_Before)) AND fb_0.T_Init.Q) AND NOT (fb_0.T_Monitoring.Q)) AND (fb_0.DiagCode = 50208)) AND fb_0.Ready) AND NOT (fb_0.S_SafeState)) AND NOT (fb_0.S_ValveOut)) AND (fb_0.S_ValveStatus = fb_0.DiagCode)) AND NOT (fb_0.SafetyDemand)) AND fb_0.ResetRequest) AND fb_0.Error));
	testState_0 := testState_0 + 1;
184:
	fb_0.Activate := TRUE; fb_0.S_OutControl := FALSE; fb_0.EDM1 := TRUE; fb_0.EDM2 := FALSE; fb_0.ValveType := TRUE; fb_0.S_StartReset := TRUE; fb_0.Reset := TRUE;
	fb_0();
	failed_0 := NOT ((((((((((((fb_0.Reset_Before AND NOT (fb_0.S_OutControl_Before)) AND fb_0.T_Init.Q) AND NOT (fb_0.T_Monitoring.Q)) AND (fb_0.DiagCode = 50208)) AND fb_0.Ready) AND NOT (fb_0.S_SafeState)) AND NOT (fb_0.S_ValveOut)) AND (fb_0.S_ValveStatus = fb_0.DiagCode)) AND NOT (fb_0.SafetyDemand)) AND fb_0.ResetRequest) AND fb_0.Error));
	testState_0 := testState_0 + 1;
185:
	fb_0.Activate := TRUE; fb_0.S_OutControl := FALSE; fb_0.EDM1 := TRUE; fb_0.EDM2 := FALSE; fb_0.ValveType := TRUE; fb_0.S_StartReset := TRUE; fb_0.Reset := TRUE;
	fb_0();
	failed_0 := NOT ((((((((((((fb_0.Reset_Before AND NOT (fb_0.S_OutControl_Before)) AND fb_0.T_Init.Q) AND NOT (fb_0.T_Monitoring.Q)) AND (fb_0.DiagCode = 49185)) AND fb_0.Ready) AND NOT (fb_0.S_SafeState)) AND NOT (fb_0.S_ValveOut)) AND (fb_0.S_ValveStatus = fb_0.DiagCode)) AND NOT (fb_0.SafetyDemand)) AND NOT (fb_0.ResetRequest)) AND fb_0.Error));
	testState_0 := testState_0 + 1;
186:
	fb_0.Activate := TRUE; fb_0.S_OutControl := FALSE; fb_0.EDM1 := TRUE; fb_0.EDM2 := FALSE; fb_0.ValveType := TRUE; fb_0.S_StartReset := TRUE; fb_0.Reset := FALSE;
	fb_0();
	failed_0 := NOT ((((((((((((NOT (fb_0.Reset_Before) AND NOT (fb_0.S_OutControl_Before)) AND fb_0.T_Init.Q) AND NOT (fb_0.T_Monitoring.Q)) AND (fb_0.DiagCode = 50208)) AND fb_0.Ready) AND NOT (fb_0.S_SafeState)) AND NOT (fb_0.S_ValveOut)) AND (fb_0.S_ValveStatus = fb_0.DiagCode)) AND NOT (fb_0.SafetyDemand)) AND fb_0.ResetRequest) AND fb_0.Error));
	testState_0 := testState_0 + 1;
187:
	fb_0.Activate := TRUE; fb_0.S_OutControl := TRUE; fb_0.EDM1 := TRUE; fb_0.EDM2 := FALSE; fb_0.ValveType := TRUE; fb_0.S_StartReset := TRUE; fb_0.Reset := FALSE;
	fb_0();
	failed_0 := NOT ((((((((((((NOT (fb_0.Reset_Before) AND fb_0.S_OutControl_Before) AND fb_0.T_Init.Q) AND NOT (fb_0.T_Monitoring.Q)) AND (fb_0.DiagCode = 49184)) AND fb_0.Ready) AND NOT (fb_0.S_SafeState)) AND NOT (fb_0.S_ValveOut)) AND (fb_0.S_ValveStatus = fb_0.DiagCode)) AND NOT (fb_0.SafetyDemand)) AND NOT (fb_0.ResetRequest)) AND fb_0.Error));
	testState_0 := testState_0 + 1;
188:
	fb_0.Activate := TRUE; fb_0.S_OutControl := FALSE; fb_0.EDM1 := TRUE; fb_0.EDM2 := FALSE; fb_0.ValveType := TRUE; fb_0.S_StartReset := TRUE; fb_0.Reset := FALSE;
	fb_0();
	failed_0 := NOT ((((((((((((NOT (fb_0.Reset_Before) AND NOT (fb_0.S_OutControl_Before)) AND fb_0.T_Init.Q) AND NOT (fb_0.T_Monitoring.Q)) AND (fb_0.DiagCode = 50208)) AND fb_0.Ready) AND NOT (fb_0.S_SafeState)) AND NOT (fb_0.S_ValveOut)) AND (fb_0.S_ValveStatus = fb_0.DiagCode)) AND NOT (fb_0.SafetyDemand)) AND fb_0.ResetRequest) AND fb_0.Error));
	testState_0 := testState_0 + 1;
189:
	fb_0.Activate := TRUE; fb_0.S_OutControl := FALSE; fb_0.EDM1 := TRUE; fb_0.EDM2 := TRUE; fb_0.ValveType := TRUE; fb_0.S_StartReset := TRUE; fb_0.Reset := TRUE;
	fb_0();
	failed_0 := NOT ((((((((((((fb_0.Reset_Before AND NOT (fb_0.S_OutControl_Before)) AND fb_0.T_Init.Q) AND NOT (fb_0.T_Monitoring.Q)) AND (fb_0.DiagCode = 34818)) AND fb_0.Ready) AND NOT (fb_0.S_SafeState)) AND NOT (fb_0.S_ValveOut)) AND (fb_0.S_ValveStatus = fb_0.DiagCode)) AND fb_0.SafetyDemand) AND NOT (fb_0.ResetRequest)) AND NOT (fb_0.Error)));
	testState_0 := testState_0 + 1;
190:
	fb_0.Activate := TRUE; fb_0.S_OutControl := TRUE; fb_0.EDM1 := FALSE; fb_0.EDM2 := FALSE; fb_0.ValveType := TRUE; fb_0.S_StartReset := TRUE; fb_0.Reset := FALSE;
	fb_0();
	failed_0 := NOT ((((((((((((NOT (fb_0.Reset_Before) AND fb_0.S_OutControl_Before) AND fb_0.T_Init.Q) AND NOT (fb_0.T_Monitoring.Q)) AND (fb_0.DiagCode = 49200)) AND fb_0.Ready) AND NOT (fb_0.S_SafeState)) AND NOT (fb_0.S_ValveOut)) AND (fb_0.S_ValveStatus = fb_0.DiagCode)) AND NOT (fb_0.SafetyDemand)) AND NOT (fb_0.ResetRequest)) AND fb_0.Error));
	testState_0 := testState_0 + 1;
191:
	fb_0.Activate := TRUE; fb_0.S_OutControl := TRUE; fb_0.EDM1 := FALSE; fb_0.EDM2 := FALSE; fb_0.ValveType := TRUE; fb_0.S_StartReset := TRUE; fb_0.Reset := TRUE;
	fb_0();
	failed_0 := NOT ((((((((((((fb_0.Reset_Before AND fb_0.S_OutControl_Before) AND fb_0.T_Init.Q) AND NOT (fb_0.T_Monitoring.Q)) AND (fb_0.DiagCode = 49200)) AND fb_0.Ready) AND NOT (fb_0.S_SafeState)) AND NOT (fb_0.S_ValveOut)) AND (fb_0.S_ValveStatus = fb_0.DiagCode)) AND NOT (fb_0.SafetyDemand)) AND NOT (fb_0.ResetRequest)) AND fb_0.Error));
	testState_0 := testState_0 + 1;
192:
	fb_0.Activate := TRUE; fb_0.S_OutControl := TRUE; fb_0.EDM1 := FALSE; fb_0.EDM2 := FALSE; fb_0.ValveType := TRUE; fb_0.S_StartReset := TRUE; fb_0.Reset := TRUE;
	fb_0();
	failed_0 := NOT ((((((((((((fb_0.Reset_Before AND fb_0.S_OutControl_Before) AND fb_0.T_Init.Q) AND NOT (fb_0.T_Monitoring.Q)) AND (fb_0.DiagCode = 49201)) AND fb_0.Ready) AND NOT (fb_0.S_SafeState)) AND NOT (fb_0.S_ValveOut)) AND (fb_0.S_ValveStatus = fb_0.DiagCode)) AND NOT (fb_0.SafetyDemand)) AND NOT (fb_0.ResetRequest)) AND fb_0.Error));
	testState_0 := testState_0 + 1;
193:
	fb_0.Activate := TRUE; fb_0.S_OutControl := TRUE; fb_0.EDM1 := FALSE; fb_0.EDM2 := FALSE; fb_0.ValveType := TRUE; fb_0.S_StartReset := TRUE; fb_0.Reset := TRUE;
	fb_0();
	failed_0 := NOT ((((((((((((fb_0.Reset_Before AND fb_0.S_OutControl_Before) AND fb_0.T_Init.Q) AND NOT (fb_0.T_Monitoring.Q)) AND (fb_0.DiagCode = 49201)) AND fb_0.Ready) AND NOT (fb_0.S_SafeState)) AND NOT (fb_0.S_ValveOut)) AND (fb_0.S_ValveStatus = fb_0.DiagCode)) AND NOT (fb_0.SafetyDemand)) AND NOT (fb_0.ResetRequest)) AND fb_0.Error));
	testState_0 := testState_0 + 1;
194:
	fb_0.Activate := TRUE; fb_0.S_OutControl := TRUE; fb_0.EDM1 := FALSE; fb_0.EDM2 := FALSE; fb_0.ValveType := TRUE; fb_0.S_StartReset := TRUE; fb_0.Reset := FALSE;
	fb_0();
	failed_0 := NOT ((((((((((((NOT (fb_0.Reset_Before) AND fb_0.S_OutControl_Before) AND fb_0.T_Init.Q) AND NOT (fb_0.T_Monitoring.Q)) AND (fb_0.DiagCode = 49200)) AND fb_0.Ready) AND NOT (fb_0.S_SafeState)) AND NOT (fb_0.S_ValveOut)) AND (fb_0.S_ValveStatus = fb_0.DiagCode)) AND NOT (fb_0.SafetyDemand)) AND NOT (fb_0.ResetRequest)) AND fb_0.Error));
	testState_0 := testState_0 + 1;
195:
	fb_0.Activate := TRUE; fb_0.S_OutControl := FALSE; fb_0.EDM1 := TRUE; fb_0.EDM2 := TRUE; fb_0.ValveType := TRUE; fb_0.S_StartReset := TRUE; fb_0.Reset := TRUE;
	fb_0();
	failed_0 := NOT ((((((((((((fb_0.Reset_Before AND NOT (fb_0.S_OutControl_Before)) AND fb_0.T_Init.Q) AND NOT (fb_0.T_Monitoring.Q)) AND (fb_0.DiagCode = 34818)) AND fb_0.Ready) AND NOT (fb_0.S_SafeState)) AND NOT (fb_0.S_ValveOut)) AND (fb_0.S_ValveStatus = fb_0.DiagCode)) AND fb_0.SafetyDemand) AND NOT (fb_0.ResetRequest)) AND NOT (fb_0.Error)));
	testState_0 := testState_0 + 1;
196:
	fb_0.Activate := TRUE; fb_0.S_OutControl := TRUE; fb_0.EDM1 := FALSE; fb_0.EDM2 := FALSE; fb_0.ValveType := TRUE; fb_0.S_StartReset := TRUE; fb_0.Reset := FALSE;
	fb_0();
	failed_0 := NOT ((((((((((((NOT (fb_0.Reset_Before) AND fb_0.S_OutControl_Before) AND fb_0.T_Init.Q) AND NOT (fb_0.T_Monitoring.Q)) AND (fb_0.DiagCode = 49200)) AND fb_0.Ready) AND NOT (fb_0.S_SafeState)) AND NOT (fb_0.S_ValveOut)) AND (fb_0.S_ValveStatus = fb_0.DiagCode)) AND NOT (fb_0.SafetyDemand)) AND NOT (fb_0.ResetRequest)) AND fb_0.Error));
	testState_0 := testState_0 + 1;
197:
	fb_0.Activate := TRUE; fb_0.S_OutControl := FALSE; fb_0.EDM1 := FALSE; fb_0.EDM2 := FALSE; fb_0.ValveType := TRUE; fb_0.S_StartReset := TRUE; fb_0.Reset := FALSE;
	fb_0();
	failed_0 := NOT ((((((((((((NOT (fb_0.Reset_Before) AND NOT (fb_0.S_OutControl_Before)) AND fb_0.T_Init.Q) AND NOT (fb_0.T_Monitoring.Q)) AND (fb_0.DiagCode = 50224)) AND fb_0.Ready) AND NOT (fb_0.S_SafeState)) AND NOT (fb_0.S_ValveOut)) AND (fb_0.S_ValveStatus = fb_0.DiagCode)) AND NOT (fb_0.SafetyDemand)) AND fb_0.ResetRequest) AND fb_0.Error));
	testState_0 := testState_0 + 1;
198:
	fb_0.Activate := TRUE; fb_0.S_OutControl := FALSE; fb_0.EDM1 := FALSE; fb_0.EDM2 := FALSE; fb_0.ValveType := TRUE; fb_0.S_StartReset := TRUE; fb_0.Reset := TRUE;
	fb_0();
	failed_0 := NOT ((((((((((((fb_0.Reset_Before AND NOT (fb_0.S_OutControl_Before)) AND fb_0.T_Init.Q) AND NOT (fb_0.T_Monitoring.Q)) AND (fb_0.DiagCode = 50224)) AND fb_0.Ready) AND NOT (fb_0.S_SafeState)) AND NOT (fb_0.S_ValveOut)) AND (fb_0.S_ValveStatus = fb_0.DiagCode)) AND NOT (fb_0.SafetyDemand)) AND fb_0.ResetRequest) AND fb_0.Error));
	testState_0 := testState_0 + 1;
199:
	fb_0.Activate := TRUE; fb_0.S_OutControl := FALSE; fb_0.EDM1 := FALSE; fb_0.EDM2 := FALSE; fb_0.ValveType := TRUE; fb_0.S_StartReset := TRUE; fb_0.Reset := TRUE;
	fb_0();
	failed_0 := NOT ((((((((((((fb_0.Reset_Before AND NOT (fb_0.S_OutControl_Before)) AND fb_0.T_Init.Q) AND NOT (fb_0.T_Monitoring.Q)) AND (fb_0.DiagCode = 49201)) AND fb_0.Ready) AND NOT (fb_0.S_SafeState)) AND NOT (fb_0.S_ValveOut)) AND (fb_0.S_ValveStatus = fb_0.DiagCode)) AND NOT (fb_0.SafetyDemand)) AND NOT (fb_0.ResetRequest)) AND fb_0.Error));
	testState_0 := testState_0 + 1;
200:
	fb_0.Activate := TRUE; fb_0.S_OutControl := FALSE; fb_0.EDM1 := FALSE; fb_0.EDM2 := FALSE; fb_0.ValveType := TRUE; fb_0.S_StartReset := TRUE; fb_0.Reset := FALSE;
	fb_0();
	failed_0 := NOT ((((((((((((NOT (fb_0.Reset_Before) AND NOT (fb_0.S_OutControl_Before)) AND fb_0.T_Init.Q) AND NOT (fb_0.T_Monitoring.Q)) AND (fb_0.DiagCode = 50224)) AND fb_0.Ready) AND NOT (fb_0.S_SafeState)) AND NOT (fb_0.S_ValveOut)) AND (fb_0.S_ValveStatus = fb_0.DiagCode)) AND NOT (fb_0.SafetyDemand)) AND fb_0.ResetRequest) AND fb_0.Error));
	testState_0 := testState_0 + 1;
201:
	fb_0.Activate := TRUE; fb_0.S_OutControl := TRUE; fb_0.EDM1 := FALSE; fb_0.EDM2 := FALSE; fb_0.ValveType := TRUE; fb_0.S_StartReset := TRUE; fb_0.Reset := FALSE;
	fb_0();
	failed_0 := NOT ((((((((((((NOT (fb_0.Reset_Before) AND fb_0.S_OutControl_Before) AND fb_0.T_Init.Q) AND NOT (fb_0.T_Monitoring.Q)) AND (fb_0.DiagCode = 49200)) AND fb_0.Ready) AND NOT (fb_0.S_SafeState)) AND NOT (fb_0.S_ValveOut)) AND (fb_0.S_ValveStatus = fb_0.DiagCode)) AND NOT (fb_0.SafetyDemand)) AND NOT (fb_0.ResetRequest)) AND fb_0.Error));
	testState_0 := testState_0 + 1;
202:
	fb_0.Activate := TRUE; fb_0.S_OutControl := FALSE; fb_0.EDM1 := FALSE; fb_0.EDM2 := FALSE; fb_0.ValveType := TRUE; fb_0.S_StartReset := TRUE; fb_0.Reset := FALSE;
	fb_0();
	failed_0 := NOT ((((((((((((NOT (fb_0.Reset_Before) AND NOT (fb_0.S_OutControl_Before)) AND fb_0.T_Init.Q) AND NOT (fb_0.T_Monitoring.Q)) AND (fb_0.DiagCode = 50224)) AND fb_0.Ready) AND NOT (fb_0.S_SafeState)) AND NOT (fb_0.S_ValveOut)) AND (fb_0.S_ValveStatus = fb_0.DiagCode)) AND NOT (fb_0.SafetyDemand)) AND fb_0.ResetRequest) AND fb_0.Error));
	testState_0 := testState_0 + 1;
203:
	fb_0.Activate := TRUE; fb_0.S_OutControl := FALSE; fb_0.EDM1 := TRUE; fb_0.EDM2 := TRUE; fb_0.ValveType := TRUE; fb_0.S_StartReset := TRUE; fb_0.Reset := TRUE;
	fb_0();
	failed_0 := NOT ((((((((((((fb_0.Reset_Before AND NOT (fb_0.S_OutControl_Before)) AND fb_0.T_Init.Q) AND NOT (fb_0.T_Monitoring.Q)) AND (fb_0.DiagCode = 34818)) AND fb_0.Ready) AND NOT (fb_0.S_SafeState)) AND NOT (fb_0.S_ValveOut)) AND (fb_0.S_ValveStatus = fb_0.DiagCode)) AND fb_0.SafetyDemand) AND NOT (fb_0.ResetRequest)) AND NOT (fb_0.Error)));
	testState_0 := testState_0 + 1;
204:
	fb_0.Activate := TRUE; fb_0.S_OutControl := FALSE; fb_0.EDM1 := TRUE; fb_0.EDM2 := TRUE; fb_0.ValveType := TRUE; fb_0.S_StartReset := TRUE; fb_0.Reset := FALSE;
	fb_0();
	IF fb_0.T_Monitoring.Q THEN
		finished_0 := TRUE;
	ELSE
		testState_0 := testState_0 + 1;
	END_IF
205:
	failed_0 := NOT ((((((((((((NOT (fb_0.Reset_Before) AND NOT (fb_0.S_OutControl_Before)) AND fb_0.T_Init.Q) AND NOT (fb_0.T_Monitoring.Q)) AND (fb_0.DiagCode = 34820)) AND fb_0.Ready) AND fb_0.S_SafeState) AND NOT (fb_0.S_ValveOut)) AND (fb_0.S_ValveStatus = fb_0.DiagCode)) AND fb_0.SafetyDemand) AND NOT (fb_0.ResetRequest)) AND NOT (fb_0.Error)));
	testState_0 := testState_0 + 1;
206:
	fb_0.Activate := TRUE; fb_0.S_OutControl := TRUE; fb_0.EDM1 := TRUE; fb_0.EDM2 := TRUE; fb_0.ValveType := TRUE; fb_0.S_StartReset := TRUE; fb_0.Reset := FALSE;
	fb_0();
	failed_0 := NOT ((((((((((((NOT (fb_0.Reset_Before) AND fb_0.S_OutControl_Before) AND fb_0.T_Init.Q) AND NOT (fb_0.T_Monitoring.Q)) AND (fb_0.DiagCode = 32800)) AND fb_0.Ready) AND NOT (fb_0.S_SafeState)) AND fb_0.S_ValveOut) AND (fb_0.S_ValveStatus = fb_0.DiagCode)) AND NOT (fb_0.SafetyDemand)) AND NOT (fb_0.ResetRequest)) AND NOT (fb_0.Error)));
	testState_0 := testState_0 + 1;
207:
	fb_0.Activate := TRUE; fb_0.S_OutControl := TRUE; fb_0.EDM1 := FALSE; fb_0.EDM2 := FALSE; fb_0.ValveType := TRUE; fb_0.S_StartReset := TRUE; fb_0.Reset := FALSE;
	fb_0();
	IF fb_0.T_Monitoring.Q THEN
		finished_0 := TRUE;
	ELSE
		testState_0 := testState_0 + 1;
	END_IF
208:
	failed_0 := NOT ((((((((((((NOT (fb_0.Reset_Before) AND fb_0.S_OutControl_Before) AND fb_0.T_Init.Q) AND NOT (fb_0.T_Monitoring.Q)) AND (fb_0.DiagCode = 32784)) AND fb_0.Ready) AND NOT (fb_0.S_SafeState)) AND fb_0.S_ValveOut) AND (fb_0.S_ValveStatus = fb_0.DiagCode)) AND NOT (fb_0.SafetyDemand)) AND NOT (fb_0.ResetRequest)) AND NOT (fb_0.Error)));
	testState_0 := testState_0 + 1;
209:
	fb_0.Activate := TRUE; fb_0.S_OutControl := TRUE; fb_0.EDM1 := FALSE; fb_0.EDM2 := FALSE; fb_0.ValveType := TRUE; fb_0.S_StartReset := TRUE; fb_0.Reset := FALSE;
	fb_0();
	failed_0 := NOT ((((((((((((NOT (fb_0.Reset_Before) AND fb_0.S_OutControl_Before) AND fb_0.T_Init.Q) AND NOT (fb_0.T_Monitoring.Q)) AND (fb_0.DiagCode = 32784)) AND fb_0.Ready) AND NOT (fb_0.S_SafeState)) AND fb_0.S_ValveOut) AND (fb_0.S_ValveStatus = fb_0.DiagCode)) AND NOT (fb_0.SafetyDemand)) AND NOT (fb_0.ResetRequest)) AND NOT (fb_0.Error)));
	testState_0 := testState_0 + 1;
210:
	fb_0.Activate := TRUE; fb_0.S_OutControl := FALSE; fb_0.EDM1 := FALSE; fb_0.EDM2 := FALSE; fb_0.ValveType := TRUE; fb_0.S_StartReset := TRUE; fb_0.Reset := FALSE;
	fb_0();
	failed_0 := NOT ((((((((((((NOT (fb_0.Reset_Before) AND NOT (fb_0.S_OutControl_Before)) AND fb_0.T_Init.Q) AND NOT (fb_0.T_Monitoring.Q)) AND (fb_0.DiagCode = 34818)) AND fb_0.Ready) AND NOT (fb_0.S_SafeState)) AND NOT (fb_0.S_ValveOut)) AND (fb_0.S_ValveStatus = fb_0.DiagCode)) AND fb_0.SafetyDemand) AND NOT (fb_0.ResetRequest)) AND NOT (fb_0.Error)));
	testState_0 := testState_0 + 1;
211:
	fb_0.Activate := TRUE; fb_0.S_OutControl := FALSE; fb_0.EDM1 := TRUE; fb_0.EDM2 := TRUE; fb_0.ValveType := TRUE; fb_0.S_StartReset := TRUE; fb_0.Reset := FALSE;
	fb_0();
	IF fb_0.T_Monitoring.Q THEN
		finished_0 := TRUE;
	ELSE
		testState_0 := testState_0 + 1;
	END_IF
212:
	failed_0 := NOT ((((((((((((NOT (fb_0.Reset_Before) AND NOT (fb_0.S_OutControl_Before)) AND fb_0.T_Init.Q) AND NOT (fb_0.T_Monitoring.Q)) AND (fb_0.DiagCode = 34820)) AND fb_0.Ready) AND fb_0.S_SafeState) AND NOT (fb_0.S_ValveOut)) AND (fb_0.S_ValveStatus = fb_0.DiagCode)) AND fb_0.SafetyDemand) AND NOT (fb_0.ResetRequest)) AND NOT (fb_0.Error)));
	testState_0 := testState_0 + 1;
213:
	fb_0.Activate := TRUE; fb_0.S_OutControl := TRUE; fb_0.EDM1 := TRUE; fb_0.EDM2 := TRUE; fb_0.ValveType := TRUE; fb_0.S_StartReset := TRUE; fb_0.Reset := FALSE;
	fb_0();
	failed_0 := NOT ((((((((((((NOT (fb_0.Reset_Before) AND fb_0.S_OutControl_Before) AND fb_0.T_Init.Q) AND NOT (fb_0.T_Monitoring.Q)) AND (fb_0.DiagCode = 32800)) AND fb_0.Ready) AND NOT (fb_0.S_SafeState)) AND fb_0.S_ValveOut) AND (fb_0.S_ValveStatus = fb_0.DiagCode)) AND NOT (fb_0.SafetyDemand)) AND NOT (fb_0.ResetRequest)) AND NOT (fb_0.Error)));
	testState_0 := testState_0 + 1;
214:
	fb_0.Activate := TRUE; fb_0.S_OutControl := TRUE; fb_0.EDM1 := FALSE; fb_0.EDM2 := FALSE; fb_0.ValveType := TRUE; fb_0.S_StartReset := TRUE; fb_0.Reset := FALSE;
	fb_0();
	IF fb_0.T_Monitoring.Q THEN
		finished_0 := TRUE;
	ELSE
		testState_0 := testState_0 + 1;
	END_IF
215:
	failed_0 := NOT ((((((((((((NOT (fb_0.Reset_Before) AND fb_0.S_OutControl_Before) AND fb_0.T_Init.Q) AND NOT (fb_0.T_Monitoring.Q)) AND (fb_0.DiagCode = 32784)) AND fb_0.Ready) AND NOT (fb_0.S_SafeState)) AND fb_0.S_ValveOut) AND (fb_0.S_ValveStatus = fb_0.DiagCode)) AND NOT (fb_0.SafetyDemand)) AND NOT (fb_0.ResetRequest)) AND NOT (fb_0.Error)));
	testState_0 := testState_0 + 1;
216:
	fb_0.Activate := TRUE; fb_0.S_OutControl := TRUE; fb_0.EDM1 := TRUE; fb_0.EDM2 := FALSE; fb_0.ValveType := TRUE; fb_0.S_StartReset := TRUE; fb_0.Reset := FALSE;
	fb_0();
	failed_0 := NOT ((((((((((((NOT (fb_0.Reset_Before) AND fb_0.S_OutControl_Before) AND fb_0.T_Init.Q) AND NOT (fb_0.T_Monitoring.Q)) AND (fb_0.DiagCode = 49264)) AND fb_0.Ready) AND NOT (fb_0.S_SafeState)) AND NOT (fb_0.S_ValveOut)) AND (fb_0.S_ValveStatus = fb_0.DiagCode)) AND NOT (fb_0.SafetyDemand)) AND NOT (fb_0.ResetRequest)) AND fb_0.Error));
	testState_0 := testState_0 + 1;
217:
	fb_0.Activate := TRUE; fb_0.S_OutControl := FALSE; fb_0.EDM1 := TRUE; fb_0.EDM2 := TRUE; fb_0.ValveType := TRUE; fb_0.S_StartReset := TRUE; fb_0.Reset := TRUE;
	fb_0();
	failed_0 := NOT ((((((((((((fb_0.Reset_Before AND NOT (fb_0.S_OutControl_Before)) AND fb_0.T_Init.Q) AND NOT (fb_0.T_Monitoring.Q)) AND (fb_0.DiagCode = 34818)) AND fb_0.Ready) AND NOT (fb_0.S_SafeState)) AND NOT (fb_0.S_ValveOut)) AND (fb_0.S_ValveStatus = fb_0.DiagCode)) AND fb_0.SafetyDemand) AND NOT (fb_0.ResetRequest)) AND NOT (fb_0.Error)));
	testState_0 := testState_0 + 1;
218:
	fb_0.Activate := TRUE; fb_0.S_OutControl := FALSE; fb_0.EDM1 := TRUE; fb_0.EDM2 := TRUE; fb_0.ValveType := TRUE; fb_0.S_StartReset := TRUE; fb_0.Reset := FALSE;
	fb_0();
	IF fb_0.T_Monitoring.Q THEN
		finished_0 := TRUE;
	ELSE
		testState_0 := testState_0 + 1;
	END_IF
219:
	failed_0 := NOT ((((((((((((NOT (fb_0.Reset_Before) AND NOT (fb_0.S_OutControl_Before)) AND fb_0.T_Init.Q) AND NOT (fb_0.T_Monitoring.Q)) AND (fb_0.DiagCode = 34820)) AND fb_0.Ready) AND fb_0.S_SafeState) AND NOT (fb_0.S_ValveOut)) AND (fb_0.S_ValveStatus = fb_0.DiagCode)) AND fb_0.SafetyDemand) AND NOT (fb_0.ResetRequest)) AND NOT (fb_0.Error)));
	testState_0 := testState_0 + 1;
220:
	fb_0.Activate := TRUE; fb_0.S_OutControl := TRUE; fb_0.EDM1 := TRUE; fb_0.EDM2 := TRUE; fb_0.ValveType := TRUE; fb_0.S_StartReset := TRUE; fb_0.Reset := FALSE;
	fb_0();
	failed_0 := NOT ((((((((((((NOT (fb_0.Reset_Before) AND fb_0.S_OutControl_Before) AND fb_0.T_Init.Q) AND NOT (fb_0.T_Monitoring.Q)) AND (fb_0.DiagCode = 32800)) AND fb_0.Ready) AND NOT (fb_0.S_SafeState)) AND fb_0.S_ValveOut) AND (fb_0.S_ValveStatus = fb_0.DiagCode)) AND NOT (fb_0.SafetyDemand)) AND NOT (fb_0.ResetRequest)) AND NOT (fb_0.Error)));
	testState_0 := testState_0 + 1;
221:
	fb_0.Activate := TRUE; fb_0.S_OutControl := TRUE; fb_0.EDM1 := FALSE; fb_0.EDM2 := FALSE; fb_0.ValveType := TRUE; fb_0.S_StartReset := TRUE; fb_0.Reset := FALSE;
	fb_0();
	IF fb_0.T_Monitoring.Q THEN
		finished_0 := TRUE;
	ELSE
		testState_0 := testState_0 + 1;
	END_IF
222:
	failed_0 := NOT ((((((((((((NOT (fb_0.Reset_Before) AND fb_0.S_OutControl_Before) AND fb_0.T_Init.Q) AND NOT (fb_0.T_Monitoring.Q)) AND (fb_0.DiagCode = 32784)) AND fb_0.Ready) AND NOT (fb_0.S_SafeState)) AND fb_0.S_ValveOut) AND (fb_0.S_ValveStatus = fb_0.DiagCode)) AND NOT (fb_0.SafetyDemand)) AND NOT (fb_0.ResetRequest)) AND NOT (fb_0.Error)));
	testState_0 := testState_0 + 1;
223:
	fb_0.Activate := TRUE; fb_0.S_OutControl := TRUE; fb_0.EDM1 := FALSE; fb_0.EDM2 := TRUE; fb_0.ValveType := TRUE; fb_0.S_StartReset := TRUE; fb_0.Reset := FALSE;
	fb_0();
	failed_0 := NOT ((((((((((((NOT (fb_0.Reset_Before) AND fb_0.S_OutControl_Before) AND fb_0.T_Init.Q) AND NOT (fb_0.T_Monitoring.Q)) AND (fb_0.DiagCode = 49280)) AND fb_0.Ready) AND NOT (fb_0.S_SafeState)) AND NOT (fb_0.S_ValveOut)) AND (fb_0.S_ValveStatus = fb_0.DiagCode)) AND NOT (fb_0.SafetyDemand)) AND NOT (fb_0.ResetRequest)) AND fb_0.Error));
	testState_0 := testState_0 + 1;
224:
	fb_0.Activate := TRUE; fb_0.S_OutControl := FALSE; fb_0.EDM1 := TRUE; fb_0.EDM2 := TRUE; fb_0.ValveType := TRUE; fb_0.S_StartReset := TRUE; fb_0.Reset := TRUE;
	fb_0();
	failed_0 := NOT ((((((((((((fb_0.Reset_Before AND NOT (fb_0.S_OutControl_Before)) AND fb_0.T_Init.Q) AND NOT (fb_0.T_Monitoring.Q)) AND (fb_0.DiagCode = 34818)) AND fb_0.Ready) AND NOT (fb_0.S_SafeState)) AND NOT (fb_0.S_ValveOut)) AND (fb_0.S_ValveStatus = fb_0.DiagCode)) AND fb_0.SafetyDemand) AND NOT (fb_0.ResetRequest)) AND NOT (fb_0.Error)));
	testState_0 := testState_0 + 1;
225:
	fb_0.Activate := TRUE; fb_0.S_OutControl := FALSE; fb_0.EDM1 := TRUE; fb_0.EDM2 := TRUE; fb_0.ValveType := TRUE; fb_0.S_StartReset := TRUE; fb_0.Reset := FALSE;
	fb_0();
	IF fb_0.T_Monitoring.Q THEN
		finished_0 := TRUE;
	ELSE
		testState_0 := testState_0 + 1;
	END_IF
226:
	failed_0 := NOT ((((((((((((NOT (fb_0.Reset_Before) AND NOT (fb_0.S_OutControl_Before)) AND fb_0.T_Init.Q) AND NOT (fb_0.T_Monitoring.Q)) AND (fb_0.DiagCode = 34820)) AND fb_0.Ready) AND fb_0.S_SafeState) AND NOT (fb_0.S_ValveOut)) AND (fb_0.S_ValveStatus = fb_0.DiagCode)) AND fb_0.SafetyDemand) AND NOT (fb_0.ResetRequest)) AND NOT (fb_0.Error)));
	testState_0 := testState_0 + 1;
227:
	fb_0.Activate := TRUE; fb_0.S_OutControl := TRUE; fb_0.EDM1 := TRUE; fb_0.EDM2 := TRUE; fb_0.ValveType := TRUE; fb_0.S_StartReset := TRUE; fb_0.Reset := FALSE;
	fb_0();
	failed_0 := NOT ((((((((((((NOT (fb_0.Reset_Before) AND fb_0.S_OutControl_Before) AND fb_0.T_Init.Q) AND NOT (fb_0.T_Monitoring.Q)) AND (fb_0.DiagCode = 32800)) AND fb_0.Ready) AND NOT (fb_0.S_SafeState)) AND fb_0.S_ValveOut) AND (fb_0.S_ValveStatus = fb_0.DiagCode)) AND NOT (fb_0.SafetyDemand)) AND NOT (fb_0.ResetRequest)) AND NOT (fb_0.Error)));
	testState_0 := testState_0 + 1;
228:
	fb_0.Activate := TRUE; fb_0.S_OutControl := TRUE; fb_0.EDM1 := FALSE; fb_0.EDM2 := FALSE; fb_0.ValveType := TRUE; fb_0.S_StartReset := TRUE; fb_0.Reset := FALSE;
	fb_0();
	IF fb_0.T_Monitoring.Q THEN
		finished_0 := TRUE;
	ELSE
		testState_0 := testState_0 + 1;
	END_IF
229:
	failed_0 := NOT ((((((((((((NOT (fb_0.Reset_Before) AND fb_0.S_OutControl_Before) AND fb_0.T_Init.Q) AND NOT (fb_0.T_Monitoring.Q)) AND (fb_0.DiagCode = 32784)) AND fb_0.Ready) AND NOT (fb_0.S_SafeState)) AND fb_0.S_ValveOut) AND (fb_0.S_ValveStatus = fb_0.DiagCode)) AND NOT (fb_0.SafetyDemand)) AND NOT (fb_0.ResetRequest)) AND NOT (fb_0.Error)));
	testState_0 := testState_0 + 1;
230:
	fb_0.Activate := TRUE; fb_0.S_OutControl := TRUE; fb_0.EDM1 := TRUE; fb_0.EDM2 := TRUE; fb_0.ValveType := TRUE; fb_0.S_StartReset := TRUE; fb_0.Reset := FALSE;
	fb_0();
	failed_0 := NOT ((((((((((((NOT (fb_0.Reset_Before) AND fb_0.S_OutControl_Before) AND fb_0.T_Init.Q) AND NOT (fb_0.T_Monitoring.Q)) AND (fb_0.DiagCode = 49296)) AND fb_0.Ready) AND NOT (fb_0.S_SafeState)) AND NOT (fb_0.S_ValveOut)) AND (fb_0.S_ValveStatus = fb_0.DiagCode)) AND NOT (fb_0.SafetyDemand)) AND NOT (fb_0.ResetRequest)) AND fb_0.Error));
	testState_0 := testState_0 + 1;
231:
	fb_0.Activate := TRUE; fb_0.S_OutControl := FALSE; fb_0.EDM1 := TRUE; fb_0.EDM2 := TRUE; fb_0.ValveType := TRUE; fb_0.S_StartReset := TRUE; fb_0.Reset := TRUE;
	fb_0();
	failed_0 := NOT ((((((((((((fb_0.Reset_Before AND NOT (fb_0.S_OutControl_Before)) AND fb_0.T_Init.Q) AND NOT (fb_0.T_Monitoring.Q)) AND (fb_0.DiagCode = 34818)) AND fb_0.Ready) AND NOT (fb_0.S_SafeState)) AND NOT (fb_0.S_ValveOut)) AND (fb_0.S_ValveStatus = fb_0.DiagCode)) AND fb_0.SafetyDemand) AND NOT (fb_0.ResetRequest)) AND NOT (fb_0.Error)));
	testState_0 := testState_0 + 1;
232:
	fb_0.Activate := TRUE; fb_0.S_OutControl := FALSE; fb_0.EDM1 := TRUE; fb_0.EDM2 := TRUE; fb_0.ValveType := TRUE; fb_0.S_StartReset := TRUE; fb_0.Reset := FALSE;
	fb_0();
	failed_0 := NOT ((fb_0.T_Monitoring.Q OR (NOT (fb_0.Reset_Before) AND (NOT (fb_0.S_OutControl_Before) AND (fb_0.T_Init.Q AND (NOT (fb_0.T_Monitoring.Q) AND ((fb_0.DiagCode = 34820) AND (fb_0.Ready AND (fb_0.S_SafeState AND (NOT (fb_0.S_ValveOut) AND ((fb_0.S_ValveStatus = fb_0.DiagCode) AND (fb_0.SafetyDemand AND (NOT (fb_0.ResetRequest) AND NOT (fb_0.Error))))))))))))));
	testState_0 := testState_0 + 1;
233:
	finished_0 := TRUE;
END_CASE
END_IF
